REGION Network 54: PBV-82 CIP ISOLATION
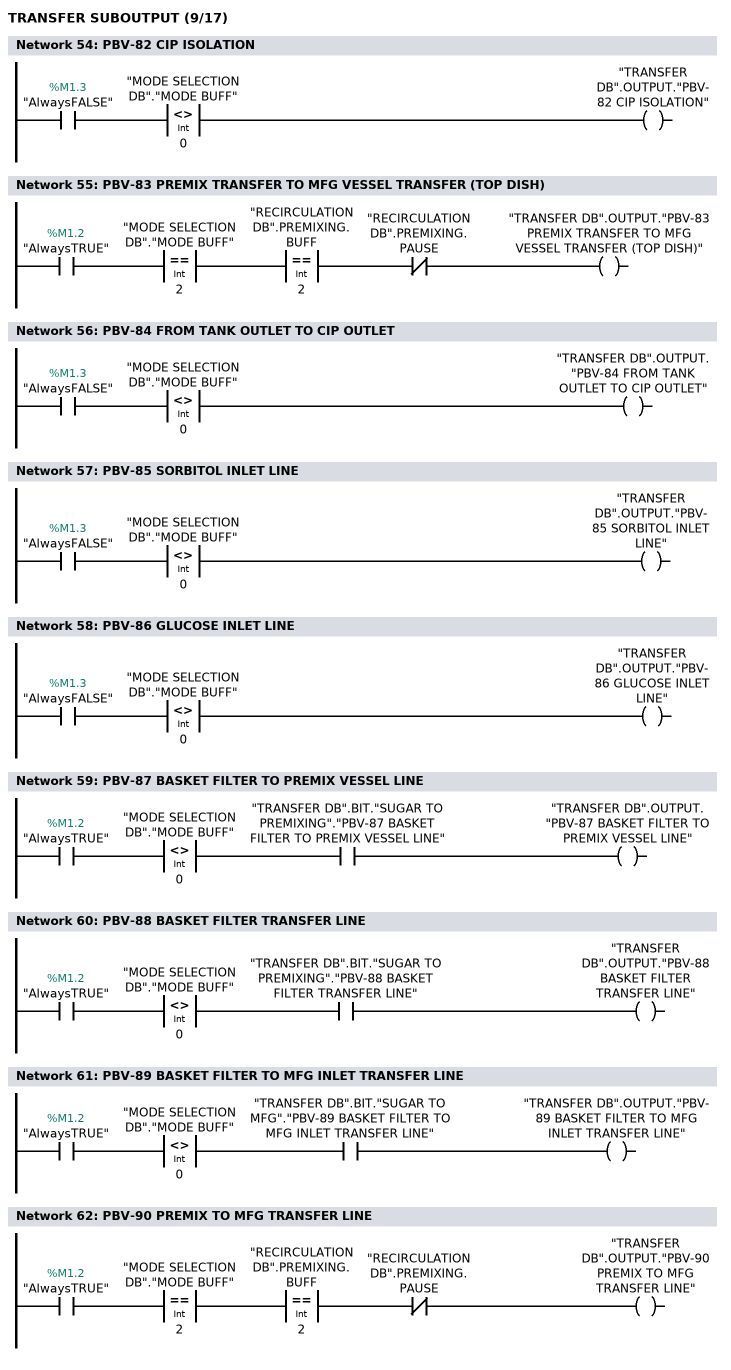
   RUNG wire#powerrail
      Contact( "AlwaysFALSE" )
      { S7_Templates := "SrcType := Int" } NE_Contact(in1 := "MODE SELECTION DB"."MODE BUFF", in2 := 0)
      Coil( "TRANSFER DB".OUTPUT."PBV-82 CIP ISOLATION" )
   END_RUNG
   // the same network as SCL:
   "TRANSFER DB".OUTPUT."PBV-82 CIP ISOLATION" := "AlwaysFALSE" AND ("MODE SELECTION DB"."MODE BUFF" <> 0);
END_REGION

REGION Network 55: PBV-83 PREMIX TRANSFER TO MFG VESSEL TRANSFER (TOP DISH)
   RUNG wire#powerrail
      Contact( "AlwaysTRUE" )
      { S7_Templates := "SrcType := Int" } EQ_Contact(in1 := "MODE SELECTION DB"."MODE BUFF", in2 := 2)
      { S7_Templates := "SrcType := Int" } EQ_Contact(in1 := "RECIRCULATION DB".PREMIXING.BUFF, in2 := 2)
      I_Contact( "RECIRCULATION DB".PREMIXING.PAUSE )
      Coil( "TRANSFER DB".OUTPUT."PBV-83 PREMIX TRANSFER TO MFG VESSEL TRANSFER (TOP DISH)" )
   END_RUNG
   // the same network as SCL:
   "TRANSFER DB".OUTPUT."PBV-83 PREMIX TRANSFER TO MFG VESSEL TRANSFER (TOP DISH)" := "AlwaysTRUE" AND ("MODE SELECTION DB"."MODE BUFF" = 2) AND ("RECIRCULATION DB".PREMIXING.BUFF = 2) AND NOT "RECIRCULATION DB".PREMIXING.PAUSE;
END_REGION

REGION Network 56: PBV-84 FROM TANK OUTLET TO CIP OUTLET
   RUNG wire#powerrail
      Contact( "AlwaysFALSE" )
      { S7_Templates := "SrcType := Int" } NE_Contact(in1 := "MODE SELECTION DB"."MODE BUFF", in2 := 0)
      Coil( "TRANSFER DB".OUTPUT."PBV-84 FROM TANK OUTLET TO CIP OUTLET" )
   END_RUNG
   // the same network as SCL:
   "TRANSFER DB".OUTPUT."PBV-84 FROM TANK OUTLET TO CIP OUTLET" := "AlwaysFALSE" AND ("MODE SELECTION DB"."MODE BUFF" <> 0);
END_REGION

REGION Network 57: PBV-85 SORBITOL INLET LINE
   RUNG wire#powerrail
      Contact( "AlwaysFALSE" )
      { S7_Templates := "SrcType := Int" } NE_Contact(in1 := "MODE SELECTION DB"."MODE BUFF", in2 := 0)
      Coil( "TRANSFER DB".OUTPUT."PBV-85 SORBITOL INLET LINE" )
   END_RUNG
   // the same network as SCL:
   "TRANSFER DB".OUTPUT."PBV-85 SORBITOL INLET LINE" := "AlwaysFALSE" AND ("MODE SELECTION DB"."MODE BUFF" <> 0);
END_REGION

REGION Network 58: PBV-86 GLUCOSE INLET LINE
   RUNG wire#powerrail
      Contact( "AlwaysFALSE" )
      { S7_Templates := "SrcType := Int" } NE_Contact(in1 := "MODE SELECTION DB"."MODE BUFF", in2 := 0)
      Coil( "TRANSFER DB".OUTPUT."PBV-86 GLUCOSE INLET LINE" )
   END_RUNG
   // the same network as SCL:
   "TRANSFER DB".OUTPUT."PBV-86 GLUCOSE INLET LINE" := "AlwaysFALSE" AND ("MODE SELECTION DB"."MODE BUFF" <> 0);
END_REGION

REGION Network 59: PBV-87 BASKET FILTER TO PREMIX VESSEL LINE
   RUNG wire#powerrail
      Contact( "AlwaysTRUE" )
      { S7_Templates := "SrcType := Int" } NE_Contact(in1 := "MODE SELECTION DB"."MODE BUFF", in2 := 0)
      Contact( "TRANSFER DB".BIT."SUGAR TO PREMIXING"."PBV-87 BASKET FILTER TO PREMIX VESSEL LINE" )
      Coil( "TRANSFER DB".OUTPUT."PBV-87 BASKET FILTER TO PREMIX VESSEL LINE" )
   END_RUNG
   // the same network as SCL:
   "TRANSFER DB".OUTPUT."PBV-87 BASKET FILTER TO PREMIX VESSEL LINE" := "AlwaysTRUE" AND ("MODE SELECTION DB"."MODE BUFF" <> 0) AND "TRANSFER DB".BIT."SUGAR TO PREMIXING"."PBV-87 BASKET FILTER TO PREMIX VESSEL LINE";
END_REGION

REGION Network 60: PBV-88 BASKET FILTER TRANSFER LINE
   RUNG wire#powerrail
      Contact( "AlwaysTRUE" )
      { S7_Templates := "SrcType := Int" } NE_Contact(in1 := "MODE SELECTION DB"."MODE BUFF", in2 := 0)
      Contact( "TRANSFER DB".BIT."SUGAR TO PREMIXING"."PBV-88 BASKET FILTER TRANSFER LINE" )
      Coil( "TRANSFER DB".OUTPUT."PBV-88 BASKET FILTER TRANSFER LINE" )
   END_RUNG
   // the same network as SCL:
   "TRANSFER DB".OUTPUT."PBV-88 BASKET FILTER TRANSFER LINE" := "AlwaysTRUE" AND ("MODE SELECTION DB"."MODE BUFF" <> 0) AND "TRANSFER DB".BIT."SUGAR TO PREMIXING"."PBV-88 BASKET FILTER TRANSFER LINE";
END_REGION

REGION Network 61: PBV-89 BASKET FILTER TO MFG INLET TRANSFER LINE
   RUNG wire#powerrail
      Contact( "AlwaysTRUE" )
      { S7_Templates := "SrcType := Int" } NE_Contact(in1 := "MODE SELECTION DB"."MODE BUFF", in2 := 0)
      Contact( "TRANSFER DB".BIT."SUGAR TO MFG"."PBV-89 BASKET FILTER TO MFG INLET TRANSFER LINE" )
      Coil( "TRANSFER DB".OUTPUT."PBV-89 BASKET FILTER TO MFG INLET TRANSFER LINE" )
   END_RUNG
   // the same network as SCL:
   "TRANSFER DB".OUTPUT."PBV-89 BASKET FILTER TO MFG INLET TRANSFER LINE" := "AlwaysTRUE" AND ("MODE SELECTION DB"."MODE BUFF" <> 0) AND "TRANSFER DB".BIT."SUGAR TO MFG"."PBV-89 BASKET FILTER TO MFG INLET TRANSFER LINE";
END_REGION

REGION Network 62: PBV-90 PREMIX TO MFG TRANSFER LINE
   RUNG wire#powerrail
      Contact( "AlwaysTRUE" )
      { S7_Templates := "SrcType := Int" } EQ_Contact(in1 := "MODE SELECTION DB"."MODE BUFF", in2 := 2)
      { S7_Templates := "SrcType := Int" } EQ_Contact(in1 := "RECIRCULATION DB".PREMIXING.BUFF, in2 := 2)
      I_Contact( "RECIRCULATION DB".PREMIXING.PAUSE )
      Coil( "TRANSFER DB".OUTPUT."PBV-90 PREMIX TO MFG TRANSFER LINE" )
   END_RUNG
   // the same network as SCL:
   "TRANSFER DB".OUTPUT."PBV-90 PREMIX TO MFG TRANSFER LINE" := "AlwaysTRUE" AND ("MODE SELECTION DB"."MODE BUFF" = 2) AND ("RECIRCULATION DB".PREMIXING.BUFF = 2) AND NOT "RECIRCULATION DB".PREMIXING.PAUSE;
END_REGION

REGION Network 63: PBV-91 PREMIX TO MFG TRANSFER LINE
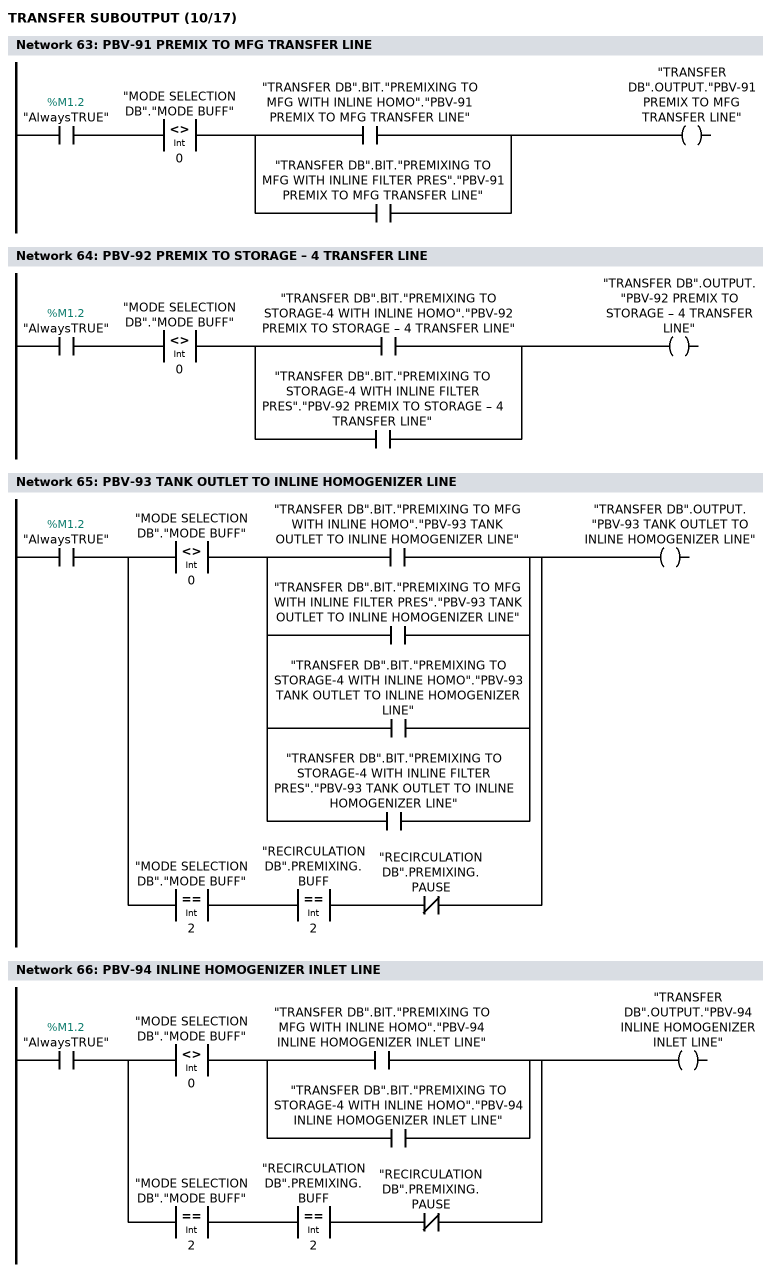
   RUNG wire#powerrail
      Contact( "AlwaysTRUE" )
      { S7_Templates := "SrcType := Int" } NE_Contact(in1 := "MODE SELECTION DB"."MODE BUFF", in2 := 0)
      wire#w1
      Contact( "TRANSFER DB".BIT."PREMIXING TO MFG WITH INLINE HOMO"."PBV-91 PREMIX TO MFG TRANSFER LINE" )
      wire#w2
      Coil( "TRANSFER DB".OUTPUT."PBV-91 PREMIX TO MFG TRANSFER LINE" )
   END_RUNG
   RUNG wire#w1
      Contact( "TRANSFER DB".BIT."PREMIXING TO MFG WITH INLINE FILTER PRES"."PBV-91 PREMIX TO MFG TRANSFER LINE" )
   END_RUNG wire#w2
   // the same network as SCL:
   "TRANSFER DB".OUTPUT."PBV-91 PREMIX TO MFG TRANSFER LINE" := "AlwaysTRUE" AND ("MODE SELECTION DB"."MODE BUFF" <> 0) AND ("TRANSFER DB".BIT."PREMIXING TO MFG WITH INLINE HOMO"."PBV-91 PREMIX TO MFG TRANSFER LINE" OR "TRANSFER DB".BIT."PREMIXING TO MFG WITH INLINE FILTER PRES"."PBV-91 PREMIX TO MFG TRANSFER LINE");
END_REGION

REGION Network 64: PBV-92 PREMIX TO STORAGE – 4 TRANSFER LINE
   RUNG wire#powerrail
      Contact( "AlwaysTRUE" )
      { S7_Templates := "SrcType := Int" } NE_Contact(in1 := "MODE SELECTION DB"."MODE BUFF", in2 := 0)
      wire#w1
      Contact( "TRANSFER DB".BIT."PREMIXING TO STORAGE-4 WITH INLINE HOMO"."PBV-92 PREMIX TO STORAGE – 4 TRANSFER LINE" )
      wire#w2
      Coil( "TRANSFER DB".OUTPUT."PBV-92 PREMIX TO STORAGE – 4 TRANSFER LINE" )
   END_RUNG
   RUNG wire#w1
      Contact( "TRANSFER DB".BIT."PREMIXING TO STORAGE-4 WITH INLINE FILTER PRES"."PBV-92 PREMIX TO STORAGE – 4 TRANSFER LINE" )
   END_RUNG wire#w2
   // the same network as SCL:
   "TRANSFER DB".OUTPUT."PBV-92 PREMIX TO STORAGE – 4 TRANSFER LINE" := "AlwaysTRUE" AND ("MODE SELECTION DB"."MODE BUFF" <> 0) AND ("TRANSFER DB".BIT."PREMIXING TO STORAGE-4 WITH INLINE HOMO"."PBV-92 PREMIX TO STORAGE – 4 TRANSFER LINE" OR "TRANSFER DB".BIT."PREMIXING TO STORAGE-4 WITH INLINE FILTER PRES"."PBV-92 PREMIX TO STORAGE – 4 TRANSFER LINE");
END_REGION

REGION Network 65: PBV-93 TANK OUTLET TO INLINE HOMOGENIZER LINE
   RUNG wire#powerrail
      Contact( "AlwaysTRUE" )
      wire#w1
      { S7_Templates := "SrcType := Int" } NE_Contact(in1 := "MODE SELECTION DB"."MODE BUFF", in2 := 0)
      wire#w2
      Contact( "TRANSFER DB".BIT."PREMIXING TO MFG WITH INLINE HOMO"."PBV-93 TANK OUTLET TO INLINE HOMOGENIZER LINE" )
      wire#w3
      Coil( "TRANSFER DB".OUTPUT."PBV-93 TANK OUTLET TO INLINE HOMOGENIZER LINE" )
   END_RUNG
   RUNG wire#w2
      Contact( "TRANSFER DB".BIT."PREMIXING TO MFG WITH INLINE FILTER PRES"."PBV-93 TANK OUTLET TO INLINE HOMOGENIZER LINE" )
   END_RUNG wire#w3
   RUNG wire#w2
      Contact( "TRANSFER DB".BIT."PREMIXING TO STORAGE-4 WITH INLINE HOMO"."PBV-93 TANK OUTLET TO INLINE HOMOGENIZER LINE" )
   END_RUNG wire#w3
   RUNG wire#w2
      Contact( "TRANSFER DB".BIT."PREMIXING TO STORAGE-4 WITH INLINE FILTER PRES"."PBV-93 TANK OUTLET TO INLINE HOMOGENIZER LINE" )
   END_RUNG wire#w3
   RUNG wire#w1
      { S7_Templates := "SrcType := Int" } EQ_Contact(in1 := "MODE SELECTION DB"."MODE BUFF", in2 := 2)
      { S7_Templates := "SrcType := Int" } EQ_Contact(in1 := "RECIRCULATION DB".PREMIXING.BUFF, in2 := 2)
      I_Contact( "RECIRCULATION DB".PREMIXING.PAUSE )
   END_RUNG wire#w3
   // the same network as SCL:
   "TRANSFER DB".OUTPUT."PBV-93 TANK OUTLET TO INLINE HOMOGENIZER LINE" := "AlwaysTRUE" AND ((("MODE SELECTION DB"."MODE BUFF" <> 0) AND ("TRANSFER DB".BIT."PREMIXING TO MFG WITH INLINE HOMO"."PBV-93 TANK OUTLET TO INLINE HOMOGENIZER LINE" OR "TRANSFER DB".BIT."PREMIXING TO MFG WITH INLINE FILTER PRES"."PBV-93 TANK OUTLET TO INLINE HOMOGENIZER LINE" OR "TRANSFER DB".BIT."PREMIXING TO STORAGE-4 WITH INLINE HOMO"."PBV-93 TANK OUTLET TO INLINE HOMOGENIZER LINE" OR "TRANSFER DB".BIT."PREMIXING TO STORAGE-4 WITH INLINE FILTER PRES"."PBV-93 TANK OUTLET TO INLINE HOMOGENIZER LINE")) OR (("MODE SELECTION DB"."MODE BUFF" = 2) AND ("RECIRCULATION DB".PREMIXING.BUFF = 2) AND NOT "RECIRCULATION DB".PREMIXING.PAUSE));
END_REGION

REGION Network 66: PBV-94 INLINE HOMOGENIZER INLET LINE
   RUNG wire#powerrail
      Contact( "AlwaysTRUE" )
      wire#w1
      { S7_Templates := "SrcType := Int" } NE_Contact(in1 := "MODE SELECTION DB"."MODE BUFF", in2 := 0)
      wire#w2
      Contact( "TRANSFER DB".BIT."PREMIXING TO MFG WITH INLINE HOMO"."PBV-94 INLINE HOMOGENIZER INLET LINE" )
      wire#w3
      Coil( "TRANSFER DB".OUTPUT."PBV-94 INLINE HOMOGENIZER INLET LINE" )
   END_RUNG
   RUNG wire#w2
      Contact( "TRANSFER DB".BIT."PREMIXING TO STORAGE-4 WITH INLINE HOMO"."PBV-94 INLINE HOMOGENIZER INLET LINE" )
   END_RUNG wire#w3
   RUNG wire#w1
      { S7_Templates := "SrcType := Int" } EQ_Contact(in1 := "MODE SELECTION DB"."MODE BUFF", in2 := 2)
      { S7_Templates := "SrcType := Int" } EQ_Contact(in1 := "RECIRCULATION DB".PREMIXING.BUFF, in2 := 2)
      I_Contact( "RECIRCULATION DB".PREMIXING.PAUSE )
   END_RUNG wire#w3
   // the same network as SCL:
   "TRANSFER DB".OUTPUT."PBV-94 INLINE HOMOGENIZER INLET LINE" := "AlwaysTRUE" AND ((("MODE SELECTION DB"."MODE BUFF" <> 0) AND ("TRANSFER DB".BIT."PREMIXING TO MFG WITH INLINE HOMO"."PBV-94 INLINE HOMOGENIZER INLET LINE" OR "TRANSFER DB".BIT."PREMIXING TO STORAGE-4 WITH INLINE HOMO"."PBV-94 INLINE HOMOGENIZER INLET LINE")) OR (("MODE SELECTION DB"."MODE BUFF" = 2) AND ("RECIRCULATION DB".PREMIXING.BUFF = 2) AND NOT "RECIRCULATION DB".PREMIXING.PAUSE));
END_REGION

REGION Network 67: PBV-95 TANK OUTLET TO FILTER PRESS LINE
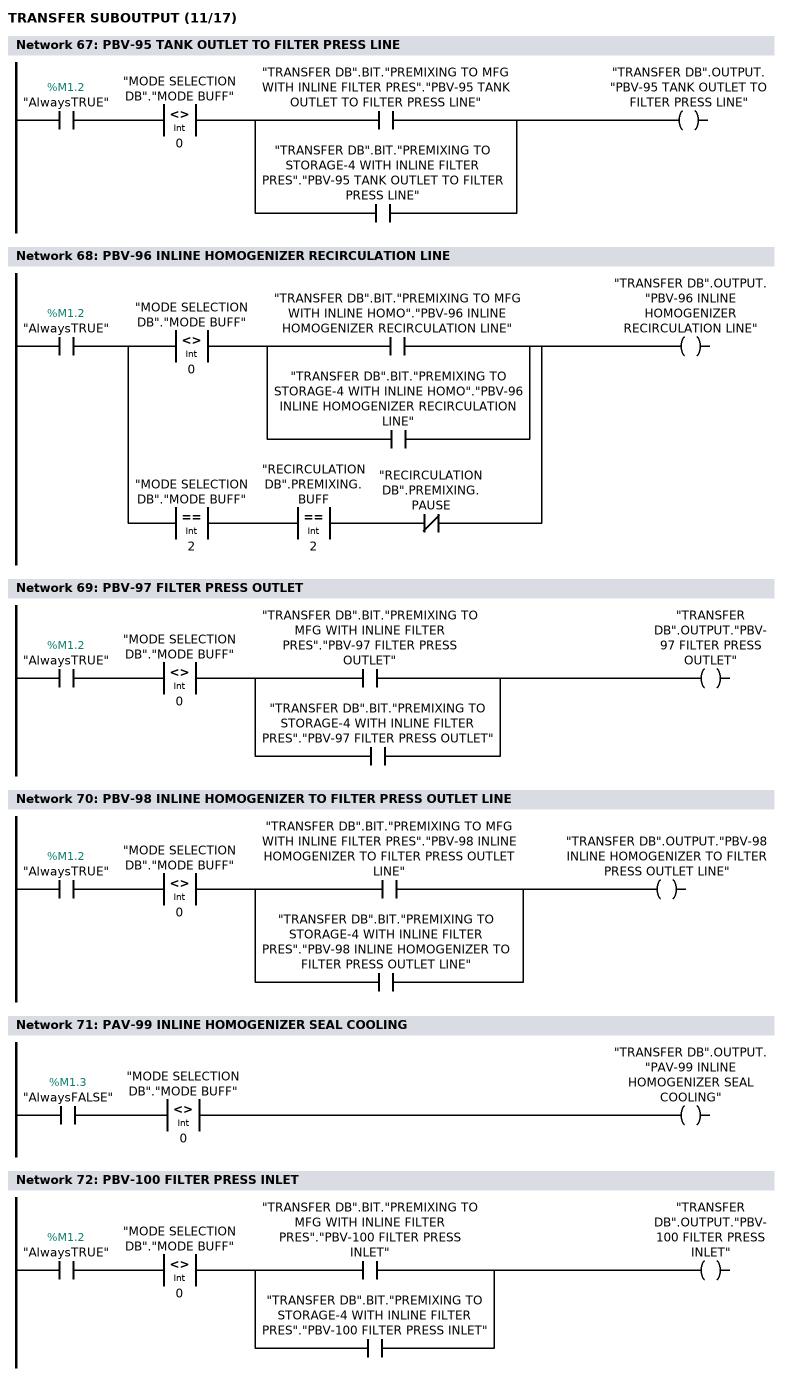
   RUNG wire#powerrail
      Contact( "AlwaysTRUE" )
      { S7_Templates := "SrcType := Int" } NE_Contact(in1 := "MODE SELECTION DB"."MODE BUFF", in2 := 0)
      wire#w1
      Contact( "TRANSFER DB".BIT."PREMIXING TO MFG WITH INLINE FILTER PRES"."PBV-95 TANK OUTLET TO FILTER PRESS LINE" )
      wire#w2
      Coil( "TRANSFER DB".OUTPUT."PBV-95 TANK OUTLET TO FILTER PRESS LINE" )
   END_RUNG
   RUNG wire#w1
      Contact( "TRANSFER DB".BIT."PREMIXING TO STORAGE-4 WITH INLINE FILTER PRES"."PBV-95 TANK OUTLET TO FILTER PRESS LINE" )
   END_RUNG wire#w2
   // the same network as SCL:
   "TRANSFER DB".OUTPUT."PBV-95 TANK OUTLET TO FILTER PRESS LINE" := "AlwaysTRUE" AND ("MODE SELECTION DB"."MODE BUFF" <> 0) AND ("TRANSFER DB".BIT."PREMIXING TO MFG WITH INLINE FILTER PRES"."PBV-95 TANK OUTLET TO FILTER PRESS LINE" OR "TRANSFER DB".BIT."PREMIXING TO STORAGE-4 WITH INLINE FILTER PRES"."PBV-95 TANK OUTLET TO FILTER PRESS LINE");
END_REGION

REGION Network 68: PBV-96 INLINE HOMOGENIZER RECIRCULATION LINE
   RUNG wire#powerrail
      Contact( "AlwaysTRUE" )
      wire#w1
      { S7_Templates := "SrcType := Int" } NE_Contact(in1 := "MODE SELECTION DB"."MODE BUFF", in2 := 0)
      wire#w2
      Contact( "TRANSFER DB".BIT."PREMIXING TO MFG WITH INLINE HOMO"."PBV-96 INLINE HOMOGENIZER RECIRCULATION LINE" )
      wire#w3
      Coil( "TRANSFER DB".OUTPUT."PBV-96 INLINE HOMOGENIZER RECIRCULATION LINE" )
   END_RUNG
   RUNG wire#w2
      Contact( "TRANSFER DB".BIT."PREMIXING TO STORAGE-4 WITH INLINE HOMO"."PBV-96 INLINE HOMOGENIZER RECIRCULATION LINE" )
   END_RUNG wire#w3
   RUNG wire#w1
      { S7_Templates := "SrcType := Int" } EQ_Contact(in1 := "MODE SELECTION DB"."MODE BUFF", in2 := 2)
      { S7_Templates := "SrcType := Int" } EQ_Contact(in1 := "RECIRCULATION DB".PREMIXING.BUFF, in2 := 2)
      I_Contact( "RECIRCULATION DB".PREMIXING.PAUSE )
   END_RUNG wire#w3
   // the same network as SCL:
   "TRANSFER DB".OUTPUT."PBV-96 INLINE HOMOGENIZER RECIRCULATION LINE" := "AlwaysTRUE" AND ((("MODE SELECTION DB"."MODE BUFF" <> 0) AND ("TRANSFER DB".BIT."PREMIXING TO MFG WITH INLINE HOMO"."PBV-96 INLINE HOMOGENIZER RECIRCULATION LINE" OR "TRANSFER DB".BIT."PREMIXING TO STORAGE-4 WITH INLINE HOMO"."PBV-96 INLINE HOMOGENIZER RECIRCULATION LINE")) OR (("MODE SELECTION DB"."MODE BUFF" = 2) AND ("RECIRCULATION DB".PREMIXING.BUFF = 2) AND NOT "RECIRCULATION DB".PREMIXING.PAUSE));
END_REGION

REGION Network 69: PBV-97 FILTER PRESS OUTLET
   RUNG wire#powerrail
      Contact( "AlwaysTRUE" )
      { S7_Templates := "SrcType := Int" } NE_Contact(in1 := "MODE SELECTION DB"."MODE BUFF", in2 := 0)
      wire#w1
      Contact( "TRANSFER DB".BIT."PREMIXING TO MFG WITH INLINE FILTER PRES"."PBV-97 FILTER PRESS OUTLET" )
      wire#w2
      Coil( "TRANSFER DB".OUTPUT."PBV-97 FILTER PRESS OUTLET" )
   END_RUNG
   RUNG wire#w1
      Contact( "TRANSFER DB".BIT."PREMIXING TO STORAGE-4 WITH INLINE FILTER PRES"."PBV-97 FILTER PRESS OUTLET" )
   END_RUNG wire#w2
   // the same network as SCL:
   "TRANSFER DB".OUTPUT."PBV-97 FILTER PRESS OUTLET" := "AlwaysTRUE" AND ("MODE SELECTION DB"."MODE BUFF" <> 0) AND ("TRANSFER DB".BIT."PREMIXING TO MFG WITH INLINE FILTER PRES"."PBV-97 FILTER PRESS OUTLET" OR "TRANSFER DB".BIT."PREMIXING TO STORAGE-4 WITH INLINE FILTER PRES"."PBV-97 FILTER PRESS OUTLET");
END_REGION

REGION Network 70: PBV-98 INLINE HOMOGENIZER TO FILTER PRESS OUTLET LINE
   RUNG wire#powerrail
      Contact( "AlwaysTRUE" )
      { S7_Templates := "SrcType := Int" } NE_Contact(in1 := "MODE SELECTION DB"."MODE BUFF", in2 := 0)
      wire#w1
      Contact( "TRANSFER DB".BIT."PREMIXING TO MFG WITH INLINE FILTER PRES"."PBV-98 INLINE HOMOGENIZER TO FILTER PRESS OUTLET LINE" )
      wire#w2
      Coil( "TRANSFER DB".OUTPUT."PBV-98 INLINE HOMOGENIZER TO FILTER PRESS OUTLET LINE" )
   END_RUNG
   RUNG wire#w1
      Contact( "TRANSFER DB".BIT."PREMIXING TO STORAGE-4 WITH INLINE FILTER PRES"."PBV-98 INLINE HOMOGENIZER TO FILTER PRESS OUTLET LINE" )
   END_RUNG wire#w2
   // the same network as SCL:
   "TRANSFER DB".OUTPUT."PBV-98 INLINE HOMOGENIZER TO FILTER PRESS OUTLET LINE" := "AlwaysTRUE" AND ("MODE SELECTION DB"."MODE BUFF" <> 0) AND ("TRANSFER DB".BIT."PREMIXING TO MFG WITH INLINE FILTER PRES"."PBV-98 INLINE HOMOGENIZER TO FILTER PRESS OUTLET LINE" OR "TRANSFER DB".BIT."PREMIXING TO STORAGE-4 WITH INLINE FILTER PRES"."PBV-98 INLINE HOMOGENIZER TO FILTER PRESS OUTLET LINE");
END_REGION

REGION Network 71: PAV-99 INLINE HOMOGENIZER SEAL COOLING
   RUNG wire#powerrail
      Contact( "AlwaysFALSE" )
      { S7_Templates := "SrcType := Int" } NE_Contact(in1 := "MODE SELECTION DB"."MODE BUFF", in2 := 0)
      Coil( "TRANSFER DB".OUTPUT."PAV-99 INLINE HOMOGENIZER SEAL COOLING" )
   END_RUNG
   // the same network as SCL:
   "TRANSFER DB".OUTPUT."PAV-99 INLINE HOMOGENIZER SEAL COOLING" := "AlwaysFALSE" AND ("MODE SELECTION DB"."MODE BUFF" <> 0);
END_REGION

REGION Network 72: PBV-100 FILTER PRESS INLET
   RUNG wire#powerrail
      Contact( "AlwaysTRUE" )
      { S7_Templates := "SrcType := Int" } NE_Contact(in1 := "MODE SELECTION DB"."MODE BUFF", in2 := 0)
      wire#w1
      Contact( "TRANSFER DB".BIT."PREMIXING TO MFG WITH INLINE FILTER PRES"."PBV-100 FILTER PRESS INLET" )
      wire#w2
      Coil( "TRANSFER DB".OUTPUT."PBV-100 FILTER PRESS INLET" )
   END_RUNG
   RUNG wire#w1
      Contact( "TRANSFER DB".BIT."PREMIXING TO STORAGE-4 WITH INLINE FILTER PRES"."PBV-100 FILTER PRESS INLET" )
   END_RUNG wire#w2
   // the same network as SCL:
   "TRANSFER DB".OUTPUT."PBV-100 FILTER PRESS INLET" := "AlwaysTRUE" AND ("MODE SELECTION DB"."MODE BUFF" <> 0) AND ("TRANSFER DB".BIT."PREMIXING TO MFG WITH INLINE FILTER PRES"."PBV-100 FILTER PRESS INLET" OR "TRANSFER DB".BIT."PREMIXING TO STORAGE-4 WITH INLINE FILTER PRES"."PBV-100 FILTER PRESS INLET");
END_REGION

REGION Network 73: PBV-101 SUGAR MELTING TO MFG TRANSFER (TOP DISH)
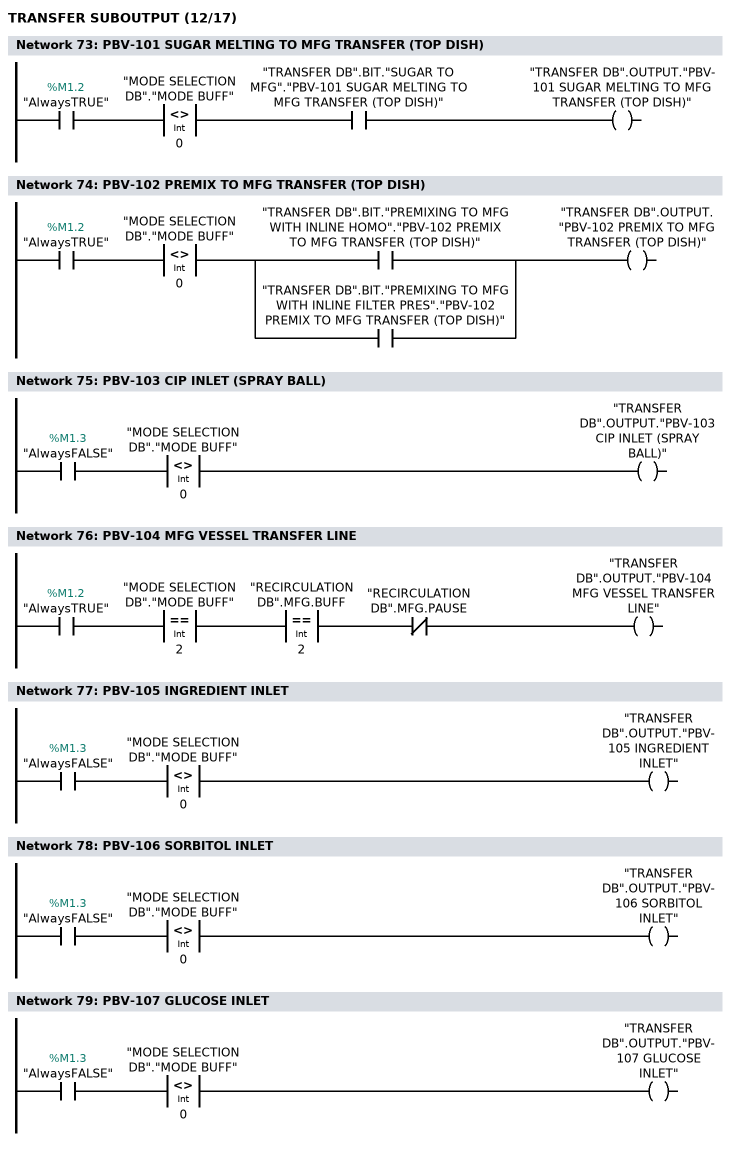
   RUNG wire#powerrail
      Contact( "AlwaysTRUE" )
      { S7_Templates := "SrcType := Int" } NE_Contact(in1 := "MODE SELECTION DB"."MODE BUFF", in2 := 0)
      Contact( "TRANSFER DB".BIT."SUGAR TO MFG"."PBV-101 SUGAR MELTING TO MFG TRANSFER (TOP DISH)" )
      Coil( "TRANSFER DB".OUTPUT."PBV-101 SUGAR MELTING TO MFG TRANSFER (TOP DISH)" )
   END_RUNG
   // the same network as SCL:
   "TRANSFER DB".OUTPUT."PBV-101 SUGAR MELTING TO MFG TRANSFER (TOP DISH)" := "AlwaysTRUE" AND ("MODE SELECTION DB"."MODE BUFF" <> 0) AND "TRANSFER DB".BIT."SUGAR TO MFG"."PBV-101 SUGAR MELTING TO MFG TRANSFER (TOP DISH)";
END_REGION

REGION Network 74: PBV-102 PREMIX TO MFG TRANSFER (TOP DISH)
   RUNG wire#powerrail
      Contact( "AlwaysTRUE" )
      { S7_Templates := "SrcType := Int" } NE_Contact(in1 := "MODE SELECTION DB"."MODE BUFF", in2 := 0)
      wire#w1
      Contact( "TRANSFER DB".BIT."PREMIXING TO MFG WITH INLINE HOMO"."PBV-102 PREMIX TO MFG TRANSFER (TOP DISH)" )
      wire#w2
      Coil( "TRANSFER DB".OUTPUT."PBV-102 PREMIX TO MFG TRANSFER (TOP DISH)" )
   END_RUNG
   RUNG wire#w1
      Contact( "TRANSFER DB".BIT."PREMIXING TO MFG WITH INLINE FILTER PRES"."PBV-102 PREMIX TO MFG TRANSFER (TOP DISH)" )
   END_RUNG wire#w2
   // the same network as SCL:
   "TRANSFER DB".OUTPUT."PBV-102 PREMIX TO MFG TRANSFER (TOP DISH)" := "AlwaysTRUE" AND ("MODE SELECTION DB"."MODE BUFF" <> 0) AND ("TRANSFER DB".BIT."PREMIXING TO MFG WITH INLINE HOMO"."PBV-102 PREMIX TO MFG TRANSFER (TOP DISH)" OR "TRANSFER DB".BIT."PREMIXING TO MFG WITH INLINE FILTER PRES"."PBV-102 PREMIX TO MFG TRANSFER (TOP DISH)");
END_REGION

REGION Network 75: PBV-103 CIP INLET (SPRAY BALL)
   RUNG wire#powerrail
      Contact( "AlwaysFALSE" )
      { S7_Templates := "SrcType := Int" } NE_Contact(in1 := "MODE SELECTION DB"."MODE BUFF", in2 := 0)
      Coil( "TRANSFER DB".OUTPUT."PBV-103 CIP INLET (SPRAY BALL)" )
   END_RUNG
   // the same network as SCL:
   "TRANSFER DB".OUTPUT."PBV-103 CIP INLET (SPRAY BALL)" := "AlwaysFALSE" AND ("MODE SELECTION DB"."MODE BUFF" <> 0);
END_REGION

REGION Network 76: PBV-104 MFG VESSEL TRANSFER LINE
   RUNG wire#powerrail
      Contact( "AlwaysTRUE" )
      { S7_Templates := "SrcType := Int" } EQ_Contact(in1 := "MODE SELECTION DB"."MODE BUFF", in2 := 2)
      { S7_Templates := "SrcType := Int" } EQ_Contact(in1 := "RECIRCULATION DB".MFG.BUFF, in2 := 2)
      I_Contact( "RECIRCULATION DB".MFG.PAUSE )
      Coil( "TRANSFER DB".OUTPUT."PBV-104 MFG VESSEL TRANSFER LINE" )
   END_RUNG
   // the same network as SCL:
   "TRANSFER DB".OUTPUT."PBV-104 MFG VESSEL TRANSFER LINE" := "AlwaysTRUE" AND ("MODE SELECTION DB"."MODE BUFF" = 2) AND ("RECIRCULATION DB".MFG.BUFF = 2) AND NOT "RECIRCULATION DB".MFG.PAUSE;
END_REGION

REGION Network 77: PBV-105 INGREDIENT INLET
   RUNG wire#powerrail
      Contact( "AlwaysFALSE" )
      { S7_Templates := "SrcType := Int" } NE_Contact(in1 := "MODE SELECTION DB"."MODE BUFF", in2 := 0)
      Coil( "TRANSFER DB".OUTPUT."PBV-105 INGREDIENT INLET" )
   END_RUNG
   // the same network as SCL:
   "TRANSFER DB".OUTPUT."PBV-105 INGREDIENT INLET" := "AlwaysFALSE" AND ("MODE SELECTION DB"."MODE BUFF" <> 0);
END_REGION

REGION Network 78: PBV-106 SORBITOL INLET
   RUNG wire#powerrail
      Contact( "AlwaysFALSE" )
      { S7_Templates := "SrcType := Int" } NE_Contact(in1 := "MODE SELECTION DB"."MODE BUFF", in2 := 0)
      Coil( "TRANSFER DB".OUTPUT."PBV-106 SORBITOL INLET" )
   END_RUNG
   // the same network as SCL:
   "TRANSFER DB".OUTPUT."PBV-106 SORBITOL INLET" := "AlwaysFALSE" AND ("MODE SELECTION DB"."MODE BUFF" <> 0);
END_REGION

REGION Network 79: PBV-107 GLUCOSE INLET
   RUNG wire#powerrail
      Contact( "AlwaysFALSE" )
      { S7_Templates := "SrcType := Int" } NE_Contact(in1 := "MODE SELECTION DB"."MODE BUFF", in2 := 0)
      Coil( "TRANSFER DB".OUTPUT."PBV-107 GLUCOSE INLET" )
   END_RUNG
   // the same network as SCL:
   "TRANSFER DB".OUTPUT."PBV-107 GLUCOSE INLET" := "AlwaysFALSE" AND ("MODE SELECTION DB"."MODE BUFF" <> 0);
END_REGION

REGION Network 80: PBV-108 INLINE HOMOGENIZER TO FILTER PRESS INLET LINE
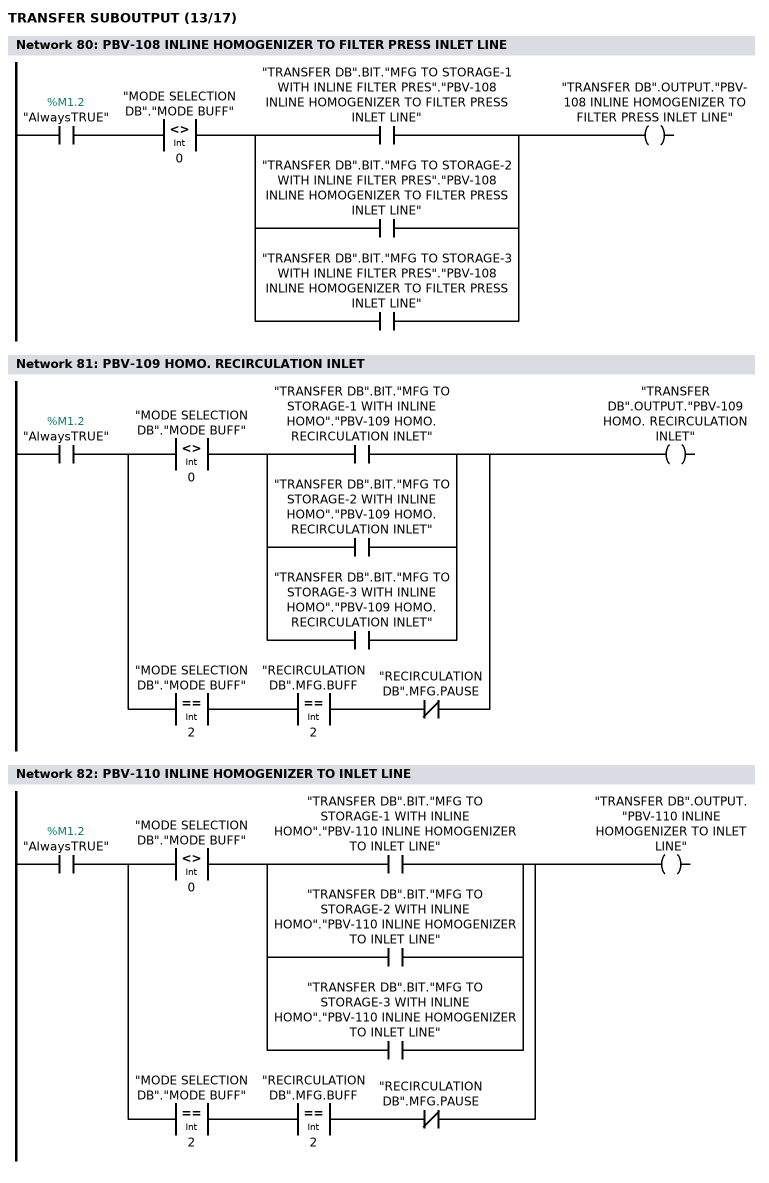
   RUNG wire#powerrail
      Contact( "AlwaysTRUE" )
      { S7_Templates := "SrcType := Int" } NE_Contact(in1 := "MODE SELECTION DB"."MODE BUFF", in2 := 0)
      wire#w1
      Contact( "TRANSFER DB".BIT."MFG TO STORAGE-1 WITH INLINE FILTER PRES"."PBV-108 INLINE HOMOGENIZER TO FILTER PRESS INLET LINE" )
      wire#w2
      Coil( "TRANSFER DB".OUTPUT."PBV-108 INLINE HOMOGENIZER TO FILTER PRESS INLET LINE" )
   END_RUNG
   RUNG wire#w1
      Contact( "TRANSFER DB".BIT."MFG TO STORAGE-2 WITH INLINE FILTER PRES"."PBV-108 INLINE HOMOGENIZER TO FILTER PRESS INLET LINE" )
   END_RUNG wire#w2
   RUNG wire#w1
      Contact( "TRANSFER DB".BIT."MFG TO STORAGE-3 WITH INLINE FILTER PRES"."PBV-108 INLINE HOMOGENIZER TO FILTER PRESS INLET LINE" )
   END_RUNG wire#w2
   // the same network as SCL:
   "TRANSFER DB".OUTPUT."PBV-108 INLINE HOMOGENIZER TO FILTER PRESS INLET LINE" := "AlwaysTRUE" AND ("MODE SELECTION DB"."MODE BUFF" <> 0) AND ("TRANSFER DB".BIT."MFG TO STORAGE-1 WITH INLINE FILTER PRES"."PBV-108 INLINE HOMOGENIZER TO FILTER PRESS INLET LINE" OR "TRANSFER DB".BIT."MFG TO STORAGE-2 WITH INLINE FILTER PRES"."PBV-108 INLINE HOMOGENIZER TO FILTER PRESS INLET LINE" OR "TRANSFER DB".BIT."MFG TO STORAGE-3 WITH INLINE FILTER PRES"."PBV-108 INLINE HOMOGENIZER TO FILTER PRESS INLET LINE");
END_REGION

REGION Network 81: PBV-109 HOMO. RECIRCULATION INLET
   RUNG wire#powerrail
      Contact( "AlwaysTRUE" )
      wire#w1
      { S7_Templates := "SrcType := Int" } NE_Contact(in1 := "MODE SELECTION DB"."MODE BUFF", in2 := 0)
      wire#w2
      Contact( "TRANSFER DB".BIT."MFG TO STORAGE-1 WITH INLINE HOMO"."PBV-109 HOMO. RECIRCULATION INLET" )
      wire#w3
      Coil( "TRANSFER DB".OUTPUT."PBV-109 HOMO. RECIRCULATION INLET" )
   END_RUNG
   RUNG wire#w2
      Contact( "TRANSFER DB".BIT."MFG TO STORAGE-2 WITH INLINE HOMO"."PBV-109 HOMO. RECIRCULATION INLET" )
   END_RUNG wire#w3
   RUNG wire#w2
      Contact( "TRANSFER DB".BIT."MFG TO STORAGE-3 WITH INLINE HOMO"."PBV-109 HOMO. RECIRCULATION INLET" )
   END_RUNG wire#w3
   RUNG wire#w1
      { S7_Templates := "SrcType := Int" } EQ_Contact(in1 := "MODE SELECTION DB"."MODE BUFF", in2 := 2)
      { S7_Templates := "SrcType := Int" } EQ_Contact(in1 := "RECIRCULATION DB".MFG.BUFF, in2 := 2)
      I_Contact( "RECIRCULATION DB".MFG.PAUSE )
   END_RUNG wire#w3
   // the same network as SCL:
   "TRANSFER DB".OUTPUT."PBV-109 HOMO. RECIRCULATION INLET" := "AlwaysTRUE" AND ((("MODE SELECTION DB"."MODE BUFF" <> 0) AND ("TRANSFER DB".BIT."MFG TO STORAGE-1 WITH INLINE HOMO"."PBV-109 HOMO. RECIRCULATION INLET" OR "TRANSFER DB".BIT."MFG TO STORAGE-2 WITH INLINE HOMO"."PBV-109 HOMO. RECIRCULATION INLET" OR "TRANSFER DB".BIT."MFG TO STORAGE-3 WITH INLINE HOMO"."PBV-109 HOMO. RECIRCULATION INLET")) OR (("MODE SELECTION DB"."MODE BUFF" = 2) AND ("RECIRCULATION DB".MFG.BUFF = 2) AND NOT "RECIRCULATION DB".MFG.PAUSE));
END_REGION

REGION Network 82: PBV-110 INLINE HOMOGENIZER TO INLET LINE
   RUNG wire#powerrail
      Contact( "AlwaysTRUE" )
      wire#w1
      { S7_Templates := "SrcType := Int" } NE_Contact(in1 := "MODE SELECTION DB"."MODE BUFF", in2 := 0)
      wire#w2
      Contact( "TRANSFER DB".BIT."MFG TO STORAGE-1 WITH INLINE HOMO"."PBV-110 INLINE HOMOGENIZER TO INLET LINE" )
      wire#w3
      Coil( "TRANSFER DB".OUTPUT."PBV-110 INLINE HOMOGENIZER TO INLET LINE" )
   END_RUNG
   RUNG wire#w2
      Contact( "TRANSFER DB".BIT."MFG TO STORAGE-2 WITH INLINE HOMO"."PBV-110 INLINE HOMOGENIZER TO INLET LINE" )
   END_RUNG wire#w3
   RUNG wire#w2
      Contact( "TRANSFER DB".BIT."MFG TO STORAGE-3 WITH INLINE HOMO"."PBV-110 INLINE HOMOGENIZER TO INLET LINE" )
   END_RUNG wire#w3
   RUNG wire#w1
      { S7_Templates := "SrcType := Int" } EQ_Contact(in1 := "MODE SELECTION DB"."MODE BUFF", in2 := 2)
      { S7_Templates := "SrcType := Int" } EQ_Contact(in1 := "RECIRCULATION DB".MFG.BUFF, in2 := 2)
      I_Contact( "RECIRCULATION DB".MFG.PAUSE )
   END_RUNG wire#w3
   // the same network as SCL:
   "TRANSFER DB".OUTPUT."PBV-110 INLINE HOMOGENIZER TO INLET LINE" := "AlwaysTRUE" AND ((("MODE SELECTION DB"."MODE BUFF" <> 0) AND ("TRANSFER DB".BIT."MFG TO STORAGE-1 WITH INLINE HOMO"."PBV-110 INLINE HOMOGENIZER TO INLET LINE" OR "TRANSFER DB".BIT."MFG TO STORAGE-2 WITH INLINE HOMO"."PBV-110 INLINE HOMOGENIZER TO INLET LINE" OR "TRANSFER DB".BIT."MFG TO STORAGE-3 WITH INLINE HOMO"."PBV-110 INLINE HOMOGENIZER TO INLET LINE")) OR (("MODE SELECTION DB"."MODE BUFF" = 2) AND ("RECIRCULATION DB".MFG.BUFF = 2) AND NOT "RECIRCULATION DB".MFG.PAUSE));
END_REGION

REGION Network 83: PBV-111 FILTER PRESS OUTLER VALVE
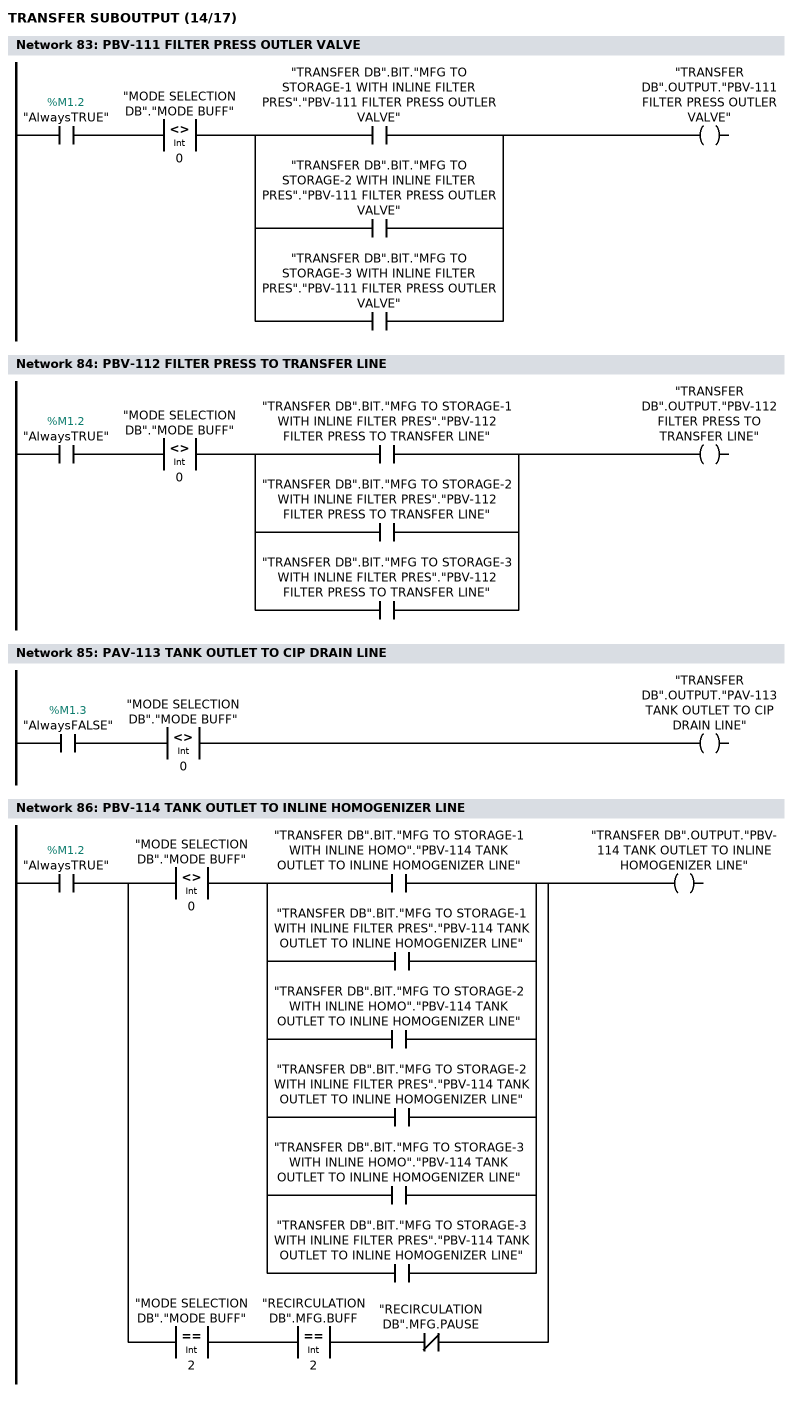
   RUNG wire#powerrail
      Contact( "AlwaysTRUE" )
      { S7_Templates := "SrcType := Int" } NE_Contact(in1 := "MODE SELECTION DB"."MODE BUFF", in2 := 0)
      wire#w1
      Contact( "TRANSFER DB".BIT."MFG TO STORAGE-1 WITH INLINE FILTER PRES"."PBV-111 FILTER PRESS OUTLER VALVE" )
      wire#w2
      Coil( "TRANSFER DB".OUTPUT."PBV-111 FILTER PRESS OUTLER VALVE" )
   END_RUNG
   RUNG wire#w1
      Contact( "TRANSFER DB".BIT."MFG TO STORAGE-2 WITH INLINE FILTER PRES"."PBV-111 FILTER PRESS OUTLER VALVE" )
   END_RUNG wire#w2
   RUNG wire#w1
      Contact( "TRANSFER DB".BIT."MFG TO STORAGE-3 WITH INLINE FILTER PRES"."PBV-111 FILTER PRESS OUTLER VALVE" )
   END_RUNG wire#w2
   // the same network as SCL:
   "TRANSFER DB".OUTPUT."PBV-111 FILTER PRESS OUTLER VALVE" := "AlwaysTRUE" AND ("MODE SELECTION DB"."MODE BUFF" <> 0) AND ("TRANSFER DB".BIT."MFG TO STORAGE-1 WITH INLINE FILTER PRES"."PBV-111 FILTER PRESS OUTLER VALVE" OR "TRANSFER DB".BIT."MFG TO STORAGE-2 WITH INLINE FILTER PRES"."PBV-111 FILTER PRESS OUTLER VALVE" OR "TRANSFER DB".BIT."MFG TO STORAGE-3 WITH INLINE FILTER PRES"."PBV-111 FILTER PRESS OUTLER VALVE");
END_REGION

REGION Network 84: PBV-112 FILTER PRESS TO TRANSFER LINE
   RUNG wire#powerrail
      Contact( "AlwaysTRUE" )
      { S7_Templates := "SrcType := Int" } NE_Contact(in1 := "MODE SELECTION DB"."MODE BUFF", in2 := 0)
      wire#w1
      Contact( "TRANSFER DB".BIT."MFG TO STORAGE-1 WITH INLINE FILTER PRES"."PBV-112 FILTER PRESS TO TRANSFER LINE" )
      wire#w2
      Coil( "TRANSFER DB".OUTPUT."PBV-112 FILTER PRESS TO TRANSFER LINE" )
   END_RUNG
   RUNG wire#w1
      Contact( "TRANSFER DB".BIT."MFG TO STORAGE-2 WITH INLINE FILTER PRES"."PBV-112 FILTER PRESS TO TRANSFER LINE" )
   END_RUNG wire#w2
   RUNG wire#w1
      Contact( "TRANSFER DB".BIT."MFG TO STORAGE-3 WITH INLINE FILTER PRES"."PBV-112 FILTER PRESS TO TRANSFER LINE" )
   END_RUNG wire#w2
   // the same network as SCL:
   "TRANSFER DB".OUTPUT."PBV-112 FILTER PRESS TO TRANSFER LINE" := "AlwaysTRUE" AND ("MODE SELECTION DB"."MODE BUFF" <> 0) AND ("TRANSFER DB".BIT."MFG TO STORAGE-1 WITH INLINE FILTER PRES"."PBV-112 FILTER PRESS TO TRANSFER LINE" OR "TRANSFER DB".BIT."MFG TO STORAGE-2 WITH INLINE FILTER PRES"."PBV-112 FILTER PRESS TO TRANSFER LINE" OR "TRANSFER DB".BIT."MFG TO STORAGE-3 WITH INLINE FILTER PRES"."PBV-112 FILTER PRESS TO TRANSFER LINE");
END_REGION

REGION Network 85: PAV-113 TANK OUTLET TO CIP DRAIN LINE
   RUNG wire#powerrail
      Contact( "AlwaysFALSE" )
      { S7_Templates := "SrcType := Int" } NE_Contact(in1 := "MODE SELECTION DB"."MODE BUFF", in2 := 0)
      Coil( "TRANSFER DB".OUTPUT."PAV-113 TANK OUTLET TO CIP DRAIN LINE" )
   END_RUNG
   // the same network as SCL:
   "TRANSFER DB".OUTPUT."PAV-113 TANK OUTLET TO CIP DRAIN LINE" := "AlwaysFALSE" AND ("MODE SELECTION DB"."MODE BUFF" <> 0);
END_REGION

REGION Network 86: PBV-114 TANK OUTLET TO INLINE HOMOGENIZER LINE
   RUNG wire#powerrail
      Contact( "AlwaysTRUE" )
      wire#w1
      { S7_Templates := "SrcType := Int" } NE_Contact(in1 := "MODE SELECTION DB"."MODE BUFF", in2 := 0)
      wire#w2
      Contact( "TRANSFER DB".BIT."MFG TO STORAGE-1 WITH INLINE HOMO"."PBV-114 TANK OUTLET TO INLINE HOMOGENIZER LINE" )
      wire#w3
      Coil( "TRANSFER DB".OUTPUT."PBV-114 TANK OUTLET TO INLINE HOMOGENIZER LINE" )
   END_RUNG
   RUNG wire#w2
      Contact( "TRANSFER DB".BIT."MFG TO STORAGE-1 WITH INLINE FILTER PRES"."PBV-114 TANK OUTLET TO INLINE HOMOGENIZER LINE" )
   END_RUNG wire#w3
   RUNG wire#w2
      Contact( "TRANSFER DB".BIT."MFG TO STORAGE-2 WITH INLINE HOMO"."PBV-114 TANK OUTLET TO INLINE HOMOGENIZER LINE" )
   END_RUNG wire#w3
   RUNG wire#w2
      Contact( "TRANSFER DB".BIT."MFG TO STORAGE-2 WITH INLINE FILTER PRES"."PBV-114 TANK OUTLET TO INLINE HOMOGENIZER LINE" )
   END_RUNG wire#w3
   RUNG wire#w2
      Contact( "TRANSFER DB".BIT."MFG TO STORAGE-3 WITH INLINE HOMO"."PBV-114 TANK OUTLET TO INLINE HOMOGENIZER LINE" )
   END_RUNG wire#w3
   RUNG wire#w2
      Contact( "TRANSFER DB".BIT."MFG TO STORAGE-3 WITH INLINE FILTER PRES"."PBV-114 TANK OUTLET TO INLINE HOMOGENIZER LINE" )
   END_RUNG wire#w3
   RUNG wire#w1
      { S7_Templates := "SrcType := Int" } EQ_Contact(in1 := "MODE SELECTION DB"."MODE BUFF", in2 := 2)
      { S7_Templates := "SrcType := Int" } EQ_Contact(in1 := "RECIRCULATION DB".MFG.BUFF, in2 := 2)
      I_Contact( "RECIRCULATION DB".MFG.PAUSE )
   END_RUNG wire#w3
   // the same network as SCL:
   "TRANSFER DB".OUTPUT."PBV-114 TANK OUTLET TO INLINE HOMOGENIZER LINE" := "AlwaysTRUE" AND ((("MODE SELECTION DB"."MODE BUFF" <> 0) AND ("TRANSFER DB".BIT."MFG TO STORAGE-1 WITH INLINE HOMO"."PBV-114 TANK OUTLET TO INLINE HOMOGENIZER LINE" OR "TRANSFER DB".BIT."MFG TO STORAGE-1 WITH INLINE FILTER PRES"."PBV-114 TANK OUTLET TO INLINE HOMOGENIZER LINE" OR "TRANSFER DB".BIT."MFG TO STORAGE-2 WITH INLINE HOMO"."PBV-114 TANK OUTLET TO INLINE HOMOGENIZER LINE" OR "TRANSFER DB".BIT."MFG TO STORAGE-2 WITH INLINE FILTER PRES"."PBV-114 TANK OUTLET TO INLINE HOMOGENIZER LINE" OR "TRANSFER DB".BIT."MFG TO STORAGE-3 WITH INLINE HOMO"."PBV-114 TANK OUTLET TO INLINE HOMOGENIZER LINE" OR "TRANSFER DB".BIT."MFG TO STORAGE-3 WITH INLINE FILTER PRES"."PBV-114 TANK OUTLET TO INLINE HOMOGENIZER LINE")) OR (("MODE SELECTION DB"."MODE BUFF" = 2) AND ("RECIRCULATION DB".MFG.BUFF = 2) AND NOT "RECIRCULATION DB".MFG.PAUSE));
END_REGION

REGION Network 87: PBV-115 MFG TO STORAGE – 1 TRANSFER LINE
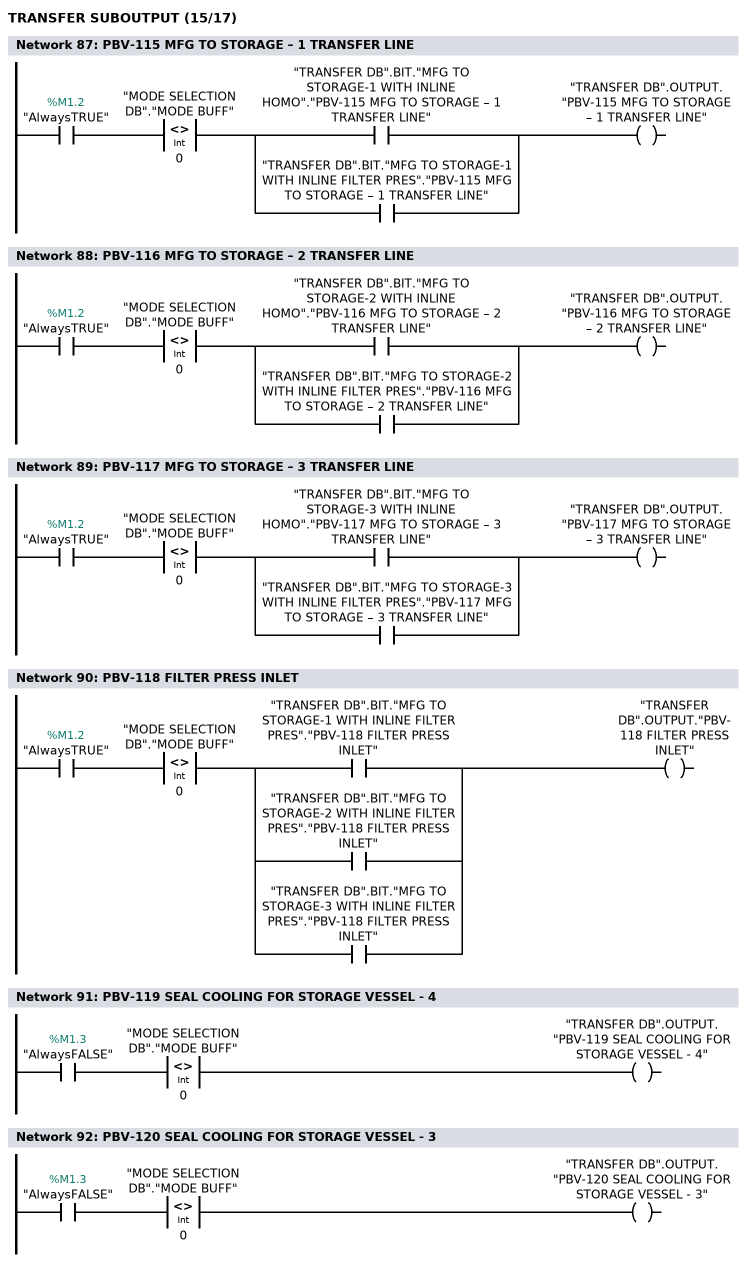
   RUNG wire#powerrail
      Contact( "AlwaysTRUE" )
      { S7_Templates := "SrcType := Int" } NE_Contact(in1 := "MODE SELECTION DB"."MODE BUFF", in2 := 0)
      wire#w1
      Contact( "TRANSFER DB".BIT."MFG TO STORAGE-1 WITH INLINE HOMO"."PBV-115 MFG TO STORAGE – 1 TRANSFER LINE" )
      wire#w2
      Coil( "TRANSFER DB".OUTPUT."PBV-115 MFG TO STORAGE – 1 TRANSFER LINE" )
   END_RUNG
   RUNG wire#w1
      Contact( "TRANSFER DB".BIT."MFG TO STORAGE-1 WITH INLINE FILTER PRES"."PBV-115 MFG TO STORAGE – 1 TRANSFER LINE" )
   END_RUNG wire#w2
   // the same network as SCL:
   "TRANSFER DB".OUTPUT."PBV-115 MFG TO STORAGE – 1 TRANSFER LINE" := "AlwaysTRUE" AND ("MODE SELECTION DB"."MODE BUFF" <> 0) AND ("TRANSFER DB".BIT."MFG TO STORAGE-1 WITH INLINE HOMO"."PBV-115 MFG TO STORAGE – 1 TRANSFER LINE" OR "TRANSFER DB".BIT."MFG TO STORAGE-1 WITH INLINE FILTER PRES"."PBV-115 MFG TO STORAGE – 1 TRANSFER LINE");
END_REGION

REGION Network 88: PBV-116 MFG TO STORAGE – 2 TRANSFER LINE
   RUNG wire#powerrail
      Contact( "AlwaysTRUE" )
      { S7_Templates := "SrcType := Int" } NE_Contact(in1 := "MODE SELECTION DB"."MODE BUFF", in2 := 0)
      wire#w1
      Contact( "TRANSFER DB".BIT."MFG TO STORAGE-2 WITH INLINE HOMO"."PBV-116 MFG TO STORAGE – 2 TRANSFER LINE" )
      wire#w2
      Coil( "TRANSFER DB".OUTPUT."PBV-116 MFG TO STORAGE – 2 TRANSFER LINE" )
   END_RUNG
   RUNG wire#w1
      Contact( "TRANSFER DB".BIT."MFG TO STORAGE-2 WITH INLINE FILTER PRES"."PBV-116 MFG TO STORAGE – 2 TRANSFER LINE" )
   END_RUNG wire#w2
   // the same network as SCL:
   "TRANSFER DB".OUTPUT."PBV-116 MFG TO STORAGE – 2 TRANSFER LINE" := "AlwaysTRUE" AND ("MODE SELECTION DB"."MODE BUFF" <> 0) AND ("TRANSFER DB".BIT."MFG TO STORAGE-2 WITH INLINE HOMO"."PBV-116 MFG TO STORAGE – 2 TRANSFER LINE" OR "TRANSFER DB".BIT."MFG TO STORAGE-2 WITH INLINE FILTER PRES"."PBV-116 MFG TO STORAGE – 2 TRANSFER LINE");
END_REGION

REGION Network 89: PBV-117 MFG TO STORAGE – 3 TRANSFER LINE
   RUNG wire#powerrail
      Contact( "AlwaysTRUE" )
      { S7_Templates := "SrcType := Int" } NE_Contact(in1 := "MODE SELECTION DB"."MODE BUFF", in2 := 0)
      wire#w1
      Contact( "TRANSFER DB".BIT."MFG TO STORAGE-3 WITH INLINE HOMO"."PBV-117 MFG TO STORAGE – 3 TRANSFER LINE" )
      wire#w2
      Coil( "TRANSFER DB".OUTPUT."PBV-117 MFG TO STORAGE – 3 TRANSFER LINE" )
   END_RUNG
   RUNG wire#w1
      Contact( "TRANSFER DB".BIT."MFG TO STORAGE-3 WITH INLINE FILTER PRES"."PBV-117 MFG TO STORAGE – 3 TRANSFER LINE" )
   END_RUNG wire#w2
   // the same network as SCL:
   "TRANSFER DB".OUTPUT."PBV-117 MFG TO STORAGE – 3 TRANSFER LINE" := "AlwaysTRUE" AND ("MODE SELECTION DB"."MODE BUFF" <> 0) AND ("TRANSFER DB".BIT."MFG TO STORAGE-3 WITH INLINE HOMO"."PBV-117 MFG TO STORAGE – 3 TRANSFER LINE" OR "TRANSFER DB".BIT."MFG TO STORAGE-3 WITH INLINE FILTER PRES"."PBV-117 MFG TO STORAGE – 3 TRANSFER LINE");
END_REGION

REGION Network 90: PBV-118 FILTER PRESS INLET
   RUNG wire#powerrail
      Contact( "AlwaysTRUE" )
      { S7_Templates := "SrcType := Int" } NE_Contact(in1 := "MODE SELECTION DB"."MODE BUFF", in2 := 0)
      wire#w1
      Contact( "TRANSFER DB".BIT."MFG TO STORAGE-1 WITH INLINE FILTER PRES"."PBV-118 FILTER PRESS INLET" )
      wire#w2
      Coil( "TRANSFER DB".OUTPUT."PBV-118 FILTER PRESS INLET" )
   END_RUNG
   RUNG wire#w1
      Contact( "TRANSFER DB".BIT."MFG TO STORAGE-2 WITH INLINE FILTER PRES"."PBV-118 FILTER PRESS INLET" )
   END_RUNG wire#w2
   RUNG wire#w1
      Contact( "TRANSFER DB".BIT."MFG TO STORAGE-3 WITH INLINE FILTER PRES"."PBV-118 FILTER PRESS INLET" )
   END_RUNG wire#w2
   // the same network as SCL:
   "TRANSFER DB".OUTPUT."PBV-118 FILTER PRESS INLET" := "AlwaysTRUE" AND ("MODE SELECTION DB"."MODE BUFF" <> 0) AND ("TRANSFER DB".BIT."MFG TO STORAGE-1 WITH INLINE FILTER PRES"."PBV-118 FILTER PRESS INLET" OR "TRANSFER DB".BIT."MFG TO STORAGE-2 WITH INLINE FILTER PRES"."PBV-118 FILTER PRESS INLET" OR "TRANSFER DB".BIT."MFG TO STORAGE-3 WITH INLINE FILTER PRES"."PBV-118 FILTER PRESS INLET");
END_REGION

REGION Network 91: PBV-119 SEAL COOLING FOR STORAGE VESSEL - 4
   RUNG wire#powerrail
      Contact( "AlwaysFALSE" )
      { S7_Templates := "SrcType := Int" } NE_Contact(in1 := "MODE SELECTION DB"."MODE BUFF", in2 := 0)
      Coil( "TRANSFER DB".OUTPUT."PBV-119 SEAL COOLING FOR STORAGE VESSEL - 4" )
   END_RUNG
   // the same network as SCL:
   "TRANSFER DB".OUTPUT."PBV-119 SEAL COOLING FOR STORAGE VESSEL - 4" := "AlwaysFALSE" AND ("MODE SELECTION DB"."MODE BUFF" <> 0);
END_REGION

REGION Network 92: PBV-120 SEAL COOLING FOR STORAGE VESSEL - 3
   RUNG wire#powerrail
      Contact( "AlwaysFALSE" )
      { S7_Templates := "SrcType := Int" } NE_Contact(in1 := "MODE SELECTION DB"."MODE BUFF", in2 := 0)
      Coil( "TRANSFER DB".OUTPUT."PBV-120 SEAL COOLING FOR STORAGE VESSEL - 3" )
   END_RUNG
   // the same network as SCL:
   "TRANSFER DB".OUTPUT."PBV-120 SEAL COOLING FOR STORAGE VESSEL - 3" := "AlwaysFALSE" AND ("MODE SELECTION DB"."MODE BUFF" <> 0);
END_REGION

REGION Network 93: PBV-121 SEAL COOLING FOR STORAGE VESSEL - 2
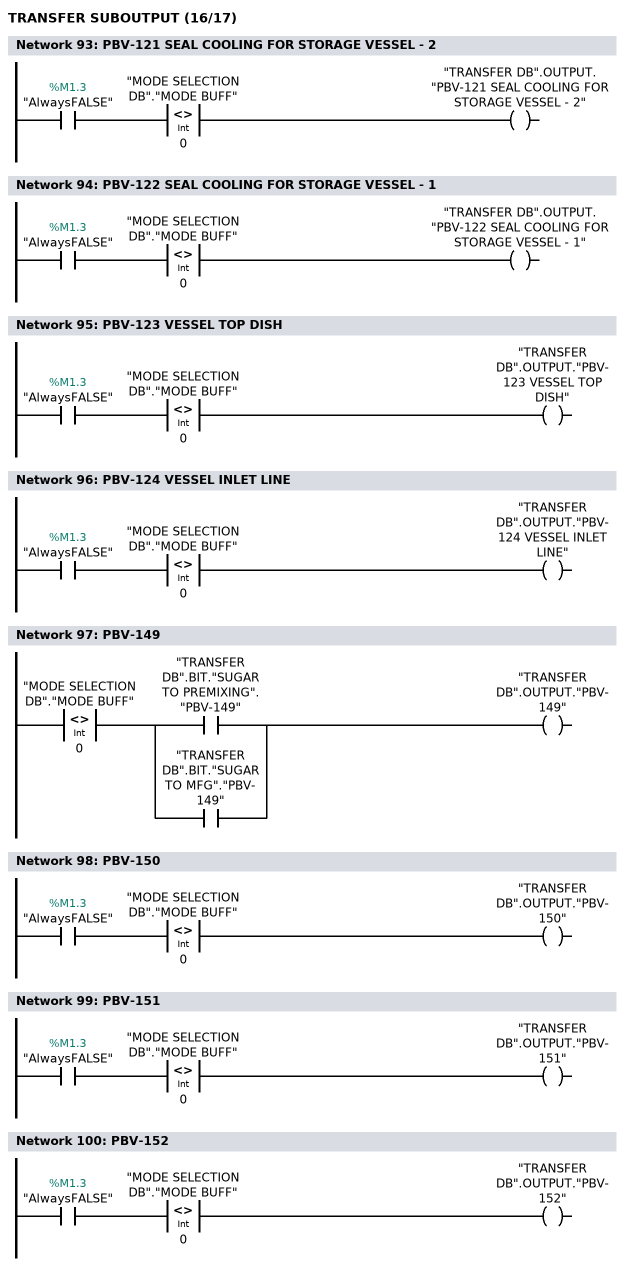
   RUNG wire#powerrail
      Contact( "AlwaysFALSE" )
      { S7_Templates := "SrcType := Int" } NE_Contact(in1 := "MODE SELECTION DB"."MODE BUFF", in2 := 0)
      Coil( "TRANSFER DB".OUTPUT."PBV-121 SEAL COOLING FOR STORAGE VESSEL - 2" )
   END_RUNG
   // the same network as SCL:
   "TRANSFER DB".OUTPUT."PBV-121 SEAL COOLING FOR STORAGE VESSEL - 2" := "AlwaysFALSE" AND ("MODE SELECTION DB"."MODE BUFF" <> 0);
END_REGION

REGION Network 94: PBV-122 SEAL COOLING FOR STORAGE VESSEL - 1
   RUNG wire#powerrail
      Contact( "AlwaysFALSE" )
      { S7_Templates := "SrcType := Int" } NE_Contact(in1 := "MODE SELECTION DB"."MODE BUFF", in2 := 0)
      Coil( "TRANSFER DB".OUTPUT."PBV-122 SEAL COOLING FOR STORAGE VESSEL - 1" )
   END_RUNG
   // the same network as SCL:
   "TRANSFER DB".OUTPUT."PBV-122 SEAL COOLING FOR STORAGE VESSEL - 1" := "AlwaysFALSE" AND ("MODE SELECTION DB"."MODE BUFF" <> 0);
END_REGION

REGION Network 95: PBV-123 VESSEL TOP DISH
   RUNG wire#powerrail
      Contact( "AlwaysFALSE" )
      { S7_Templates := "SrcType := Int" } NE_Contact(in1 := "MODE SELECTION DB"."MODE BUFF", in2 := 0)
      Coil( "TRANSFER DB".OUTPUT."PBV-123 VESSEL TOP DISH" )
   END_RUNG
   // the same network as SCL:
   "TRANSFER DB".OUTPUT."PBV-123 VESSEL TOP DISH" := "AlwaysFALSE" AND ("MODE SELECTION DB"."MODE BUFF" <> 0);
END_REGION

REGION Network 96: PBV-124 VESSEL INLET LINE
   RUNG wire#powerrail
      Contact( "AlwaysFALSE" )
      { S7_Templates := "SrcType := Int" } NE_Contact(in1 := "MODE SELECTION DB"."MODE BUFF", in2 := 0)
      Coil( "TRANSFER DB".OUTPUT."PBV-124 VESSEL INLET LINE" )
   END_RUNG
   // the same network as SCL:
   "TRANSFER DB".OUTPUT."PBV-124 VESSEL INLET LINE" := "AlwaysFALSE" AND ("MODE SELECTION DB"."MODE BUFF" <> 0);
END_REGION

REGION Network 97: PBV-149
   RUNG wire#powerrail
      { S7_Templates := "SrcType := Int" } NE_Contact(in1 := "MODE SELECTION DB"."MODE BUFF", in2 := 0)
      wire#w1
      Contact( "TRANSFER DB".BIT."SUGAR TO PREMIXING"."PBV-149" )
      wire#w2
      Coil( "TRANSFER DB".OUTPUT."PBV-149" )
   END_RUNG
   RUNG wire#w1
      Contact( "TRANSFER DB".BIT."SUGAR TO MFG"."PBV-149" )
   END_RUNG wire#w2
   // the same network as SCL:
   "TRANSFER DB".OUTPUT."PBV-149" := ("MODE SELECTION DB"."MODE BUFF" <> 0) AND ("TRANSFER DB".BIT."SUGAR TO PREMIXING"."PBV-149" OR "TRANSFER DB".BIT."SUGAR TO MFG"."PBV-149");
END_REGION

REGION Network 98: PBV-150
   RUNG wire#powerrail
      Contact( "AlwaysFALSE" )
      { S7_Templates := "SrcType := Int" } NE_Contact(in1 := "MODE SELECTION DB"."MODE BUFF", in2 := 0)
      Coil( "TRANSFER DB".OUTPUT."PBV-150" )
   END_RUNG
   // the same network as SCL:
   "TRANSFER DB".OUTPUT."PBV-150" := "AlwaysFALSE" AND ("MODE SELECTION DB"."MODE BUFF" <> 0);
END_REGION

REGION Network 99: PBV-151
   RUNG wire#powerrail
      Contact( "AlwaysFALSE" )
      { S7_Templates := "SrcType := Int" } NE_Contact(in1 := "MODE SELECTION DB"."MODE BUFF", in2 := 0)
      Coil( "TRANSFER DB".OUTPUT."PBV-151" )
   END_RUNG
   // the same network as SCL:
   "TRANSFER DB".OUTPUT."PBV-151" := "AlwaysFALSE" AND ("MODE SELECTION DB"."MODE BUFF" <> 0);
END_REGION

REGION Network 100: PBV-152
   RUNG wire#powerrail
      Contact( "AlwaysFALSE" )
      { S7_Templates := "SrcType := Int" } NE_Contact(in1 := "MODE SELECTION DB"."MODE BUFF", in2 := 0)
      Coil( "TRANSFER DB".OUTPUT."PBV-152" )
   END_RUNG
   // the same network as SCL:
   "TRANSFER DB".OUTPUT."PBV-152" := "AlwaysFALSE" AND ("MODE SELECTION DB"."MODE BUFF" <> 0);
END_REGION

REGION Network 101: PBV-153
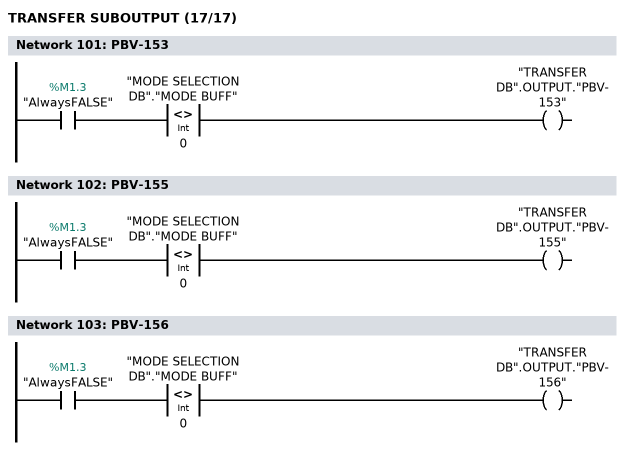
   RUNG wire#powerrail
      Contact( "AlwaysFALSE" )
      { S7_Templates := "SrcType := Int" } NE_Contact(in1 := "MODE SELECTION DB"."MODE BUFF", in2 := 0)
      Coil( "TRANSFER DB".OUTPUT."PBV-153" )
   END_RUNG
   // the same network as SCL:
   "TRANSFER DB".OUTPUT."PBV-153" := "AlwaysFALSE" AND ("MODE SELECTION DB"."MODE BUFF" <> 0);
END_REGION

REGION Network 102: PBV-155
   RUNG wire#powerrail
      Contact( "AlwaysFALSE" )
      { S7_Templates := "SrcType := Int" } NE_Contact(in1 := "MODE SELECTION DB"."MODE BUFF", in2 := 0)
      Coil( "TRANSFER DB".OUTPUT."PBV-155" )
   END_RUNG
   // the same network as SCL:
   "TRANSFER DB".OUTPUT."PBV-155" := "AlwaysFALSE" AND ("MODE SELECTION DB"."MODE BUFF" <> 0);
END_REGION

REGION Network 103: PBV-156
   RUNG wire#powerrail
      Contact( "AlwaysFALSE" )
      { S7_Templates := "SrcType := Int" } NE_Contact(in1 := "MODE SELECTION DB"."MODE BUFF", in2 := 0)
      Coil( "TRANSFER DB".OUTPUT."PBV-156" )
   END_RUNG
   // the same network as SCL:
   "TRANSFER DB".OUTPUT."PBV-156" := "AlwaysFALSE" AND ("MODE SELECTION DB"."MODE BUFF" <> 0);
END_REGION
END_FUNCTION

FUNCTION "AUTO ALARM" : Void   // FC17, LAD
{ S7_Optimized_Access := 'TRUE' }
// stored: SetENOAutomatically false
BEGIN

REGION Network 1: ///////////////////////////////MFG PUPUP/////////////////////////////////////
END_REGION

REGION Network 2: PURIFIED WATER PROCESS SELECT
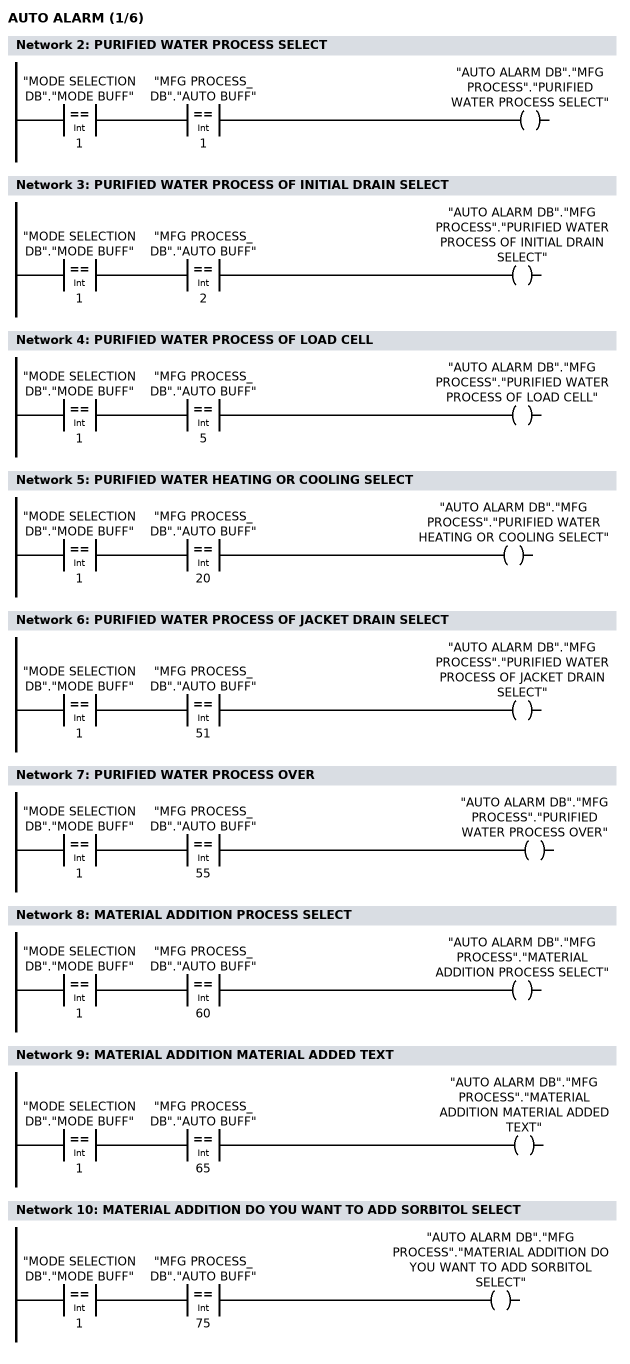
   RUNG wire#powerrail
      { S7_Templates := "SrcType := Int" } EQ_Contact(in1 := "MODE SELECTION DB"."MODE BUFF", in2 := 1)
      { S7_Templates := "SrcType := Int" } EQ_Contact(in1 := "MFG PROCESS_DB"."AUTO BUFF", in2 := 1)
      Coil( "AUTO ALARM DB"."MFG PROCESS"."PURIFIED WATER PROCESS SELECT" )
   END_RUNG
   // the same network as SCL:
   "AUTO ALARM DB"."MFG PROCESS"."PURIFIED WATER PROCESS SELECT" := ("MODE SELECTION DB"."MODE BUFF" = 1) AND ("MFG PROCESS_DB"."AUTO BUFF" = 1);
END_REGION

REGION Network 3: PURIFIED WATER PROCESS OF INITIAL DRAIN SELECT
   RUNG wire#powerrail
      { S7_Templates := "SrcType := Int" } EQ_Contact(in1 := "MODE SELECTION DB"."MODE BUFF", in2 := 1)
      { S7_Templates := "SrcType := Int" } EQ_Contact(in1 := "MFG PROCESS_DB"."AUTO BUFF", in2 := 2)
      Coil( "AUTO ALARM DB"."MFG PROCESS"."PURIFIED WATER PROCESS OF INITIAL DRAIN SELECT" )
   END_RUNG
   // the same network as SCL:
   "AUTO ALARM DB"."MFG PROCESS"."PURIFIED WATER PROCESS OF INITIAL DRAIN SELECT" := ("MODE SELECTION DB"."MODE BUFF" = 1) AND ("MFG PROCESS_DB"."AUTO BUFF" = 2);
END_REGION

REGION Network 4: PURIFIED WATER PROCESS OF LOAD CELL
   RUNG wire#powerrail
      { S7_Templates := "SrcType := Int" } EQ_Contact(in1 := "MODE SELECTION DB"."MODE BUFF", in2 := 1)
      { S7_Templates := "SrcType := Int" } EQ_Contact(in1 := "MFG PROCESS_DB"."AUTO BUFF", in2 := 5)
      Coil( "AUTO ALARM DB"."MFG PROCESS"."PURIFIED WATER PROCESS OF LOAD CELL" )
   END_RUNG
   // the same network as SCL:
   "AUTO ALARM DB"."MFG PROCESS"."PURIFIED WATER PROCESS OF LOAD CELL" := ("MODE SELECTION DB"."MODE BUFF" = 1) AND ("MFG PROCESS_DB"."AUTO BUFF" = 5);
END_REGION

REGION Network 5: PURIFIED WATER HEATING OR COOLING SELECT
   RUNG wire#powerrail
      { S7_Templates := "SrcType := Int" } EQ_Contact(in1 := "MODE SELECTION DB"."MODE BUFF", in2 := 1)
      { S7_Templates := "SrcType := Int" } EQ_Contact(in1 := "MFG PROCESS_DB"."AUTO BUFF", in2 := 20)
      Coil( "AUTO ALARM DB"."MFG PROCESS"."PURIFIED WATER HEATING OR COOLING SELECT" )
   END_RUNG
   // the same network as SCL:
   "AUTO ALARM DB"."MFG PROCESS"."PURIFIED WATER HEATING OR COOLING SELECT" := ("MODE SELECTION DB"."MODE BUFF" = 1) AND ("MFG PROCESS_DB"."AUTO BUFF" = 20);
END_REGION

REGION Network 6: PURIFIED WATER PROCESS OF JACKET DRAIN SELECT
   RUNG wire#powerrail
      { S7_Templates := "SrcType := Int" } EQ_Contact(in1 := "MODE SELECTION DB"."MODE BUFF", in2 := 1)
      { S7_Templates := "SrcType := Int" } EQ_Contact(in1 := "MFG PROCESS_DB"."AUTO BUFF", in2 := 51)
      Coil( "AUTO ALARM DB"."MFG PROCESS"."PURIFIED WATER PROCESS OF JACKET DRAIN SELECT" )
   END_RUNG
   // the same network as SCL:
   "AUTO ALARM DB"."MFG PROCESS"."PURIFIED WATER PROCESS OF JACKET DRAIN SELECT" := ("MODE SELECTION DB"."MODE BUFF" = 1) AND ("MFG PROCESS_DB"."AUTO BUFF" = 51);
END_REGION

REGION Network 7: PURIFIED WATER PROCESS OVER
   RUNG wire#powerrail
      { S7_Templates := "SrcType := Int" } EQ_Contact(in1 := "MODE SELECTION DB"."MODE BUFF", in2 := 1)
      { S7_Templates := "SrcType := Int" } EQ_Contact(in1 := "MFG PROCESS_DB"."AUTO BUFF", in2 := 55)
      Coil( "AUTO ALARM DB"."MFG PROCESS"."PURIFIED WATER PROCESS OVER" )
   END_RUNG
   // the same network as SCL:
   "AUTO ALARM DB"."MFG PROCESS"."PURIFIED WATER PROCESS OVER" := ("MODE SELECTION DB"."MODE BUFF" = 1) AND ("MFG PROCESS_DB"."AUTO BUFF" = 55);
END_REGION

REGION Network 8: MATERIAL ADDITION PROCESS SELECT
   RUNG wire#powerrail
      { S7_Templates := "SrcType := Int" } EQ_Contact(in1 := "MODE SELECTION DB"."MODE BUFF", in2 := 1)
      { S7_Templates := "SrcType := Int" } EQ_Contact(in1 := "MFG PROCESS_DB"."AUTO BUFF", in2 := 60)
      Coil( "AUTO ALARM DB"."MFG PROCESS"."MATERIAL ADDITION PROCESS SELECT" )
   END_RUNG
   // the same network as SCL:
   "AUTO ALARM DB"."MFG PROCESS"."MATERIAL ADDITION PROCESS SELECT" := ("MODE SELECTION DB"."MODE BUFF" = 1) AND ("MFG PROCESS_DB"."AUTO BUFF" = 60);
END_REGION

REGION Network 9: MATERIAL ADDITION MATERIAL ADDED TEXT
   RUNG wire#powerrail
      { S7_Templates := "SrcType := Int" } EQ_Contact(in1 := "MODE SELECTION DB"."MODE BUFF", in2 := 1)
      { S7_Templates := "SrcType := Int" } EQ_Contact(in1 := "MFG PROCESS_DB"."AUTO BUFF", in2 := 65)
      Coil( "AUTO ALARM DB"."MFG PROCESS"."MATERIAL ADDITION MATERIAL ADDED TEXT" )
   END_RUNG
   // the same network as SCL:
   "AUTO ALARM DB"."MFG PROCESS"."MATERIAL ADDITION MATERIAL ADDED TEXT" := ("MODE SELECTION DB"."MODE BUFF" = 1) AND ("MFG PROCESS_DB"."AUTO BUFF" = 65);
END_REGION

REGION Network 10: MATERIAL ADDITION DO YOU WANT TO ADD SORBITOL SELECT
   RUNG wire#powerrail
      { S7_Templates := "SrcType := Int" } EQ_Contact(in1 := "MODE SELECTION DB"."MODE BUFF", in2 := 1)
      { S7_Templates := "SrcType := Int" } EQ_Contact(in1 := "MFG PROCESS_DB"."AUTO BUFF", in2 := 75)
      Coil( "AUTO ALARM DB"."MFG PROCESS"."MATERIAL ADDITION DO YOU WANT TO ADD SORBITOL SELECT" )
   END_RUNG
   // the same network as SCL:
   "AUTO ALARM DB"."MFG PROCESS"."MATERIAL ADDITION DO YOU WANT TO ADD SORBITOL SELECT" := ("MODE SELECTION DB"."MODE BUFF" = 1) AND ("MFG PROCESS_DB"."AUTO BUFF" = 75);
END_REGION

REGION Network 11: MATERIAL ADDITION OF SORBITOL OVER
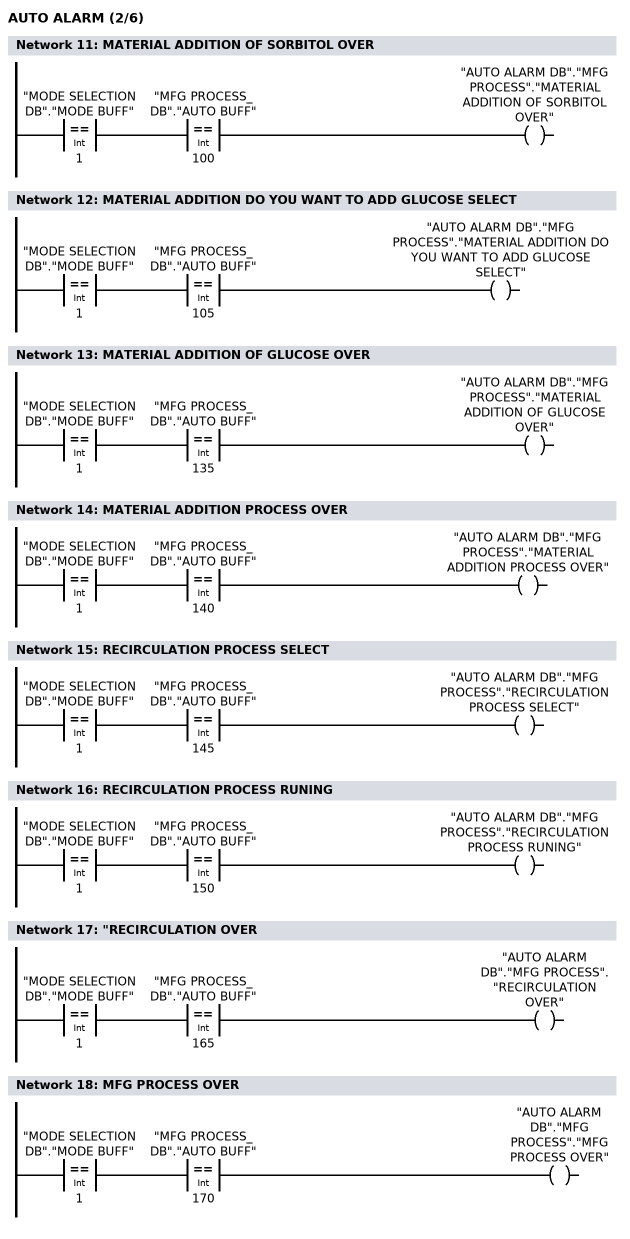
   RUNG wire#powerrail
      { S7_Templates := "SrcType := Int" } EQ_Contact(in1 := "MODE SELECTION DB"."MODE BUFF", in2 := 1)
      { S7_Templates := "SrcType := Int" } EQ_Contact(in1 := "MFG PROCESS_DB"."AUTO BUFF", in2 := 100)
      Coil( "AUTO ALARM DB"."MFG PROCESS"."MATERIAL ADDITION OF SORBITOL OVER" )
   END_RUNG
   // the same network as SCL:
   "AUTO ALARM DB"."MFG PROCESS"."MATERIAL ADDITION OF SORBITOL OVER" := ("MODE SELECTION DB"."MODE BUFF" = 1) AND ("MFG PROCESS_DB"."AUTO BUFF" = 100);
END_REGION

REGION Network 12: MATERIAL ADDITION DO YOU WANT TO ADD GLUCOSE SELECT
   RUNG wire#powerrail
      { S7_Templates := "SrcType := Int" } EQ_Contact(in1 := "MODE SELECTION DB"."MODE BUFF", in2 := 1)
      { S7_Templates := "SrcType := Int" } EQ_Contact(in1 := "MFG PROCESS_DB"."AUTO BUFF", in2 := 105)
      Coil( "AUTO ALARM DB"."MFG PROCESS"."MATERIAL ADDITION DO YOU WANT TO ADD GLUCOSE SELECT" )
   END_RUNG
   // the same network as SCL:
   "AUTO ALARM DB"."MFG PROCESS"."MATERIAL ADDITION DO YOU WANT TO ADD GLUCOSE SELECT" := ("MODE SELECTION DB"."MODE BUFF" = 1) AND ("MFG PROCESS_DB"."AUTO BUFF" = 105);
END_REGION

REGION Network 13: MATERIAL ADDITION OF GLUCOSE OVER
   RUNG wire#powerrail
      { S7_Templates := "SrcType := Int" } EQ_Contact(in1 := "MODE SELECTION DB"."MODE BUFF", in2 := 1)
      { S7_Templates := "SrcType := Int" } EQ_Contact(in1 := "MFG PROCESS_DB"."AUTO BUFF", in2 := 135)
      Coil( "AUTO ALARM DB"."MFG PROCESS"."MATERIAL ADDITION OF GLUCOSE OVER" )
   END_RUNG
   // the same network as SCL:
   "AUTO ALARM DB"."MFG PROCESS"."MATERIAL ADDITION OF GLUCOSE OVER" := ("MODE SELECTION DB"."MODE BUFF" = 1) AND ("MFG PROCESS_DB"."AUTO BUFF" = 135);
END_REGION

REGION Network 14: MATERIAL ADDITION PROCESS OVER
   RUNG wire#powerrail
      { S7_Templates := "SrcType := Int" } EQ_Contact(in1 := "MODE SELECTION DB"."MODE BUFF", in2 := 1)
      { S7_Templates := "SrcType := Int" } EQ_Contact(in1 := "MFG PROCESS_DB"."AUTO BUFF", in2 := 140)
      Coil( "AUTO ALARM DB"."MFG PROCESS"."MATERIAL ADDITION PROCESS OVER" )
   END_RUNG
   // the same network as SCL:
   "AUTO ALARM DB"."MFG PROCESS"."MATERIAL ADDITION PROCESS OVER" := ("MODE SELECTION DB"."MODE BUFF" = 1) AND ("MFG PROCESS_DB"."AUTO BUFF" = 140);
END_REGION

REGION Network 15: RECIRCULATION PROCESS SELECT
   RUNG wire#powerrail
      { S7_Templates := "SrcType := Int" } EQ_Contact(in1 := "MODE SELECTION DB"."MODE BUFF", in2 := 1)
      { S7_Templates := "SrcType := Int" } EQ_Contact(in1 := "MFG PROCESS_DB"."AUTO BUFF", in2 := 145)
      Coil( "AUTO ALARM DB"."MFG PROCESS"."RECIRCULATION PROCESS SELECT" )
   END_RUNG
   // the same network as SCL:
   "AUTO ALARM DB"."MFG PROCESS"."RECIRCULATION PROCESS SELECT" := ("MODE SELECTION DB"."MODE BUFF" = 1) AND ("MFG PROCESS_DB"."AUTO BUFF" = 145);
END_REGION

REGION Network 16: RECIRCULATION PROCESS RUNING
   RUNG wire#powerrail
      { S7_Templates := "SrcType := Int" } EQ_Contact(in1 := "MODE SELECTION DB"."MODE BUFF", in2 := 1)
      { S7_Templates := "SrcType := Int" } EQ_Contact(in1 := "MFG PROCESS_DB"."AUTO BUFF", in2 := 150)
      Coil( "AUTO ALARM DB"."MFG PROCESS"."RECIRCULATION PROCESS RUNING" )
   END_RUNG
   // the same network as SCL:
   "AUTO ALARM DB"."MFG PROCESS"."RECIRCULATION PROCESS RUNING" := ("MODE SELECTION DB"."MODE BUFF" = 1) AND ("MFG PROCESS_DB"."AUTO BUFF" = 150);
END_REGION

REGION Network 17: "RECIRCULATION OVER
   RUNG wire#powerrail
      { S7_Templates := "SrcType := Int" } EQ_Contact(in1 := "MODE SELECTION DB"."MODE BUFF", in2 := 1)
      { S7_Templates := "SrcType := Int" } EQ_Contact(in1 := "MFG PROCESS_DB"."AUTO BUFF", in2 := 165)
      Coil( "AUTO ALARM DB"."MFG PROCESS"."RECIRCULATION OVER" )
   END_RUNG
   // the same network as SCL:
   "AUTO ALARM DB"."MFG PROCESS"."RECIRCULATION OVER" := ("MODE SELECTION DB"."MODE BUFF" = 1) AND ("MFG PROCESS_DB"."AUTO BUFF" = 165);
END_REGION

REGION Network 18: MFG PROCESS OVER
   RUNG wire#powerrail
      { S7_Templates := "SrcType := Int" } EQ_Contact(in1 := "MODE SELECTION DB"."MODE BUFF", in2 := 1)
      { S7_Templates := "SrcType := Int" } EQ_Contact(in1 := "MFG PROCESS_DB"."AUTO BUFF", in2 := 170)
      Coil( "AUTO ALARM DB"."MFG PROCESS"."MFG PROCESS OVER" )
   END_RUNG
   // the same network as SCL:
   "AUTO ALARM DB"."MFG PROCESS"."MFG PROCESS OVER" := ("MODE SELECTION DB"."MODE BUFF" = 1) AND ("MFG PROCESS_DB"."AUTO BUFF" = 170);
END_REGION

REGION Network 20: TRANSFER START_MFG TO STORAGE-1 WITH INLINE HOMO
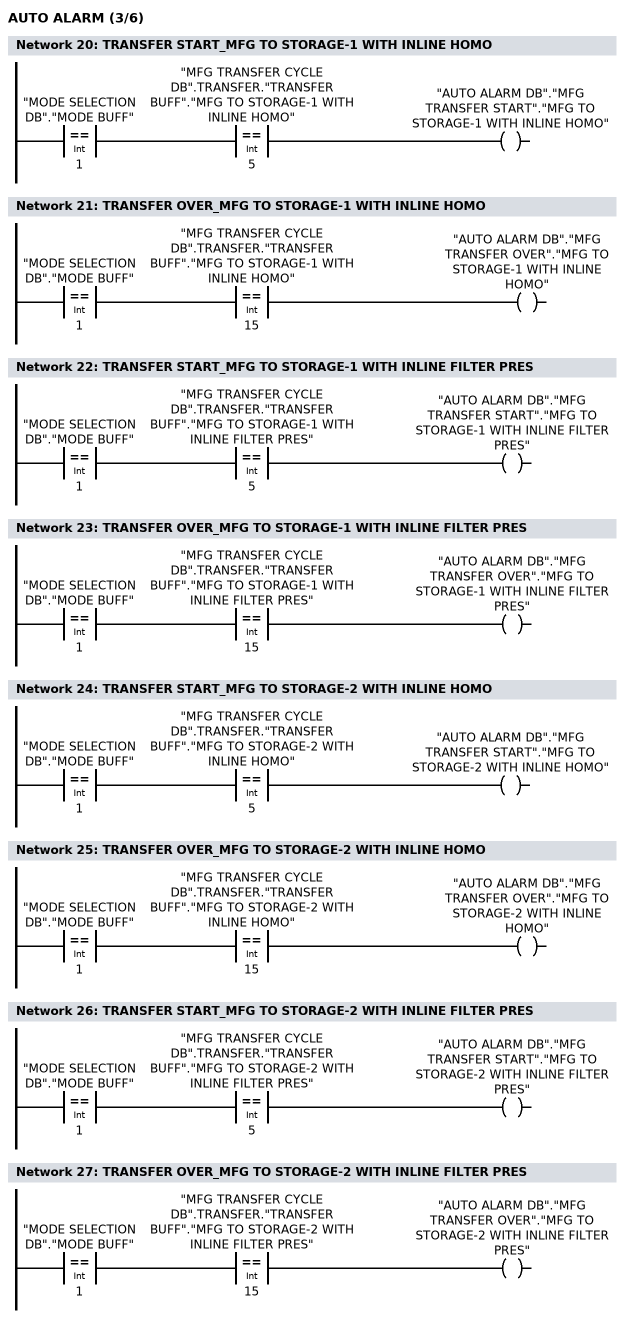
   RUNG wire#powerrail
      { S7_Templates := "SrcType := Int" } EQ_Contact(in1 := "MODE SELECTION DB"."MODE BUFF", in2 := 1)
      { S7_Templates := "SrcType := Int" } EQ_Contact(in1 := "MFG TRANSFER CYCLE DB".TRANSFER."TRANSFER BUFF"."MFG TO STORAGE-1 WITH INLINE HOMO", in2 := 5)
      Coil( "AUTO ALARM DB"."MFG TRANSFER START"."MFG TO STORAGE-1 WITH INLINE HOMO" )
   END_RUNG
   // the same network as SCL:
   "AUTO ALARM DB"."MFG TRANSFER START"."MFG TO STORAGE-1 WITH INLINE HOMO" := ("MODE SELECTION DB"."MODE BUFF" = 1) AND ("MFG TRANSFER CYCLE DB".TRANSFER."TRANSFER BUFF"."MFG TO STORAGE-1 WITH INLINE HOMO" = 5);
END_REGION

REGION Network 21: TRANSFER OVER_MFG TO STORAGE-1 WITH INLINE HOMO
   RUNG wire#powerrail
      { S7_Templates := "SrcType := Int" } EQ_Contact(in1 := "MODE SELECTION DB"."MODE BUFF", in2 := 1)
      { S7_Templates := "SrcType := Int" } EQ_Contact(in1 := "MFG TRANSFER CYCLE DB".TRANSFER."TRANSFER BUFF"."MFG TO STORAGE-1 WITH INLINE HOMO", in2 := 15)
      Coil( "AUTO ALARM DB"."MFG TRANSFER OVER"."MFG TO STORAGE-1 WITH INLINE HOMO" )
   END_RUNG
   // the same network as SCL:
   "AUTO ALARM DB"."MFG TRANSFER OVER"."MFG TO STORAGE-1 WITH INLINE HOMO" := ("MODE SELECTION DB"."MODE BUFF" = 1) AND ("MFG TRANSFER CYCLE DB".TRANSFER."TRANSFER BUFF"."MFG TO STORAGE-1 WITH INLINE HOMO" = 15);
END_REGION

REGION Network 22: TRANSFER START_MFG TO STORAGE-1 WITH INLINE FILTER PRES
   RUNG wire#powerrail
      { S7_Templates := "SrcType := Int" } EQ_Contact(in1 := "MODE SELECTION DB"."MODE BUFF", in2 := 1)
      { S7_Templates := "SrcType := Int" } EQ_Contact(in1 := "MFG TRANSFER CYCLE DB".TRANSFER."TRANSFER BUFF"."MFG TO STORAGE-1 WITH INLINE FILTER PRES", in2 := 5)
      Coil( "AUTO ALARM DB"."MFG TRANSFER START"."MFG TO STORAGE-1 WITH INLINE FILTER PRES" )
   END_RUNG
   // the same network as SCL:
   "AUTO ALARM DB"."MFG TRANSFER START"."MFG TO STORAGE-1 WITH INLINE FILTER PRES" := ("MODE SELECTION DB"."MODE BUFF" = 1) AND ("MFG TRANSFER CYCLE DB".TRANSFER."TRANSFER BUFF"."MFG TO STORAGE-1 WITH INLINE FILTER PRES" = 5);
END_REGION

REGION Network 23: TRANSFER OVER_MFG TO STORAGE-1 WITH INLINE FILTER PRES
   RUNG wire#powerrail
      { S7_Templates := "SrcType := Int" } EQ_Contact(in1 := "MODE SELECTION DB"."MODE BUFF", in2 := 1)
      { S7_Templates := "SrcType := Int" } EQ_Contact(in1 := "MFG TRANSFER CYCLE DB".TRANSFER."TRANSFER BUFF"."MFG TO STORAGE-1 WITH INLINE FILTER PRES", in2 := 15)
      Coil( "AUTO ALARM DB"."MFG TRANSFER OVER"."MFG TO STORAGE-1 WITH INLINE FILTER PRES" )
   END_RUNG
   // the same network as SCL:
   "AUTO ALARM DB"."MFG TRANSFER OVER"."MFG TO STORAGE-1 WITH INLINE FILTER PRES" := ("MODE SELECTION DB"."MODE BUFF" = 1) AND ("MFG TRANSFER CYCLE DB".TRANSFER."TRANSFER BUFF"."MFG TO STORAGE-1 WITH INLINE FILTER PRES" = 15);
END_REGION

REGION Network 24: TRANSFER START_MFG TO STORAGE-2 WITH INLINE HOMO
   RUNG wire#powerrail
      { S7_Templates := "SrcType := Int" } EQ_Contact(in1 := "MODE SELECTION DB"."MODE BUFF", in2 := 1)
      { S7_Templates := "SrcType := Int" } EQ_Contact(in1 := "MFG TRANSFER CYCLE DB".TRANSFER."TRANSFER BUFF"."MFG TO STORAGE-2 WITH INLINE HOMO", in2 := 5)
      Coil( "AUTO ALARM DB"."MFG TRANSFER START"."MFG TO STORAGE-2 WITH INLINE HOMO" )
   END_RUNG
   // the same network as SCL:
   "AUTO ALARM DB"."MFG TRANSFER START"."MFG TO STORAGE-2 WITH INLINE HOMO" := ("MODE SELECTION DB"."MODE BUFF" = 1) AND ("MFG TRANSFER CYCLE DB".TRANSFER."TRANSFER BUFF"."MFG TO STORAGE-2 WITH INLINE HOMO" = 5);
END_REGION

REGION Network 25: TRANSFER OVER_MFG TO STORAGE-2 WITH INLINE HOMO
   RUNG wire#powerrail
      { S7_Templates := "SrcType := Int" } EQ_Contact(in1 := "MODE SELECTION DB"."MODE BUFF", in2 := 1)
      { S7_Templates := "SrcType := Int" } EQ_Contact(in1 := "MFG TRANSFER CYCLE DB".TRANSFER."TRANSFER BUFF"."MFG TO STORAGE-2 WITH INLINE HOMO", in2 := 15)
      Coil( "AUTO ALARM DB"."MFG TRANSFER OVER"."MFG TO STORAGE-2 WITH INLINE HOMO" )
   END_RUNG
   // the same network as SCL:
   "AUTO ALARM DB"."MFG TRANSFER OVER"."MFG TO STORAGE-2 WITH INLINE HOMO" := ("MODE SELECTION DB"."MODE BUFF" = 1) AND ("MFG TRANSFER CYCLE DB".TRANSFER."TRANSFER BUFF"."MFG TO STORAGE-2 WITH INLINE HOMO" = 15);
END_REGION

REGION Network 26: TRANSFER START_MFG TO STORAGE-2 WITH INLINE FILTER PRES
   RUNG wire#powerrail
      { S7_Templates := "SrcType := Int" } EQ_Contact(in1 := "MODE SELECTION DB"."MODE BUFF", in2 := 1)
      { S7_Templates := "SrcType := Int" } EQ_Contact(in1 := "MFG TRANSFER CYCLE DB".TRANSFER."TRANSFER BUFF"."MFG TO STORAGE-2 WITH INLINE FILTER PRES", in2 := 5)
      Coil( "AUTO ALARM DB"."MFG TRANSFER START"."MFG TO STORAGE-2 WITH INLINE FILTER PRES" )
   END_RUNG
   // the same network as SCL:
   "AUTO ALARM DB"."MFG TRANSFER START"."MFG TO STORAGE-2 WITH INLINE FILTER PRES" := ("MODE SELECTION DB"."MODE BUFF" = 1) AND ("MFG TRANSFER CYCLE DB".TRANSFER."TRANSFER BUFF"."MFG TO STORAGE-2 WITH INLINE FILTER PRES" = 5);
END_REGION

REGION Network 27: TRANSFER OVER_MFG TO STORAGE-2 WITH INLINE FILTER PRES
   RUNG wire#powerrail
      { S7_Templates := "SrcType := Int" } EQ_Contact(in1 := "MODE SELECTION DB"."MODE BUFF", in2 := 1)
      { S7_Templates := "SrcType := Int" } EQ_Contact(in1 := "MFG TRANSFER CYCLE DB".TRANSFER."TRANSFER BUFF"."MFG TO STORAGE-2 WITH INLINE FILTER PRES", in2 := 15)
      Coil( "AUTO ALARM DB"."MFG TRANSFER OVER"."MFG TO STORAGE-2 WITH INLINE FILTER PRES" )
   END_RUNG
   // the same network as SCL:
   "AUTO ALARM DB"."MFG TRANSFER OVER"."MFG TO STORAGE-2 WITH INLINE FILTER PRES" := ("MODE SELECTION DB"."MODE BUFF" = 1) AND ("MFG TRANSFER CYCLE DB".TRANSFER."TRANSFER BUFF"."MFG TO STORAGE-2 WITH INLINE FILTER PRES" = 15);
END_REGION

REGION Network 28: TRANSFER START_MFG TO STORAGE-3 WITH INLINE HOMO
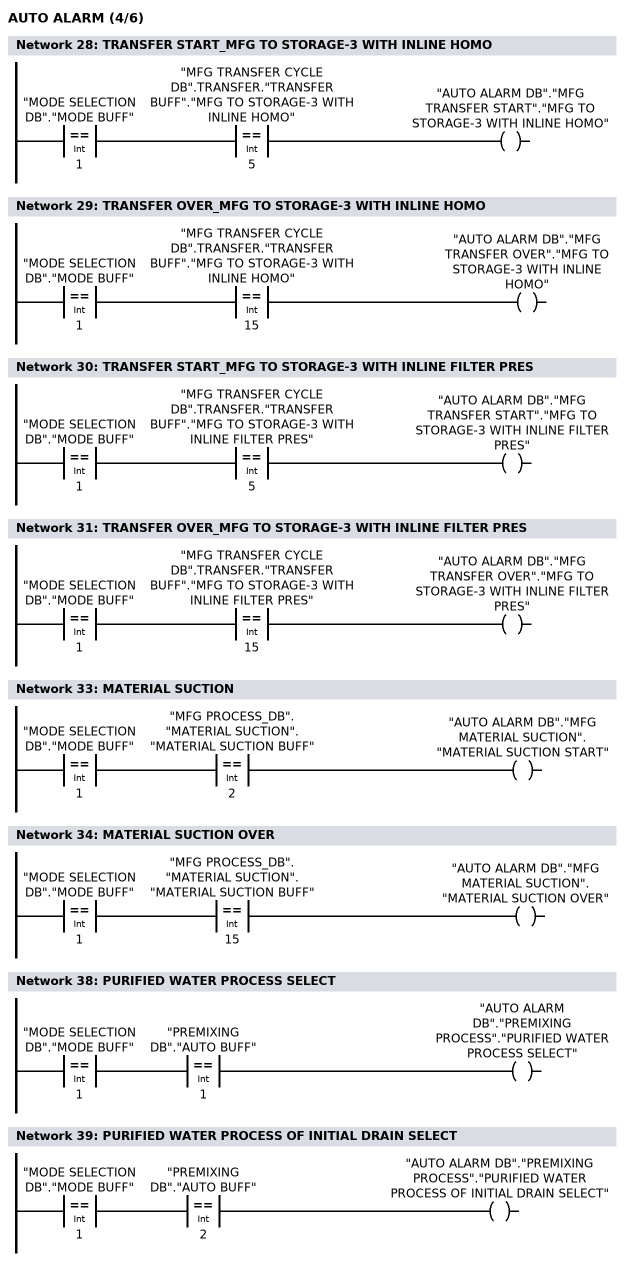
   RUNG wire#powerrail
      { S7_Templates := "SrcType := Int" } EQ_Contact(in1 := "MODE SELECTION DB"."MODE BUFF", in2 := 1)
      { S7_Templates := "SrcType := Int" } EQ_Contact(in1 := "MFG TRANSFER CYCLE DB".TRANSFER."TRANSFER BUFF"."MFG TO STORAGE-3 WITH INLINE HOMO", in2 := 5)
      Coil( "AUTO ALARM DB"."MFG TRANSFER START"."MFG TO STORAGE-3 WITH INLINE HOMO" )
   END_RUNG
   // the same network as SCL:
   "AUTO ALARM DB"."MFG TRANSFER START"."MFG TO STORAGE-3 WITH INLINE HOMO" := ("MODE SELECTION DB"."MODE BUFF" = 1) AND ("MFG TRANSFER CYCLE DB".TRANSFER."TRANSFER BUFF"."MFG TO STORAGE-3 WITH INLINE HOMO" = 5);
END_REGION

REGION Network 29: TRANSFER OVER_MFG TO STORAGE-3 WITH INLINE HOMO
   RUNG wire#powerrail
      { S7_Templates := "SrcType := Int" } EQ_Contact(in1 := "MODE SELECTION DB"."MODE BUFF", in2 := 1)
      { S7_Templates := "SrcType := Int" } EQ_Contact(in1 := "MFG TRANSFER CYCLE DB".TRANSFER."TRANSFER BUFF"."MFG TO STORAGE-3 WITH INLINE HOMO", in2 := 15)
      Coil( "AUTO ALARM DB"."MFG TRANSFER OVER"."MFG TO STORAGE-3 WITH INLINE HOMO" )
   END_RUNG
   // the same network as SCL:
   "AUTO ALARM DB"."MFG TRANSFER OVER"."MFG TO STORAGE-3 WITH INLINE HOMO" := ("MODE SELECTION DB"."MODE BUFF" = 1) AND ("MFG TRANSFER CYCLE DB".TRANSFER."TRANSFER BUFF"."MFG TO STORAGE-3 WITH INLINE HOMO" = 15);
END_REGION

REGION Network 30: TRANSFER START_MFG TO STORAGE-3 WITH INLINE FILTER PRES
   RUNG wire#powerrail
      { S7_Templates := "SrcType := Int" } EQ_Contact(in1 := "MODE SELECTION DB"."MODE BUFF", in2 := 1)
      { S7_Templates := "SrcType := Int" } EQ_Contact(in1 := "MFG TRANSFER CYCLE DB".TRANSFER."TRANSFER BUFF"."MFG TO STORAGE-3 WITH INLINE FILTER PRES", in2 := 5)
      Coil( "AUTO ALARM DB"."MFG TRANSFER START"."MFG TO STORAGE-3 WITH INLINE FILTER PRES" )
   END_RUNG
   // the same network as SCL:
   "AUTO ALARM DB"."MFG TRANSFER START"."MFG TO STORAGE-3 WITH INLINE FILTER PRES" := ("MODE SELECTION DB"."MODE BUFF" = 1) AND ("MFG TRANSFER CYCLE DB".TRANSFER."TRANSFER BUFF"."MFG TO STORAGE-3 WITH INLINE FILTER PRES" = 5);
END_REGION

REGION Network 31: TRANSFER OVER_MFG TO STORAGE-3 WITH INLINE FILTER PRES
   RUNG wire#powerrail
      { S7_Templates := "SrcType := Int" } EQ_Contact(in1 := "MODE SELECTION DB"."MODE BUFF", in2 := 1)
      { S7_Templates := "SrcType := Int" } EQ_Contact(in1 := "MFG TRANSFER CYCLE DB".TRANSFER."TRANSFER BUFF"."MFG TO STORAGE-3 WITH INLINE FILTER PRES", in2 := 15)
      Coil( "AUTO ALARM DB"."MFG TRANSFER OVER"."MFG TO STORAGE-3 WITH INLINE FILTER PRES" )
   END_RUNG
   // the same network as SCL:
   "AUTO ALARM DB"."MFG TRANSFER OVER"."MFG TO STORAGE-3 WITH INLINE FILTER PRES" := ("MODE SELECTION DB"."MODE BUFF" = 1) AND ("MFG TRANSFER CYCLE DB".TRANSFER."TRANSFER BUFF"."MFG TO STORAGE-3 WITH INLINE FILTER PRES" = 15);
END_REGION

REGION Network 33: MATERIAL SUCTION
   RUNG wire#powerrail
      { S7_Templates := "SrcType := Int" } EQ_Contact(in1 := "MODE SELECTION DB"."MODE BUFF", in2 := 1)
      { S7_Templates := "SrcType := Int" } EQ_Contact(in1 := "MFG PROCESS_DB"."MATERIAL SUCTION"."MATERIAL SUCTION BUFF", in2 := 2)
      Coil( "AUTO ALARM DB"."MFG MATERIAL SUCTION"."MATERIAL SUCTION START" )
   END_RUNG
   // the same network as SCL:
   "AUTO ALARM DB"."MFG MATERIAL SUCTION"."MATERIAL SUCTION START" := ("MODE SELECTION DB"."MODE BUFF" = 1) AND ("MFG PROCESS_DB"."MATERIAL SUCTION"."MATERIAL SUCTION BUFF" = 2);
END_REGION

REGION Network 34: MATERIAL SUCTION OVER
   RUNG wire#powerrail
      { S7_Templates := "SrcType := Int" } EQ_Contact(in1 := "MODE SELECTION DB"."MODE BUFF", in2 := 1)
      { S7_Templates := "SrcType := Int" } EQ_Contact(in1 := "MFG PROCESS_DB"."MATERIAL SUCTION"."MATERIAL SUCTION BUFF", in2 := 15)
      Coil( "AUTO ALARM DB"."MFG MATERIAL SUCTION"."MATERIAL SUCTION OVER" )
   END_RUNG
   // the same network as SCL:
   "AUTO ALARM DB"."MFG MATERIAL SUCTION"."MATERIAL SUCTION OVER" := ("MODE SELECTION DB"."MODE BUFF" = 1) AND ("MFG PROCESS_DB"."MATERIAL SUCTION"."MATERIAL SUCTION BUFF" = 15);
END_REGION

REGION Network 37: /////////////////////////////// PREMIXING PUPUP /////////////////////////////////////
END_REGION

REGION Network 38: PURIFIED WATER PROCESS SELECT
   RUNG wire#powerrail
      { S7_Templates := "SrcType := Int" } EQ_Contact(in1 := "MODE SELECTION DB"."MODE BUFF", in2 := 1)
      { S7_Templates := "SrcType := Int" } EQ_Contact(in1 := "PREMIXING DB"."AUTO BUFF", in2 := 1)
      Coil( "AUTO ALARM DB"."PREMIXING PROCESS"."PURIFIED WATER PROCESS SELECT" )
   END_RUNG
   // the same network as SCL:
   "AUTO ALARM DB"."PREMIXING PROCESS"."PURIFIED WATER PROCESS SELECT" := ("MODE SELECTION DB"."MODE BUFF" = 1) AND ("PREMIXING DB"."AUTO BUFF" = 1);
END_REGION

REGION Network 39: PURIFIED WATER PROCESS OF INITIAL DRAIN SELECT
   RUNG wire#powerrail
      { S7_Templates := "SrcType := Int" } EQ_Contact(in1 := "MODE SELECTION DB"."MODE BUFF", in2 := 1)
      { S7_Templates := "SrcType := Int" } EQ_Contact(in1 := "PREMIXING DB"."AUTO BUFF", in2 := 2)
      Coil( "AUTO ALARM DB"."PREMIXING PROCESS"."PURIFIED WATER PROCESS OF INITIAL DRAIN SELECT" )
   END_RUNG
   // the same network as SCL:
   "AUTO ALARM DB"."PREMIXING PROCESS"."PURIFIED WATER PROCESS OF INITIAL DRAIN SELECT" := ("MODE SELECTION DB"."MODE BUFF" = 1) AND ("PREMIXING DB"."AUTO BUFF" = 2);
END_REGION

REGION Network 40: PURIFIED WATER PROCESS OF LOAD CELL
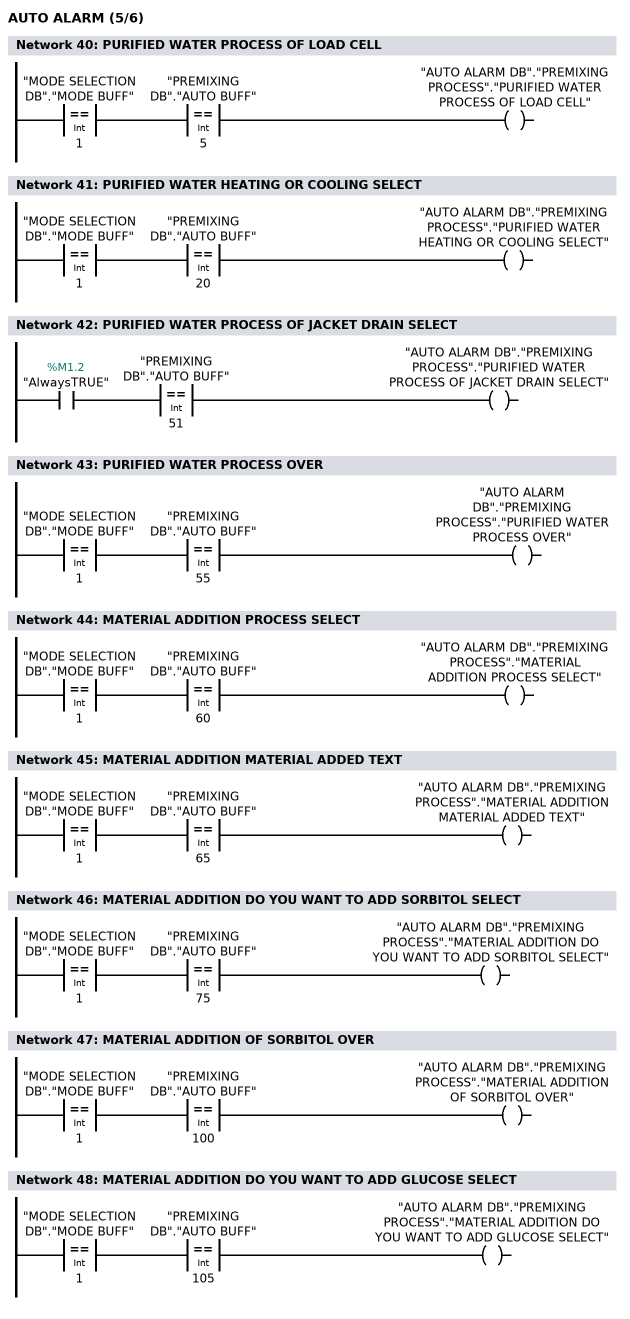
   RUNG wire#powerrail
      { S7_Templates := "SrcType := Int" } EQ_Contact(in1 := "MODE SELECTION DB"."MODE BUFF", in2 := 1)
      { S7_Templates := "SrcType := Int" } EQ_Contact(in1 := "PREMIXING DB"."AUTO BUFF", in2 := 5)
      Coil( "AUTO ALARM DB"."PREMIXING PROCESS"."PURIFIED WATER PROCESS OF LOAD CELL" )
   END_RUNG
   // the same network as SCL:
   "AUTO ALARM DB"."PREMIXING PROCESS"."PURIFIED WATER PROCESS OF LOAD CELL" := ("MODE SELECTION DB"."MODE BUFF" = 1) AND ("PREMIXING DB"."AUTO BUFF" = 5);
END_REGION

REGION Network 41: PURIFIED WATER HEATING OR COOLING SELECT
   RUNG wire#powerrail
      { S7_Templates := "SrcType := Int" } EQ_Contact(in1 := "MODE SELECTION DB"."MODE BUFF", in2 := 1)
      { S7_Templates := "SrcType := Int" } EQ_Contact(in1 := "PREMIXING DB"."AUTO BUFF", in2 := 20)
      Coil( "AUTO ALARM DB"."PREMIXING PROCESS"."PURIFIED WATER HEATING OR COOLING SELECT" )
   END_RUNG
   // the same network as SCL:
   "AUTO ALARM DB"."PREMIXING PROCESS"."PURIFIED WATER HEATING OR COOLING SELECT" := ("MODE SELECTION DB"."MODE BUFF" = 1) AND ("PREMIXING DB"."AUTO BUFF" = 20);
END_REGION

REGION Network 42: PURIFIED WATER PROCESS OF JACKET DRAIN SELECT
   RUNG wire#powerrail
      Contact( "AlwaysTRUE" )
      { S7_Templates := "SrcType := Int" } EQ_Contact(in1 := "PREMIXING DB"."AUTO BUFF", in2 := 51)
      Coil( "AUTO ALARM DB"."PREMIXING PROCESS"."PURIFIED WATER PROCESS OF JACKET DRAIN SELECT" )
   END_RUNG
   // the same network as SCL:
   "AUTO ALARM DB"."PREMIXING PROCESS"."PURIFIED WATER PROCESS OF JACKET DRAIN SELECT" := "AlwaysTRUE" AND ("PREMIXING DB"."AUTO BUFF" = 51);
END_REGION

REGION Network 43: PURIFIED WATER PROCESS OVER
   RUNG wire#powerrail
      { S7_Templates := "SrcType := Int" } EQ_Contact(in1 := "MODE SELECTION DB"."MODE BUFF", in2 := 1)
      { S7_Templates := "SrcType := Int" } EQ_Contact(in1 := "PREMIXING DB"."AUTO BUFF", in2 := 55)
      Coil( "AUTO ALARM DB"."PREMIXING PROCESS"."PURIFIED WATER PROCESS OVER" )
   END_RUNG
   // the same network as SCL:
   "AUTO ALARM DB"."PREMIXING PROCESS"."PURIFIED WATER PROCESS OVER" := ("MODE SELECTION DB"."MODE BUFF" = 1) AND ("PREMIXING DB"."AUTO BUFF" = 55);
END_REGION

REGION Network 44: MATERIAL ADDITION PROCESS SELECT
   RUNG wire#powerrail
      { S7_Templates := "SrcType := Int" } EQ_Contact(in1 := "MODE SELECTION DB"."MODE BUFF", in2 := 1)
      { S7_Templates := "SrcType := Int" } EQ_Contact(in1 := "PREMIXING DB"."AUTO BUFF", in2 := 60)
      Coil( "AUTO ALARM DB"."PREMIXING PROCESS"."MATERIAL ADDITION PROCESS SELECT" )
   END_RUNG
   // the same network as SCL:
   "AUTO ALARM DB"."PREMIXING PROCESS"."MATERIAL ADDITION PROCESS SELECT" := ("MODE SELECTION DB"."MODE BUFF" = 1) AND ("PREMIXING DB"."AUTO BUFF" = 60);
END_REGION

REGION Network 45: MATERIAL ADDITION MATERIAL ADDED TEXT
   RUNG wire#powerrail
      { S7_Templates := "SrcType := Int" } EQ_Contact(in1 := "MODE SELECTION DB"."MODE BUFF", in2 := 1)
      { S7_Templates := "SrcType := Int" } EQ_Contact(in1 := "PREMIXING DB"."AUTO BUFF", in2 := 65)
      Coil( "AUTO ALARM DB"."PREMIXING PROCESS"."MATERIAL ADDITION MATERIAL ADDED TEXT" )
   END_RUNG
   // the same network as SCL:
   "AUTO ALARM DB"."PREMIXING PROCESS"."MATERIAL ADDITION MATERIAL ADDED TEXT" := ("MODE SELECTION DB"."MODE BUFF" = 1) AND ("PREMIXING DB"."AUTO BUFF" = 65);
END_REGION

REGION Network 46: MATERIAL ADDITION DO YOU WANT TO ADD SORBITOL SELECT
   RUNG wire#powerrail
      { S7_Templates := "SrcType := Int" } EQ_Contact(in1 := "MODE SELECTION DB"."MODE BUFF", in2 := 1)
      { S7_Templates := "SrcType := Int" } EQ_Contact(in1 := "PREMIXING DB"."AUTO BUFF", in2 := 75)
      Coil( "AUTO ALARM DB"."PREMIXING PROCESS"."MATERIAL ADDITION DO YOU WANT TO ADD SORBITOL SELECT" )
   END_RUNG
   // the same network as SCL:
   "AUTO ALARM DB"."PREMIXING PROCESS"."MATERIAL ADDITION DO YOU WANT TO ADD SORBITOL SELECT" := ("MODE SELECTION DB"."MODE BUFF" = 1) AND ("PREMIXING DB"."AUTO BUFF" = 75);
END_REGION

REGION Network 47: MATERIAL ADDITION OF SORBITOL OVER
   RUNG wire#powerrail
      { S7_Templates := "SrcType := Int" } EQ_Contact(in1 := "MODE SELECTION DB"."MODE BUFF", in2 := 1)
      { S7_Templates := "SrcType := Int" } EQ_Contact(in1 := "PREMIXING DB"."AUTO BUFF", in2 := 100)
      Coil( "AUTO ALARM DB"."PREMIXING PROCESS"."MATERIAL ADDITION OF SORBITOL OVER" )
   END_RUNG
   // the same network as SCL:
   "AUTO ALARM DB"."PREMIXING PROCESS"."MATERIAL ADDITION OF SORBITOL OVER" := ("MODE SELECTION DB"."MODE BUFF" = 1) AND ("PREMIXING DB"."AUTO BUFF" = 100);
END_REGION

REGION Network 48: MATERIAL ADDITION DO YOU WANT TO ADD GLUCOSE SELECT
   RUNG wire#powerrail
      { S7_Templates := "SrcType := Int" } EQ_Contact(in1 := "MODE SELECTION DB"."MODE BUFF", in2 := 1)
      { S7_Templates := "SrcType := Int" } EQ_Contact(in1 := "PREMIXING DB"."AUTO BUFF", in2 := 105)
      Coil( "AUTO ALARM DB"."PREMIXING PROCESS"."MATERIAL ADDITION DO YOU WANT TO ADD GLUCOSE SELECT" )
   END_RUNG
   // the same network as SCL:
   "AUTO ALARM DB"."PREMIXING PROCESS"."MATERIAL ADDITION DO YOU WANT TO ADD GLUCOSE SELECT" := ("MODE SELECTION DB"."MODE BUFF" = 1) AND ("PREMIXING DB"."AUTO BUFF" = 105);
END_REGION

REGION Network 49: MATERIAL ADDITION OF GLUCOSE OVER
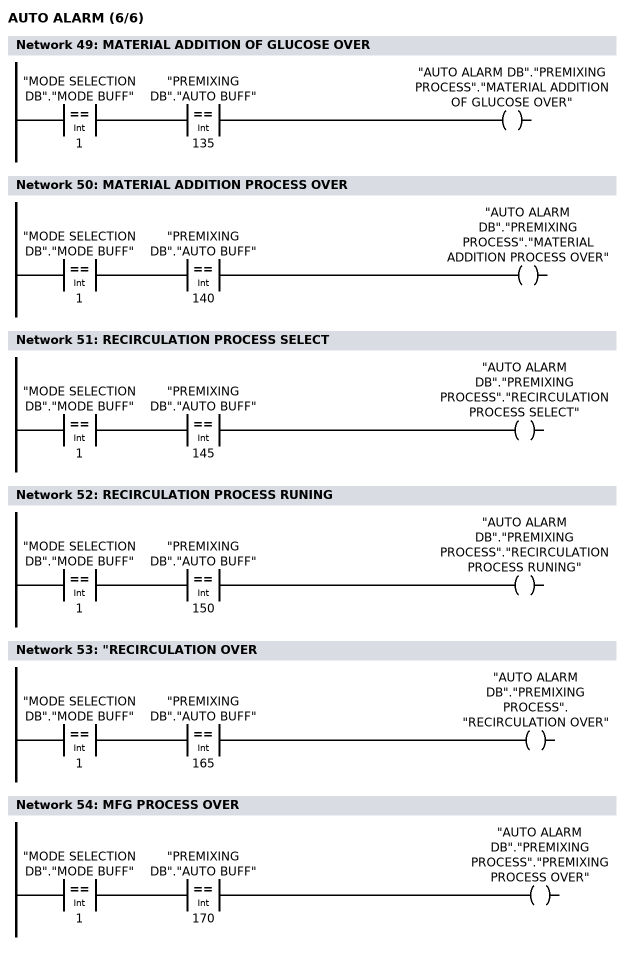
   RUNG wire#powerrail
      { S7_Templates := "SrcType := Int" } EQ_Contact(in1 := "MODE SELECTION DB"."MODE BUFF", in2 := 1)
      { S7_Templates := "SrcType := Int" } EQ_Contact(in1 := "PREMIXING DB"."AUTO BUFF", in2 := 135)
      Coil( "AUTO ALARM DB"."PREMIXING PROCESS"."MATERIAL ADDITION OF GLUCOSE OVER" )
   END_RUNG
   // the same network as SCL:
   "AUTO ALARM DB"."PREMIXING PROCESS"."MATERIAL ADDITION OF GLUCOSE OVER" := ("MODE SELECTION DB"."MODE BUFF" = 1) AND ("PREMIXING DB"."AUTO BUFF" = 135);
END_REGION

REGION Network 50: MATERIAL ADDITION PROCESS OVER
   RUNG wire#powerrail
      { S7_Templates := "SrcType := Int" } EQ_Contact(in1 := "MODE SELECTION DB"."MODE BUFF", in2 := 1)
      { S7_Templates := "SrcType := Int" } EQ_Contact(in1 := "PREMIXING DB"."AUTO BUFF", in2 := 140)
      Coil( "AUTO ALARM DB"."PREMIXING PROCESS"."MATERIAL ADDITION PROCESS OVER" )
   END_RUNG
   // the same network as SCL:
   "AUTO ALARM DB"."PREMIXING PROCESS"."MATERIAL ADDITION PROCESS OVER" := ("MODE SELECTION DB"."MODE BUFF" = 1) AND ("PREMIXING DB"."AUTO BUFF" = 140);
END_REGION

REGION Network 51: RECIRCULATION PROCESS SELECT
   RUNG wire#powerrail
      { S7_Templates := "SrcType := Int" } EQ_Contact(in1 := "MODE SELECTION DB"."MODE BUFF", in2 := 1)
      { S7_Templates := "SrcType := Int" } EQ_Contact(in1 := "PREMIXING DB"."AUTO BUFF", in2 := 145)
      Coil( "AUTO ALARM DB"."PREMIXING PROCESS"."RECIRCULATION PROCESS SELECT" )
   END_RUNG
   // the same network as SCL:
   "AUTO ALARM DB"."PREMIXING PROCESS"."RECIRCULATION PROCESS SELECT" := ("MODE SELECTION DB"."MODE BUFF" = 1) AND ("PREMIXING DB"."AUTO BUFF" = 145);
END_REGION

REGION Network 52: RECIRCULATION PROCESS RUNING
   RUNG wire#powerrail
      { S7_Templates := "SrcType := Int" } EQ_Contact(in1 := "MODE SELECTION DB"."MODE BUFF", in2 := 1)
      { S7_Templates := "SrcType := Int" } EQ_Contact(in1 := "PREMIXING DB"."AUTO BUFF", in2 := 150)
      Coil( "AUTO ALARM DB"."PREMIXING PROCESS"."RECIRCULATION PROCESS RUNING" )
   END_RUNG
   // the same network as SCL:
   "AUTO ALARM DB"."PREMIXING PROCESS"."RECIRCULATION PROCESS RUNING" := ("MODE SELECTION DB"."MODE BUFF" = 1) AND ("PREMIXING DB"."AUTO BUFF" = 150);
END_REGION

REGION Network 53: "RECIRCULATION OVER
   RUNG wire#powerrail
      { S7_Templates := "SrcType := Int" } EQ_Contact(in1 := "MODE SELECTION DB"."MODE BUFF", in2 := 1)
      { S7_Templates := "SrcType := Int" } EQ_Contact(in1 := "PREMIXING DB"."AUTO BUFF", in2 := 165)
      Coil( "AUTO ALARM DB"."PREMIXING PROCESS"."RECIRCULATION OVER" )
   END_RUNG
   // the same network as SCL:
   "AUTO ALARM DB"."PREMIXING PROCESS"."RECIRCULATION OVER" := ("MODE SELECTION DB"."MODE BUFF" = 1) AND ("PREMIXING DB"."AUTO BUFF" = 165);
END_REGION

REGION Network 54: MFG PROCESS OVER
   RUNG wire#powerrail
      { S7_Templates := "SrcType := Int" } EQ_Contact(in1 := "MODE SELECTION DB"."MODE BUFF", in2 := 1)
      { S7_Templates := "SrcType := Int" } EQ_Contact(in1 := "PREMIXING DB"."AUTO BUFF", in2 := 170)
      Coil( "AUTO ALARM DB"."PREMIXING PROCESS"."PREMIXING PROCESS OVER" )
   END_RUNG
   // the same network as SCL:
   "AUTO ALARM DB"."PREMIXING PROCESS"."PREMIXING PROCESS OVER" := ("MODE SELECTION DB"."MODE BUFF" = 1) AND ("PREMIXING DB"."AUTO BUFF" = 170);
END_REGION
END_FUNCTION

FUNCTION "MANUAL INTERLOCK" : Void   // FC8, LAD
{ S7_Optimized_Access := 'TRUE' }
// stored: SetENOAutomatically false
BEGIN

REGION Network 1: ERROR BIT
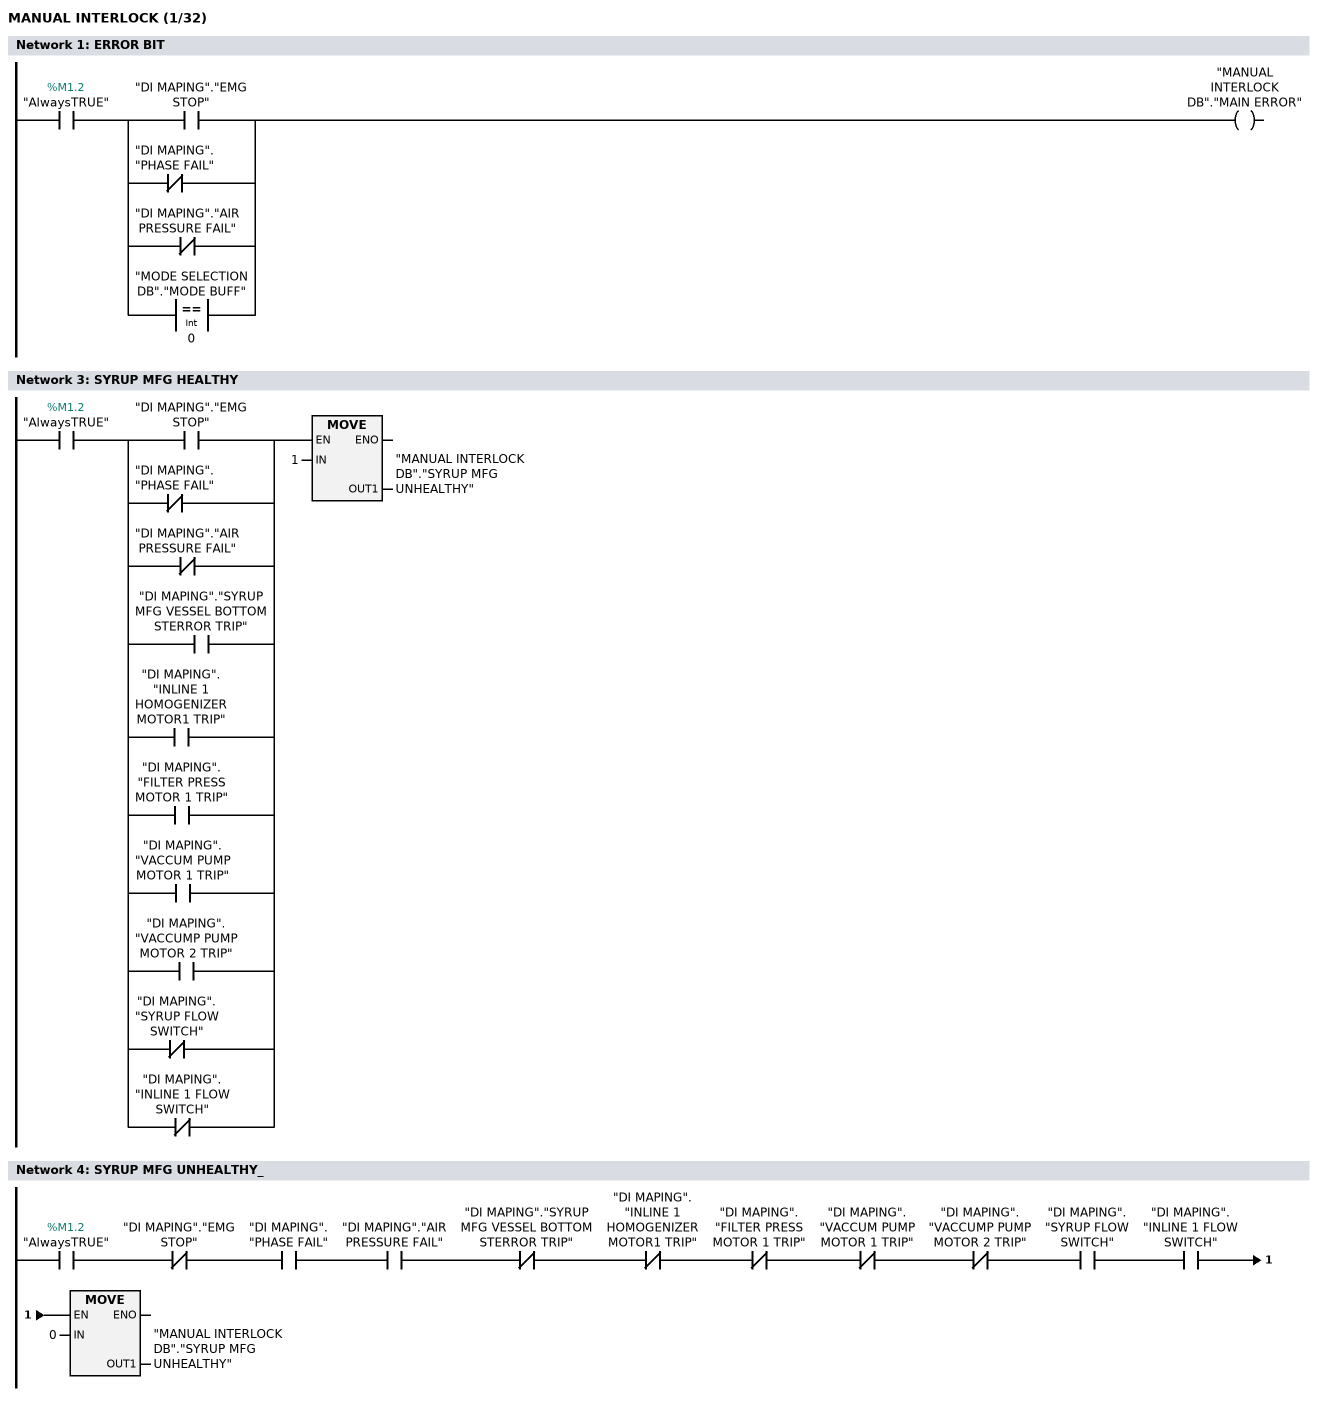
   RUNG wire#powerrail
      Contact( "AlwaysTRUE" )
      wire#w1
      Contact( "DI MAPING"."EMG STOP" )
      wire#w2
      Coil( "MANUAL INTERLOCK DB"."MAIN ERROR" )
   END_RUNG
   RUNG wire#w1
      I_Contact( "DI MAPING"."PHASE FAIL" )
   END_RUNG wire#w2
   RUNG wire#w1
      I_Contact( "DI MAPING"."AIR PRESSURE FAIL" )
   END_RUNG wire#w2
   RUNG wire#w1
      { S7_Templates := "SrcType := Int" } EQ_Contact(in1 := "MODE SELECTION DB"."MODE BUFF", in2 := 0)
   END_RUNG wire#w2
   // the same network as SCL:
   "MANUAL INTERLOCK DB"."MAIN ERROR" := "AlwaysTRUE" AND ("DI MAPING"."EMG STOP" OR NOT "DI MAPING"."PHASE FAIL" OR NOT "DI MAPING"."AIR PRESSURE FAIL" OR ("MODE SELECTION DB"."MODE BUFF" = 0));
END_REGION

REGION Network 3: SYRUP MFG HEALTHY
   RUNG wire#powerrail
      Contact( "AlwaysTRUE" )
      wire#w1
      Contact( "DI MAPING"."EMG STOP" )
      wire#w2
      Move(in := 1, out1 => "MANUAL INTERLOCK DB"."SYRUP MFG UNHEALTHY")
   END_RUNG
   RUNG wire#w1
      I_Contact( "DI MAPING"."PHASE FAIL" )
   END_RUNG wire#w2
   RUNG wire#w1
      I_Contact( "DI MAPING"."AIR PRESSURE FAIL" )
   END_RUNG wire#w2
   RUNG wire#w1
      Contact( "DI MAPING"."SYRUP MFG VESSEL BOTTOM STERROR TRIP" )
   END_RUNG wire#w2
   RUNG wire#w1
      Contact( "DI MAPING"."INLINE 1 HOMOGENIZER MOTOR1 TRIP" )
   END_RUNG wire#w2
   RUNG wire#w1
      Contact( "DI MAPING"."FILTER PRESS MOTOR 1 TRIP" )
   END_RUNG wire#w2
   RUNG wire#w1
      Contact( "DI MAPING"."VACCUM PUMP MOTOR 1 TRIP" )
   END_RUNG wire#w2
   RUNG wire#w1
      Contact( "DI MAPING"."VACCUMP PUMP MOTOR 2 TRIP" )
   END_RUNG wire#w2
   RUNG wire#w1
      I_Contact( "DI MAPING"."SYRUP FLOW SWITCH" )
   END_RUNG wire#w2
   RUNG wire#w1
      I_Contact( "DI MAPING"."INLINE 1 FLOW SWITCH" )
   END_RUNG wire#w2
   // the same network as SCL:
   IF "AlwaysTRUE" AND ("DI MAPING"."EMG STOP" OR NOT "DI MAPING"."PHASE FAIL" OR NOT "DI MAPING"."AIR PRESSURE FAIL" OR "DI MAPING"."SYRUP MFG VESSEL BOTTOM STERROR TRIP" OR "DI MAPING"."INLINE 1 HOMOGENIZER MOTOR1 TRIP" OR "DI MAPING"."FILTER PRESS MOTOR 1 TRIP" OR "DI MAPING"."VACCUM PUMP MOTOR 1 TRIP" OR "DI MAPING"."VACCUMP PUMP MOTOR 2 TRIP" OR NOT "DI MAPING"."SYRUP FLOW SWITCH" OR NOT "DI MAPING"."INLINE 1 FLOW SWITCH") THEN
       "MANUAL INTERLOCK DB"."SYRUP MFG UNHEALTHY" := 1;
   END_IF;
END_REGION

REGION Network 4: SYRUP MFG UNHEALTHY_
   RUNG wire#powerrail
      Contact( "AlwaysTRUE" )
      I_Contact( "DI MAPING"."EMG STOP" )
      Contact( "DI MAPING"."PHASE FAIL" )
      Contact( "DI MAPING"."AIR PRESSURE FAIL" )
      I_Contact( "DI MAPING"."SYRUP MFG VESSEL BOTTOM STERROR TRIP" )
      I_Contact( "DI MAPING"."INLINE 1 HOMOGENIZER MOTOR1 TRIP" )
      I_Contact( "DI MAPING"."FILTER PRESS MOTOR 1 TRIP" )
      I_Contact( "DI MAPING"."VACCUM PUMP MOTOR 1 TRIP" )
      I_Contact( "DI MAPING"."VACCUMP PUMP MOTOR 2 TRIP" )
      Contact( "DI MAPING"."SYRUP FLOW SWITCH" )
      Contact( "DI MAPING"."INLINE 1 FLOW SWITCH" )
      Move(in := 0, out1 => "MANUAL INTERLOCK DB"."SYRUP MFG UNHEALTHY")
   END_RUNG
   // the same network as SCL:
   IF "AlwaysTRUE" AND NOT "DI MAPING"."EMG STOP" AND "DI MAPING"."PHASE FAIL" AND "DI MAPING"."AIR PRESSURE FAIL" AND NOT "DI MAPING"."SYRUP MFG VESSEL BOTTOM STERROR TRIP" AND NOT "DI MAPING"."INLINE 1 HOMOGENIZER MOTOR1 TRIP" AND NOT "DI MAPING"."FILTER PRESS MOTOR 1 TRIP" AND NOT "DI MAPING"."VACCUM PUMP MOTOR 1 TRIP" AND NOT "DI MAPING"."VACCUMP PUMP MOTOR 2 TRIP" AND "DI MAPING"."SYRUP FLOW SWITCH" AND "DI MAPING"."INLINE 1 FLOW SWITCH" THEN
       "MANUAL INTERLOCK DB"."SYRUP MFG UNHEALTHY" := 0;
   END_IF;
END_REGION

REGION Network 5: PREMIXING HEALTHY
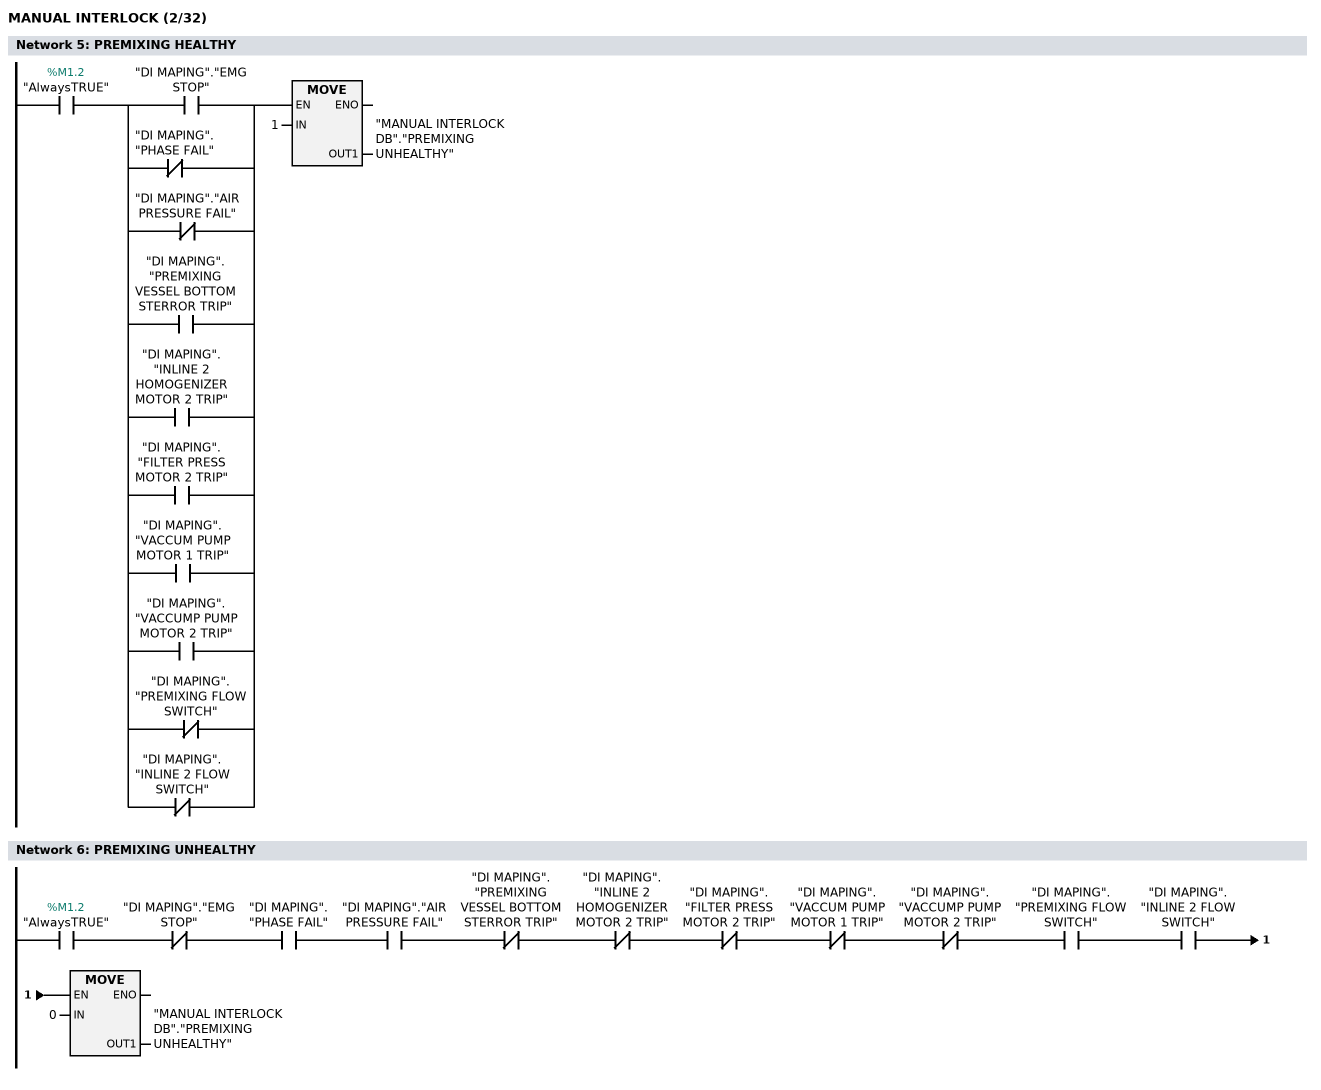
   RUNG wire#powerrail
      Contact( "AlwaysTRUE" )
      wire#w1
      Contact( "DI MAPING"."EMG STOP" )
      wire#w2
      Move(in := 1, out1 => "MANUAL INTERLOCK DB"."PREMIXING UNHEALTHY")
   END_RUNG
   RUNG wire#w1
      I_Contact( "DI MAPING"."PHASE FAIL" )
   END_RUNG wire#w2
   RUNG wire#w1
      I_Contact( "DI MAPING"."AIR PRESSURE FAIL" )
   END_RUNG wire#w2
   RUNG wire#w1
      Contact( "DI MAPING"."PREMIXING VESSEL BOTTOM STERROR TRIP" )
   END_RUNG wire#w2
   RUNG wire#w1
      Contact( "DI MAPING"."INLINE 2 HOMOGENIZER MOTOR 2 TRIP" )
   END_RUNG wire#w2
   RUNG wire#w1
      Contact( "DI MAPING"."FILTER PRESS MOTOR 2 TRIP" )
   END_RUNG wire#w2
   RUNG wire#w1
      Contact( "DI MAPING"."VACCUM PUMP MOTOR 1 TRIP" )
   END_RUNG wire#w2
   RUNG wire#w1
      Contact( "DI MAPING"."VACCUMP PUMP MOTOR 2 TRIP" )
   END_RUNG wire#w2
   RUNG wire#w1
      I_Contact( "DI MAPING"."PREMIXING FLOW SWITCH" )
   END_RUNG wire#w2
   RUNG wire#w1
      I_Contact( "DI MAPING"."INLINE 2 FLOW SWITCH" )
   END_RUNG wire#w2
   // the same network as SCL:
   IF "AlwaysTRUE" AND ("DI MAPING"."EMG STOP" OR NOT "DI MAPING"."PHASE FAIL" OR NOT "DI MAPING"."AIR PRESSURE FAIL" OR "DI MAPING"."PREMIXING VESSEL BOTTOM STERROR TRIP" OR "DI MAPING"."INLINE 2 HOMOGENIZER MOTOR 2 TRIP" OR "DI MAPING"."FILTER PRESS MOTOR 2 TRIP" OR "DI MAPING"."VACCUM PUMP MOTOR 1 TRIP" OR "DI MAPING"."VACCUMP PUMP MOTOR 2 TRIP" OR NOT "DI MAPING"."PREMIXING FLOW SWITCH" OR NOT "DI MAPING"."INLINE 2 FLOW SWITCH") THEN
       "MANUAL INTERLOCK DB"."PREMIXING UNHEALTHY" := 1;
   END_IF;
END_REGION

REGION Network 6: PREMIXING UNHEALTHY
   RUNG wire#powerrail
      Contact( "AlwaysTRUE" )
      I_Contact( "DI MAPING"."EMG STOP" )
      Contact( "DI MAPING"."PHASE FAIL" )
      Contact( "DI MAPING"."AIR PRESSURE FAIL" )
      I_Contact( "DI MAPING"."PREMIXING VESSEL BOTTOM STERROR TRIP" )
      I_Contact( "DI MAPING"."INLINE 2 HOMOGENIZER MOTOR 2 TRIP" )
      I_Contact( "DI MAPING"."FILTER PRESS MOTOR 2 TRIP" )
      I_Contact( "DI MAPING"."VACCUM PUMP MOTOR 1 TRIP" )
      I_Contact( "DI MAPING"."VACCUMP PUMP MOTOR 2 TRIP" )
      Contact( "DI MAPING"."PREMIXING FLOW SWITCH" )
      Contact( "DI MAPING"."INLINE 2 FLOW SWITCH" )
      Move(in := 0, out1 => "MANUAL INTERLOCK DB"."PREMIXING UNHEALTHY")
   END_RUNG
   // the same network as SCL:
   IF "AlwaysTRUE" AND NOT "DI MAPING"."EMG STOP" AND "DI MAPING"."PHASE FAIL" AND "DI MAPING"."AIR PRESSURE FAIL" AND NOT "DI MAPING"."PREMIXING VESSEL BOTTOM STERROR TRIP" AND NOT "DI MAPING"."INLINE 2 HOMOGENIZER MOTOR 2 TRIP" AND NOT "DI MAPING"."FILTER PRESS MOTOR 2 TRIP" AND NOT "DI MAPING"."VACCUM PUMP MOTOR 1 TRIP" AND NOT "DI MAPING"."VACCUMP PUMP MOTOR 2 TRIP" AND "DI MAPING"."PREMIXING FLOW SWITCH" AND "DI MAPING"."INLINE 2 FLOW SWITCH" THEN
       "MANUAL INTERLOCK DB"."PREMIXING UNHEALTHY" := 0;
   END_IF;
END_REGION

REGION Network 7: SUGAR HEALTHY
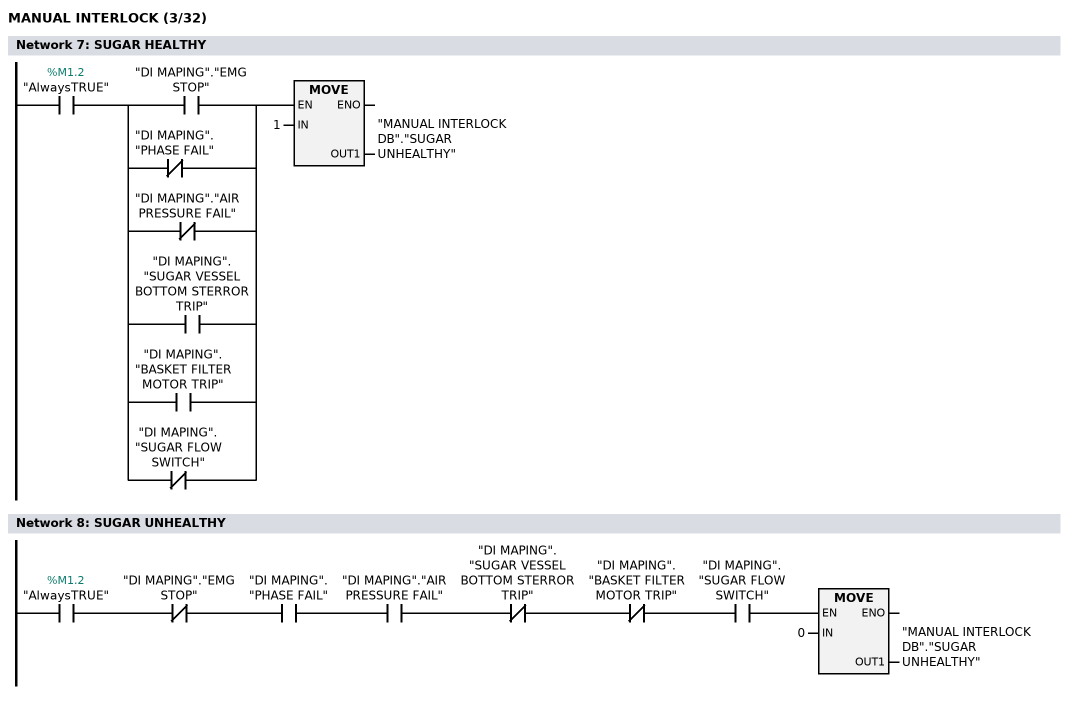
   RUNG wire#powerrail
      Contact( "AlwaysTRUE" )
      wire#w1
      Contact( "DI MAPING"."EMG STOP" )
      wire#w2
      Move(in := 1, out1 => "MANUAL INTERLOCK DB"."SUGAR UNHEALTHY")
   END_RUNG
   RUNG wire#w1
      I_Contact( "DI MAPING"."PHASE FAIL" )
   END_RUNG wire#w2
   RUNG wire#w1
      I_Contact( "DI MAPING"."AIR PRESSURE FAIL" )
   END_RUNG wire#w2
   RUNG wire#w1
      Contact( "DI MAPING"."SUGAR VESSEL BOTTOM STERROR TRIP" )
   END_RUNG wire#w2
   RUNG wire#w1
      Contact( "DI MAPING"."BASKET FILTER MOTOR TRIP" )
   END_RUNG wire#w2
   RUNG wire#w1
      I_Contact( "DI MAPING"."SUGAR FLOW SWITCH" )
   END_RUNG wire#w2
   // the same network as SCL:
   IF "AlwaysTRUE" AND ("DI MAPING"."EMG STOP" OR NOT "DI MAPING"."PHASE FAIL" OR NOT "DI MAPING"."AIR PRESSURE FAIL" OR "DI MAPING"."SUGAR VESSEL BOTTOM STERROR TRIP" OR "DI MAPING"."BASKET FILTER MOTOR TRIP" OR NOT "DI MAPING"."SUGAR FLOW SWITCH") THEN
       "MANUAL INTERLOCK DB"."SUGAR UNHEALTHY" := 1;
   END_IF;
END_REGION

REGION Network 8: SUGAR UNHEALTHY
   RUNG wire#powerrail
      Contact( "AlwaysTRUE" )
      I_Contact( "DI MAPING"."EMG STOP" )
      Contact( "DI MAPING"."PHASE FAIL" )
      Contact( "DI MAPING"."AIR PRESSURE FAIL" )
      I_Contact( "DI MAPING"."SUGAR VESSEL BOTTOM STERROR TRIP" )
      I_Contact( "DI MAPING"."BASKET FILTER MOTOR TRIP" )
      Contact( "DI MAPING"."SUGAR FLOW SWITCH" )
      Move(in := 0, out1 => "MANUAL INTERLOCK DB"."SUGAR UNHEALTHY")
   END_RUNG
   // the same network as SCL:
   IF "AlwaysTRUE" AND NOT "DI MAPING"."EMG STOP" AND "DI MAPING"."PHASE FAIL" AND "DI MAPING"."AIR PRESSURE FAIL" AND NOT "DI MAPING"."SUGAR VESSEL BOTTOM STERROR TRIP" AND NOT "DI MAPING"."BASKET FILTER MOTOR TRIP" AND "DI MAPING"."SUGAR FLOW SWITCH" THEN
       "MANUAL INTERLOCK DB"."SUGAR UNHEALTHY" := 0;
   END_IF;
END_REGION

REGION Network 10: ------------------------------------------ CONTINUE RESET-------------------------------------
END_REGION

REGION Network 11: SYRUP MFG PROCESS ERROR FOR CONTINUE
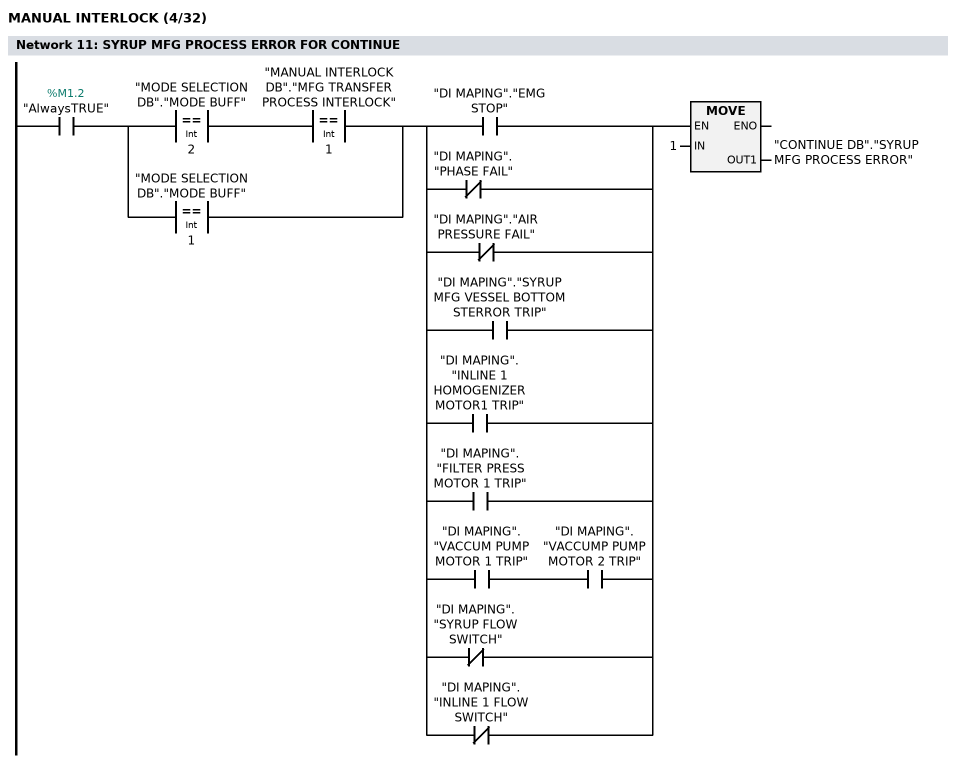
   RUNG wire#powerrail
      Contact( "AlwaysTRUE" )
      wire#w1
      { S7_Templates := "SrcType := Int" } EQ_Contact(in1 := "MODE SELECTION DB"."MODE BUFF", in2 := 2)
      { S7_Templates := "SrcType := Int" } EQ_Contact(in1 := "MANUAL INTERLOCK DB"."MFG TRANSFER PROCESS INTERLOCK", in2 := 1)
      wire#w2
      Contact( "DI MAPING"."EMG STOP" )
      wire#w3
      Move(in := 1, out1 => "CONTINUE DB"."SYRUP MFG PROCESS ERROR")
   END_RUNG
   RUNG wire#w1
      { S7_Templates := "SrcType := Int" } EQ_Contact(in1 := "MODE SELECTION DB"."MODE BUFF", in2 := 1)
   END_RUNG wire#w2
   RUNG wire#w2
      I_Contact( "DI MAPING"."PHASE FAIL" )
   END_RUNG wire#w3
   RUNG wire#w2
      I_Contact( "DI MAPING"."AIR PRESSURE FAIL" )
   END_RUNG wire#w3
   RUNG wire#w2
      Contact( "DI MAPING"."SYRUP MFG VESSEL BOTTOM STERROR TRIP" )
   END_RUNG wire#w3
   RUNG wire#w2
      Contact( "DI MAPING"."INLINE 1 HOMOGENIZER MOTOR1 TRIP" )
   END_RUNG wire#w3
   RUNG wire#w2
      Contact( "DI MAPING"."FILTER PRESS MOTOR 1 TRIP" )
   END_RUNG wire#w3
   RUNG wire#w2
      Contact( "DI MAPING"."VACCUM PUMP MOTOR 1 TRIP" )
      Contact( "DI MAPING"."VACCUMP PUMP MOTOR 2 TRIP" )
   END_RUNG wire#w3
   RUNG wire#w2
      I_Contact( "DI MAPING"."SYRUP FLOW SWITCH" )
   END_RUNG wire#w3
   RUNG wire#w2
      I_Contact( "DI MAPING"."INLINE 1 FLOW SWITCH" )
   END_RUNG wire#w3
   // the same network as SCL:
   IF "AlwaysTRUE" AND ((("MODE SELECTION DB"."MODE BUFF" = 2) AND ("MANUAL INTERLOCK DB"."MFG TRANSFER PROCESS INTERLOCK" = 1)) OR ("MODE SELECTION DB"."MODE BUFF" = 1)) AND ("DI MAPING"."EMG STOP" OR NOT "DI MAPING"."PHASE FAIL" OR NOT "DI MAPING"."AIR PRESSURE FAIL" OR "DI MAPING"."SYRUP MFG VESSEL BOTTOM STERROR TRIP" OR "DI MAPING"."INLINE 1 HOMOGENIZER MOTOR1 TRIP" OR "DI MAPING"."FILTER PRESS MOTOR 1 TRIP" OR ("DI MAPING"."VACCUM PUMP MOTOR 1 TRIP" AND "DI MAPING"."VACCUMP PUMP MOTOR 2 TRIP") OR NOT "DI MAPING"."SYRUP FLOW SWITCH" OR NOT "DI MAPING"."INLINE 1 FLOW SWITCH") THEN
       "CONTINUE DB"."SYRUP MFG PROCESS ERROR" := 1;
   END_IF;
END_REGION

REGION Network 12: PREMIXING PROCESS ERROR FOR CONTINUE
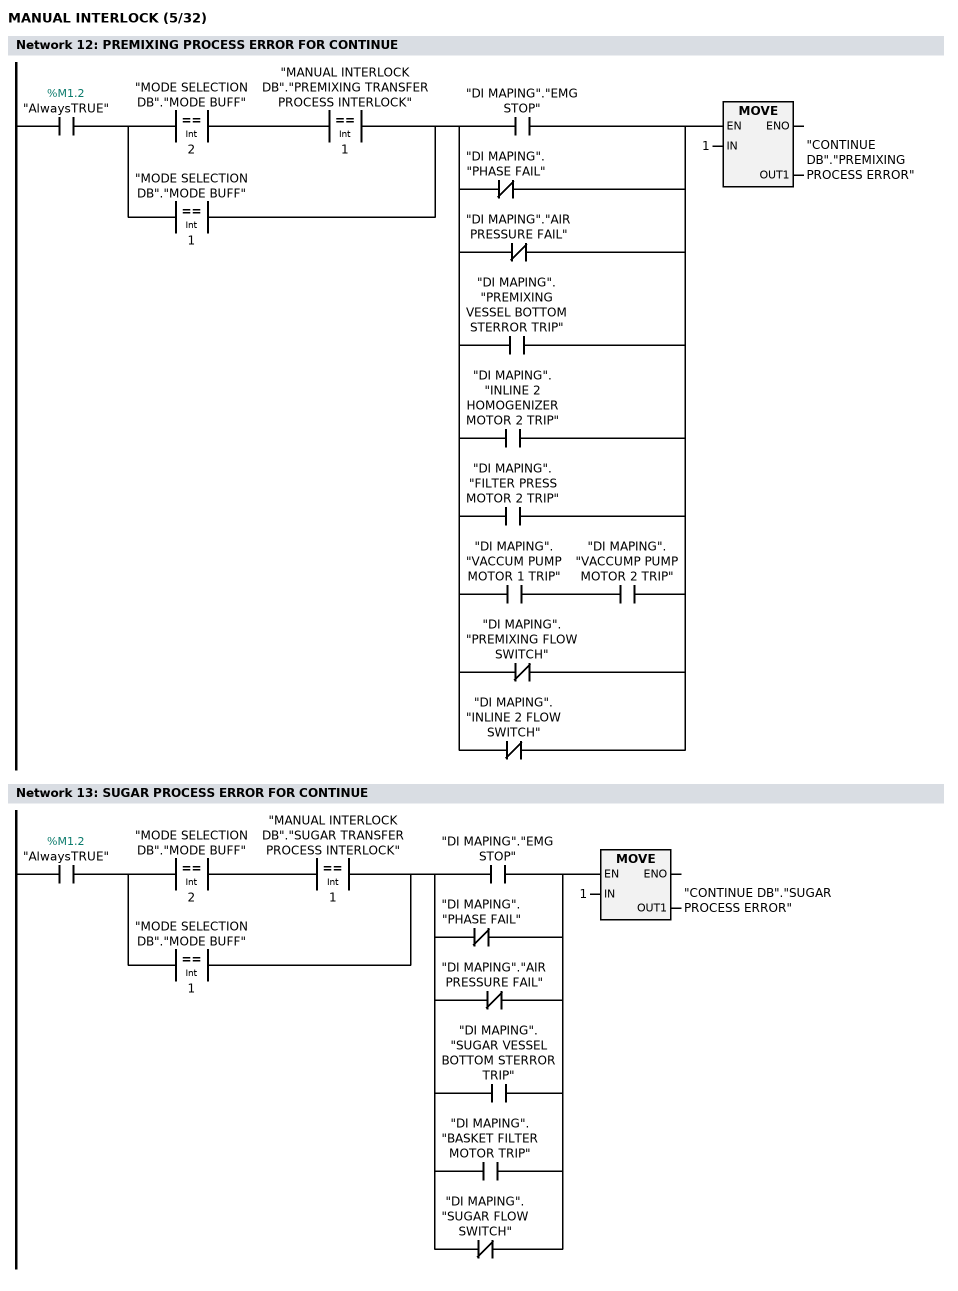
   RUNG wire#powerrail
      Contact( "AlwaysTRUE" )
      wire#w1
      { S7_Templates := "SrcType := Int" } EQ_Contact(in1 := "MODE SELECTION DB"."MODE BUFF", in2 := 2)
      { S7_Templates := "SrcType := Int" } EQ_Contact(in1 := "MANUAL INTERLOCK DB"."PREMIXING TRANSFER PROCESS INTERLOCK", in2 := 1)
      wire#w2
      Contact( "DI MAPING"."EMG STOP" )
      wire#w3
      Move(in := 1, out1 => "CONTINUE DB"."PREMIXING PROCESS ERROR")
   END_RUNG
   RUNG wire#w1
      { S7_Templates := "SrcType := Int" } EQ_Contact(in1 := "MODE SELECTION DB"."MODE BUFF", in2 := 1)
   END_RUNG wire#w2
   RUNG wire#w2
      I_Contact( "DI MAPING"."PHASE FAIL" )
   END_RUNG wire#w3
   RUNG wire#w2
      I_Contact( "DI MAPING"."AIR PRESSURE FAIL" )
   END_RUNG wire#w3
   RUNG wire#w2
      Contact( "DI MAPING"."PREMIXING VESSEL BOTTOM STERROR TRIP" )
   END_RUNG wire#w3
   RUNG wire#w2
      Contact( "DI MAPING"."INLINE 2 HOMOGENIZER MOTOR 2 TRIP" )
   END_RUNG wire#w3
   RUNG wire#w2
      Contact( "DI MAPING"."FILTER PRESS MOTOR 2 TRIP" )
   END_RUNG wire#w3
   RUNG wire#w2
      Contact( "DI MAPING"."VACCUM PUMP MOTOR 1 TRIP" )
      Contact( "DI MAPING"."VACCUMP PUMP MOTOR 2 TRIP" )
   END_RUNG wire#w3
   RUNG wire#w2
      I_Contact( "DI MAPING"."PREMIXING FLOW SWITCH" )
   END_RUNG wire#w3
   RUNG wire#w2
      I_Contact( "DI MAPING"."INLINE 2 FLOW SWITCH" )
   END_RUNG wire#w3
   // the same network as SCL:
   IF "AlwaysTRUE" AND ((("MODE SELECTION DB"."MODE BUFF" = 2) AND ("MANUAL INTERLOCK DB"."PREMIXING TRANSFER PROCESS INTERLOCK" = 1)) OR ("MODE SELECTION DB"."MODE BUFF" = 1)) AND ("DI MAPING"."EMG STOP" OR NOT "DI MAPING"."PHASE FAIL" OR NOT "DI MAPING"."AIR PRESSURE FAIL" OR "DI MAPING"."PREMIXING VESSEL BOTTOM STERROR TRIP" OR "DI MAPING"."INLINE 2 HOMOGENIZER MOTOR 2 TRIP" OR "DI MAPING"."FILTER PRESS MOTOR 2 TRIP" OR ("DI MAPING"."VACCUM PUMP MOTOR 1 TRIP" AND "DI MAPING"."VACCUMP PUMP MOTOR 2 TRIP") OR NOT "DI MAPING"."PREMIXING FLOW SWITCH" OR NOT "DI MAPING"."INLINE 2 FLOW SWITCH") THEN
       "CONTINUE DB"."PREMIXING PROCESS ERROR" := 1;
   END_IF;
END_REGION

REGION Network 13: SUGAR PROCESS ERROR FOR CONTINUE
   RUNG wire#powerrail
      Contact( "AlwaysTRUE" )
      wire#w1
      { S7_Templates := "SrcType := Int" } EQ_Contact(in1 := "MODE SELECTION DB"."MODE BUFF", in2 := 2)
      { S7_Templates := "SrcType := Int" } EQ_Contact(in1 := "MANUAL INTERLOCK DB"."SUGAR TRANSFER PROCESS INTERLOCK", in2 := 1)
      wire#w2
      Contact( "DI MAPING"."EMG STOP" )
      wire#w3
      Move(in := 1, out1 => "CONTINUE DB"."SUGAR PROCESS ERROR")
   END_RUNG
   RUNG wire#w1
      { S7_Templates := "SrcType := Int" } EQ_Contact(in1 := "MODE SELECTION DB"."MODE BUFF", in2 := 1)
   END_RUNG wire#w2
   RUNG wire#w2
      I_Contact( "DI MAPING"."PHASE FAIL" )
   END_RUNG wire#w3
   RUNG wire#w2
      I_Contact( "DI MAPING"."AIR PRESSURE FAIL" )
   END_RUNG wire#w3
   RUNG wire#w2
      Contact( "DI MAPING"."SUGAR VESSEL BOTTOM STERROR TRIP" )
   END_RUNG wire#w3
   RUNG wire#w2
      Contact( "DI MAPING"."BASKET FILTER MOTOR TRIP" )
   END_RUNG wire#w3
   RUNG wire#w2
      I_Contact( "DI MAPING"."SUGAR FLOW SWITCH" )
   END_RUNG wire#w3
   // the same network as SCL:
   IF "AlwaysTRUE" AND ((("MODE SELECTION DB"."MODE BUFF" = 2) AND ("MANUAL INTERLOCK DB"."SUGAR TRANSFER PROCESS INTERLOCK" = 1)) OR ("MODE SELECTION DB"."MODE BUFF" = 1)) AND ("DI MAPING"."EMG STOP" OR NOT "DI MAPING"."PHASE FAIL" OR NOT "DI MAPING"."AIR PRESSURE FAIL" OR "DI MAPING"."SUGAR VESSEL BOTTOM STERROR TRIP" OR "DI MAPING"."BASKET FILTER MOTOR TRIP" OR NOT "DI MAPING"."SUGAR FLOW SWITCH") THEN
       "CONTINUE DB"."SUGAR PROCESS ERROR" := 1;
   END_IF;
END_REGION

REGION Network 15: CONTINUE PROCESS-SYRUP MFG
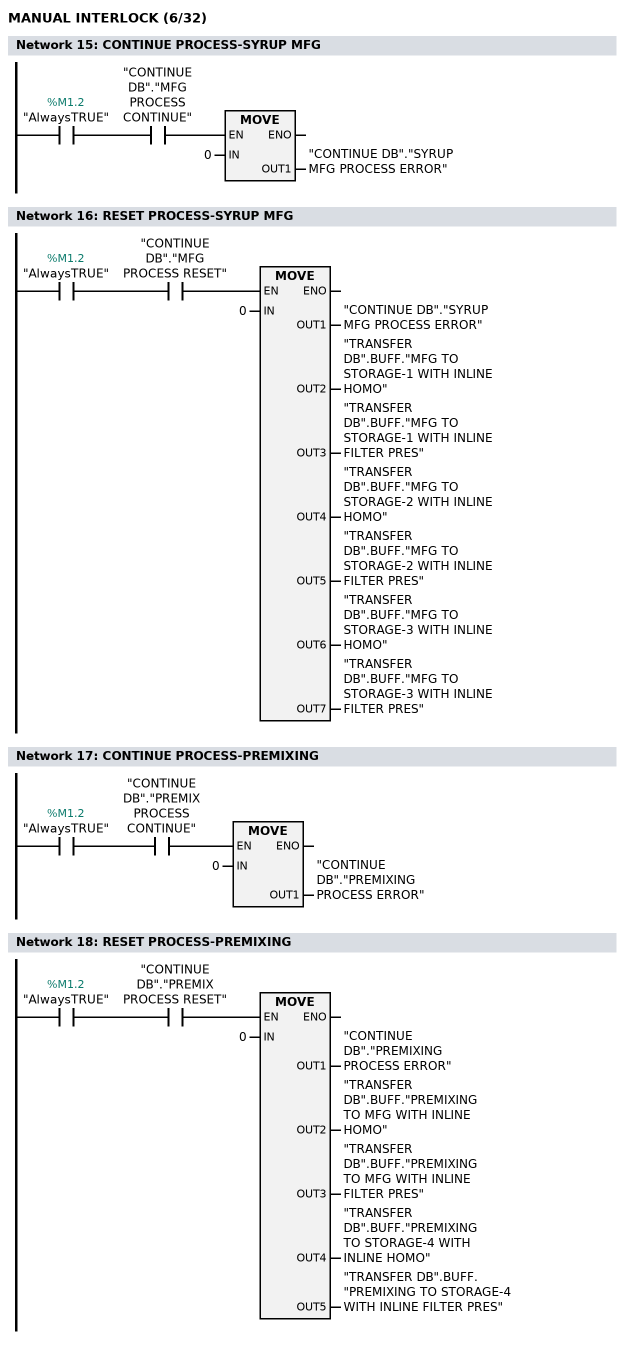
   RUNG wire#powerrail
      Contact( "AlwaysTRUE" )
      Contact( "CONTINUE DB"."MFG PROCESS CONTINUE" )
      Move(in := 0, out1 => "CONTINUE DB"."SYRUP MFG PROCESS ERROR")
   END_RUNG
   // the same network as SCL:
   IF "AlwaysTRUE" AND "CONTINUE DB"."MFG PROCESS CONTINUE" THEN
       "CONTINUE DB"."SYRUP MFG PROCESS ERROR" := 0;
   END_IF;
END_REGION

REGION Network 16: RESET PROCESS-SYRUP MFG
   RUNG wire#powerrail
      Contact( "AlwaysTRUE" )
      Contact( "CONTINUE DB"."MFG PROCESS RESET" )
      Move(in := 0, out1 => "CONTINUE DB"."SYRUP MFG PROCESS ERROR", out2 => "TRANSFER DB".BUFF."MFG TO STORAGE-1 WITH INLINE HOMO", out3 => "TRANSFER DB".BUFF."MFG TO STORAGE-1 WITH INLINE FILTER PRES", out4 => "TRANSFER DB".BUFF."MFG TO STORAGE-2 WITH INLINE HOMO", out5 => "TRANSFER DB".BUFF."MFG TO STORAGE-2 WITH INLINE FILTER PRES", out6 => "TRANSFER DB".BUFF."MFG TO STORAGE-3 WITH INLINE HOMO", out7 => "TRANSFER DB".BUFF."MFG TO STORAGE-3 WITH INLINE FILTER PRES")
   END_RUNG
   // the same network as SCL:
   IF "AlwaysTRUE" AND "CONTINUE DB"."MFG PROCESS RESET" THEN
       "CONTINUE DB"."SYRUP MFG PROCESS ERROR" := 0;
       "TRANSFER DB".BUFF."MFG TO STORAGE-1 WITH INLINE HOMO" := 0;
       "TRANSFER DB".BUFF."MFG TO STORAGE-1 WITH INLINE FILTER PRES" := 0;
       "TRANSFER DB".BUFF."MFG TO STORAGE-2 WITH INLINE HOMO" := 0;
       "TRANSFER DB".BUFF."MFG TO STORAGE-2 WITH INLINE FILTER PRES" := 0;
       "TRANSFER DB".BUFF."MFG TO STORAGE-3 WITH INLINE HOMO" := 0;
       "TRANSFER DB".BUFF."MFG TO STORAGE-3 WITH INLINE FILTER PRES" := 0;
   END_IF;
END_REGION

REGION Network 17: CONTINUE PROCESS-PREMIXING
   RUNG wire#powerrail
      Contact( "AlwaysTRUE" )
      Contact( "CONTINUE DB"."PREMIX PROCESS CONTINUE" )
      Move(in := 0, out1 => "CONTINUE DB"."PREMIXING PROCESS ERROR")
   END_RUNG
   // the same network as SCL:
   IF "AlwaysTRUE" AND "CONTINUE DB"."PREMIX PROCESS CONTINUE" THEN
       "CONTINUE DB"."PREMIXING PROCESS ERROR" := 0;
   END_IF;
END_REGION

REGION Network 18: RESET PROCESS-PREMIXING
   RUNG wire#powerrail
      Contact( "AlwaysTRUE" )
      Contact( "CONTINUE DB"."PREMIX PROCESS RESET" )
      Move(in := 0, out1 => "CONTINUE DB"."PREMIXING PROCESS ERROR", out2 => "TRANSFER DB".BUFF."PREMIXING TO MFG WITH INLINE HOMO", out3 => "TRANSFER DB".BUFF."PREMIXING TO MFG WITH INLINE FILTER PRES", out4 => "TRANSFER DB".BUFF."PREMIXING TO STORAGE-4 WITH INLINE HOMO", out5 => "TRANSFER DB".BUFF."PREMIXING TO STORAGE-4 WITH INLINE FILTER PRES")
   END_RUNG
   // the same network as SCL:
   IF "AlwaysTRUE" AND "CONTINUE DB"."PREMIX PROCESS RESET" THEN
       "CONTINUE DB"."PREMIXING PROCESS ERROR" := 0;
       "TRANSFER DB".BUFF."PREMIXING TO MFG WITH INLINE HOMO" := 0;
       "TRANSFER DB".BUFF."PREMIXING TO MFG WITH INLINE FILTER PRES" := 0;
       "TRANSFER DB".BUFF."PREMIXING TO STORAGE-4 WITH INLINE HOMO" := 0;
       "TRANSFER DB".BUFF."PREMIXING TO STORAGE-4 WITH INLINE FILTER PRES" := 0;
   END_IF;
END_REGION

REGION Network 19: CONTINUE PROCESS-SUGAR
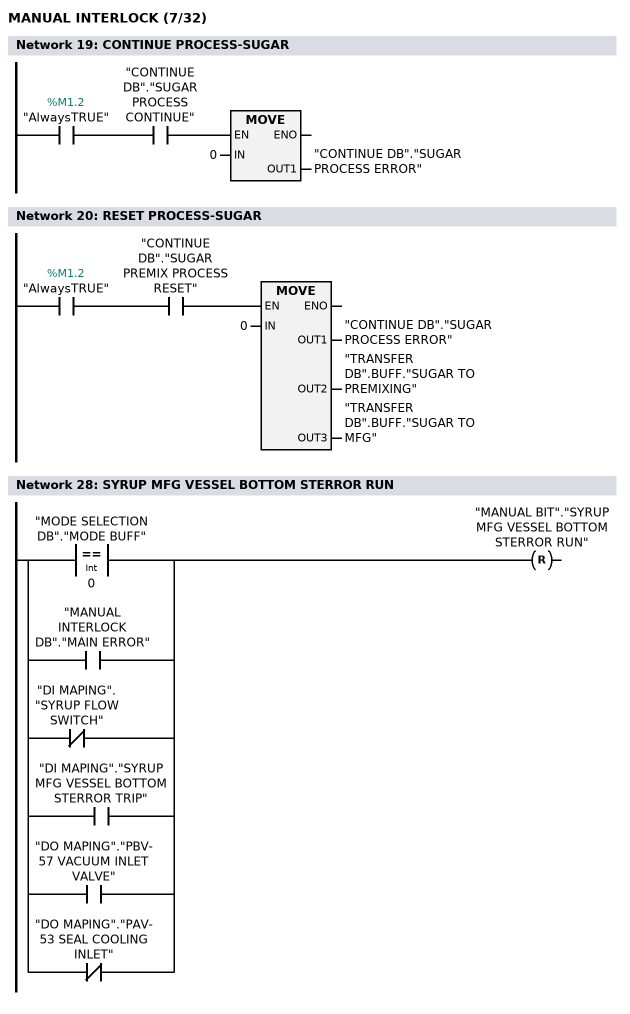
   RUNG wire#powerrail
      Contact( "AlwaysTRUE" )
      Contact( "CONTINUE DB"."SUGAR PROCESS CONTINUE" )
      Move(in := 0, out1 => "CONTINUE DB"."SUGAR PROCESS ERROR")
   END_RUNG
   // the same network as SCL:
   IF "AlwaysTRUE" AND "CONTINUE DB"."SUGAR PROCESS CONTINUE" THEN
       "CONTINUE DB"."SUGAR PROCESS ERROR" := 0;
   END_IF;
END_REGION

REGION Network 20: RESET PROCESS-SUGAR
   RUNG wire#powerrail
      Contact( "AlwaysTRUE" )
      Contact( "CONTINUE DB"."SUGAR PREMIX PROCESS RESET" )
      Move(in := 0, out1 => "CONTINUE DB"."SUGAR PROCESS ERROR", out2 => "TRANSFER DB".BUFF."SUGAR TO PREMIXING", out3 => "TRANSFER DB".BUFF."SUGAR TO MFG")
   END_RUNG
   // the same network as SCL:
   IF "AlwaysTRUE" AND "CONTINUE DB"."SUGAR PREMIX PROCESS RESET" THEN
       "CONTINUE DB"."SUGAR PROCESS ERROR" := 0;
       "TRANSFER DB".BUFF."SUGAR TO PREMIXING" := 0;
       "TRANSFER DB".BUFF."SUGAR TO MFG" := 0;
   END_IF;
END_REGION

REGION Network 22: ------------------------------TRANSFER PROCESS INTERLOCK---------------------------------------
END_REGION

REGION Network 23 (SCL): MFG TRANSFER PROCESS INTERLOCK
   IF 
       "TRANSFER DB".BUFF."MFG TO STORAGE-1 WITH INLINE HOMO" <> 0 OR
       "TRANSFER DB".BUFF."MFG TO STORAGE-1 WITH INLINE FILTER PRES" <> 0 OR
       "TRANSFER DB".BUFF."MFG TO STORAGE-2 WITH INLINE HOMO" <> 0 OR
       "TRANSFER DB".BUFF."MFG TO STORAGE-2 WITH INLINE FILTER PRES" <> 0 OR
       "TRANSFER DB".BUFF."MFG TO STORAGE-3 WITH INLINE HOMO" <> 0 OR
       "TRANSFER DB".BUFF."MFG TO STORAGE-3 WITH INLINE FILTER PRES" <> 0
   THEN
       "MANUAL INTERLOCK DB"."MFG TRANSFER PROCESS INTERLOCK" := 1;
   ELSIF "TRANSFER DB"."MFG VACCUM PUMP MOTOR-W 1 BIT"<>0
       OR "TRANSFER DB"."MFG VACCUMP PUMP MOTOR-S2 BIT"<>0
   THEN
       "MANUAL INTERLOCK DB"."MFG TRANSFER PROCESS INTERLOCK" := 2;
   ELSIF "RECIRCULATION DB".MFG.BUFF<>0
   THEN
       "MANUAL INTERLOCK DB"."MFG TRANSFER PROCESS INTERLOCK" := 3;
   ELSE
       "MANUAL INTERLOCK DB"."MFG TRANSFER PROCESS INTERLOCK" := 0;
   END_IF;
END_REGION

REGION Network 24 (SCL): PREMIXING TRANSFER PROCESS INTERLOCK
   IF
       "TRANSFER DB".BUFF."PREMIXING TO MFG WITH INLINE HOMO" <> 0 OR
       "TRANSFER DB".BUFF."PREMIXING TO MFG WITH INLINE FILTER PRES" <> 0 OR
       "TRANSFER DB".BUFF."PREMIXING TO STORAGE-4 WITH INLINE HOMO" <> 0 OR
       "TRANSFER DB".BUFF."PREMIXING TO STORAGE-4 WITH INLINE FILTER PRES" <> 0
   THEN
       "MANUAL INTERLOCK DB"."PREMIXING TRANSFER PROCESS INTERLOCK" := 1;
   ELSIF "TRANSFER DB"."PREMIXING VACCUM PUMP MOTOR-W 1 BIT"<>0 OR
       "TRANSFER DB"."PREMIXING VACCUMP PUMP MOTOR-S2 BIT"
   THEN
       "MANUAL INTERLOCK DB"."PREMIXING TRANSFER PROCESS INTERLOCK" := 2;
   ELSIF "RECIRCULATION DB".PREMIXING.BUFF<>0
   THEN
       "MANUAL INTERLOCK DB"."PREMIXING TRANSFER PROCESS INTERLOCK" := 3;
   ELSE
       "MANUAL INTERLOCK DB"."PREMIXING TRANSFER PROCESS INTERLOCK" := 0;
   END_IF;
END_REGION

REGION Network 25 (SCL): SUGAR TRANSFER PROCESS INTERLOCK
   IF "TRANSFER DB".BUFF."SUGAR TO PREMIXING" <>0 OR
       "TRANSFER DB".BUFF."SUGAR TO MFG"<>0
   THEN
       "MANUAL INTERLOCK DB"."SUGAR TRANSFER PROCESS INTERLOCK" := 1;
   ELSIF "DO MAPING"."PBV-30 VACUUM INLET VALVE" <>0
   THEN
       "MANUAL INTERLOCK DB"."SUGAR TRANSFER PROCESS INTERLOCK" := 2;
   ELSE
       "MANUAL INTERLOCK DB"."SUGAR TRANSFER PROCESS INTERLOCK" := 0;

   END_IF;
END_REGION

REGION Network 27: ------------------------------------------ MANUAL BIT RESET-------------------------------------
END_REGION

REGION Network 28: SYRUP MFG VESSEL BOTTOM STERROR RUN
   RUNG wire#powerrail
      { S7_Templates := "SrcType := Int" } EQ_Contact(in1 := "MODE SELECTION DB"."MODE BUFF", in2 := 0)
      wire#w1
      R_Coil( "MANUAL BIT"."SYRUP MFG VESSEL BOTTOM STERROR RUN" )
   END_RUNG
   RUNG wire#powerrail
      Contact( "MANUAL INTERLOCK DB"."MAIN ERROR" )
   END_RUNG wire#w1
   RUNG wire#powerrail
      I_Contact( "DI MAPING"."SYRUP FLOW SWITCH" )
   END_RUNG wire#w1
   RUNG wire#powerrail
      Contact( "DI MAPING"."SYRUP MFG VESSEL BOTTOM STERROR TRIP" )
   END_RUNG wire#w1
   RUNG wire#powerrail
      Contact( "DO MAPING"."PBV-57 VACUUM INLET VALVE" )
   END_RUNG wire#w1
   RUNG wire#powerrail
      I_Contact( "DO MAPING"."PAV-53 SEAL COOLING INLET" )
   END_RUNG wire#w1
   // the same network as SCL:
   IF ("MODE SELECTION DB"."MODE BUFF" = 0) OR "MANUAL INTERLOCK DB"."MAIN ERROR" OR NOT "DI MAPING"."SYRUP FLOW SWITCH" OR "DI MAPING"."SYRUP MFG VESSEL BOTTOM STERROR TRIP" OR "DO MAPING"."PBV-57 VACUUM INLET VALVE" OR NOT "DO MAPING"."PAV-53 SEAL COOLING INLET" THEN
       "MANUAL BIT"."SYRUP MFG VESSEL BOTTOM STERROR RUN" := FALSE;
   END_IF;
END_REGION

REGION Network 29: PREMIXING VESSEL BOTTOM STERROR RUN
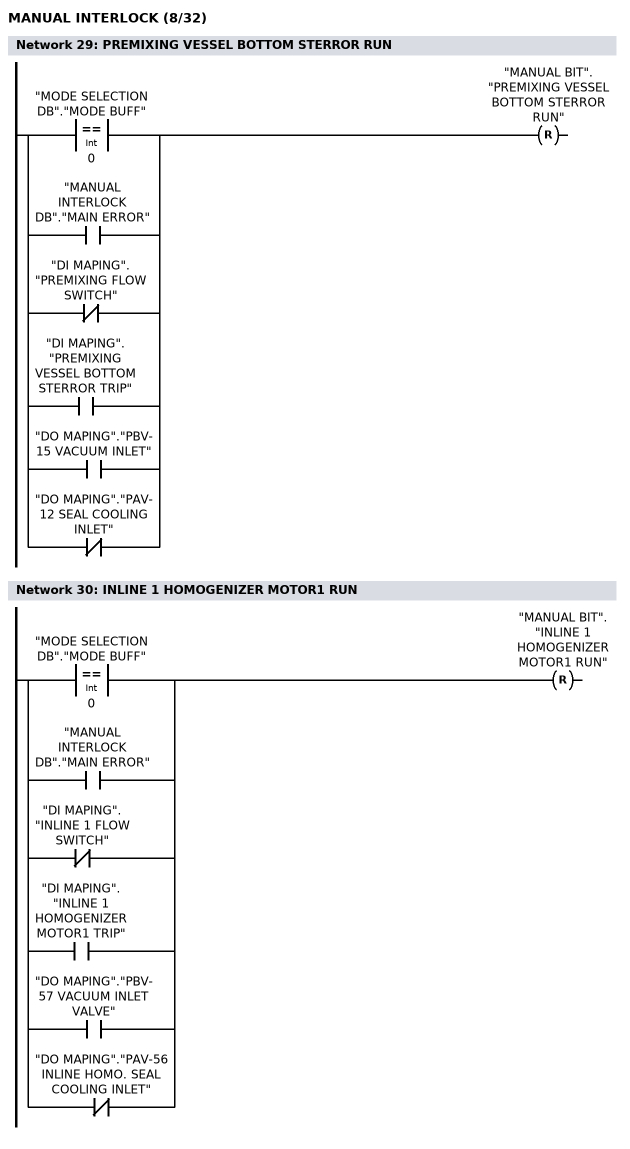
   RUNG wire#powerrail
      { S7_Templates := "SrcType := Int" } EQ_Contact(in1 := "MODE SELECTION DB"."MODE BUFF", in2 := 0)
      wire#w1
      R_Coil( "MANUAL BIT"."PREMIXING VESSEL BOTTOM STERROR RUN" )
   END_RUNG
   RUNG wire#powerrail
      Contact( "MANUAL INTERLOCK DB"."MAIN ERROR" )
   END_RUNG wire#w1
   RUNG wire#powerrail
      I_Contact( "DI MAPING"."PREMIXING FLOW SWITCH" )
   END_RUNG wire#w1
   RUNG wire#powerrail
      Contact( "DI MAPING"."PREMIXING VESSEL BOTTOM STERROR TRIP" )
   END_RUNG wire#w1
   RUNG wire#powerrail
      Contact( "DO MAPING"."PBV-15 VACUUM INLET" )
   END_RUNG wire#w1
   RUNG wire#powerrail
      I_Contact( "DO MAPING"."PAV-12 SEAL COOLING INLET" )
   END_RUNG wire#w1
   // the same network as SCL:
   IF ("MODE SELECTION DB"."MODE BUFF" = 0) OR "MANUAL INTERLOCK DB"."MAIN ERROR" OR NOT "DI MAPING"."PREMIXING FLOW SWITCH" OR "DI MAPING"."PREMIXING VESSEL BOTTOM STERROR TRIP" OR "DO MAPING"."PBV-15 VACUUM INLET" OR NOT "DO MAPING"."PAV-12 SEAL COOLING INLET" THEN
       "MANUAL BIT"."PREMIXING VESSEL BOTTOM STERROR RUN" := FALSE;
   END_IF;
END_REGION

REGION Network 30: INLINE 1 HOMOGENIZER MOTOR1 RUN
   RUNG wire#powerrail
      { S7_Templates := "SrcType := Int" } EQ_Contact(in1 := "MODE SELECTION DB"."MODE BUFF", in2 := 0)
      wire#w1
      R_Coil( "MANUAL BIT"."INLINE 1 HOMOGENIZER MOTOR1 RUN" )
   END_RUNG
   RUNG wire#powerrail
      Contact( "MANUAL INTERLOCK DB"."MAIN ERROR" )
   END_RUNG wire#w1
   RUNG wire#powerrail
      I_Contact( "DI MAPING"."INLINE 1 FLOW SWITCH" )
   END_RUNG wire#w1
   RUNG wire#powerrail
      Contact( "DI MAPING"."INLINE 1 HOMOGENIZER MOTOR1 TRIP" )
   END_RUNG wire#w1
   RUNG wire#powerrail
      Contact( "DO MAPING"."PBV-57 VACUUM INLET VALVE" )
   END_RUNG wire#w1
   RUNG wire#powerrail
      I_Contact( "DO MAPING"."PAV-56 INLINE HOMO. SEAL COOLING INLET" )
   END_RUNG wire#w1
   // the same network as SCL:
   IF ("MODE SELECTION DB"."MODE BUFF" = 0) OR "MANUAL INTERLOCK DB"."MAIN ERROR" OR NOT "DI MAPING"."INLINE 1 FLOW SWITCH" OR "DI MAPING"."INLINE 1 HOMOGENIZER MOTOR1 TRIP" OR "DO MAPING"."PBV-57 VACUUM INLET VALVE" OR NOT "DO MAPING"."PAV-56 INLINE HOMO. SEAL COOLING INLET" THEN
       "MANUAL BIT"."INLINE 1 HOMOGENIZER MOTOR1 RUN" := FALSE;
   END_IF;
END_REGION

REGION Network 31: INLINE 2 HOMOGENIZER MOTOR 2 RUN
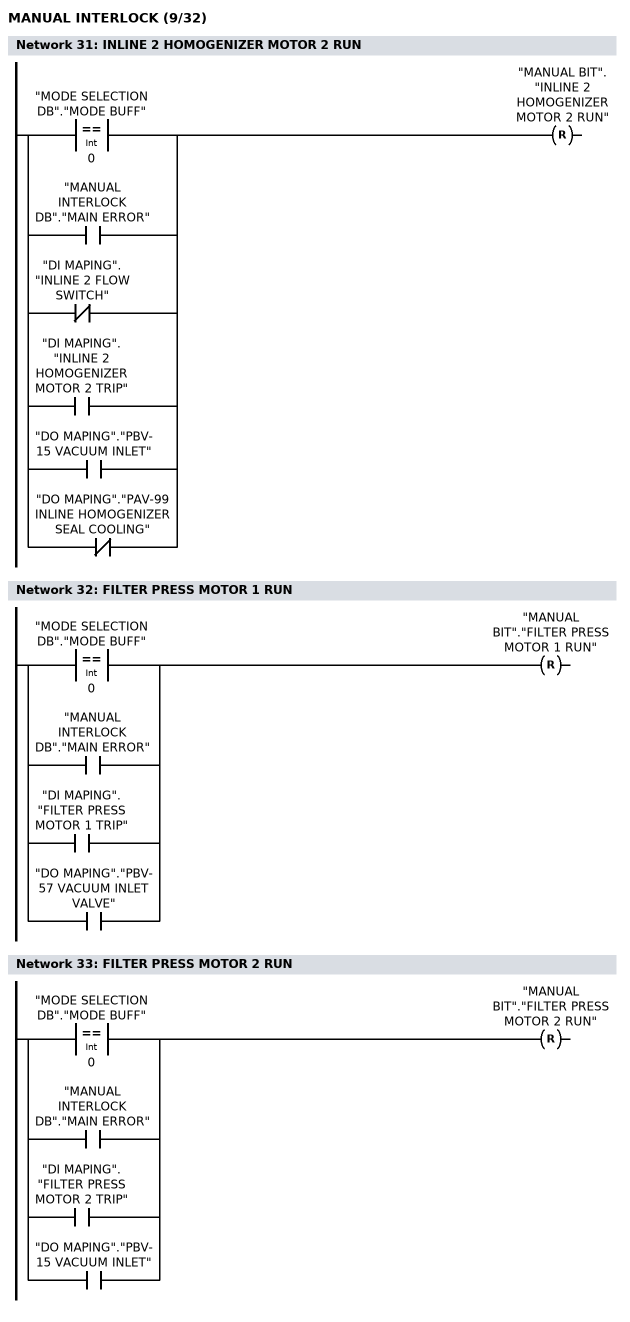
   RUNG wire#powerrail
      { S7_Templates := "SrcType := Int" } EQ_Contact(in1 := "MODE SELECTION DB"."MODE BUFF", in2 := 0)
      wire#w1
      R_Coil( "MANUAL BIT"."INLINE 2 HOMOGENIZER MOTOR 2 RUN" )
   END_RUNG
   RUNG wire#powerrail
      Contact( "MANUAL INTERLOCK DB"."MAIN ERROR" )
   END_RUNG wire#w1
   RUNG wire#powerrail
      I_Contact( "DI MAPING"."INLINE 2 FLOW SWITCH" )
   END_RUNG wire#w1
   RUNG wire#powerrail
      Contact( "DI MAPING"."INLINE 2 HOMOGENIZER MOTOR 2 TRIP" )
   END_RUNG wire#w1
   RUNG wire#powerrail
      Contact( "DO MAPING"."PBV-15 VACUUM INLET" )
   END_RUNG wire#w1
   RUNG wire#powerrail
      I_Contact( "DO MAPING"."PAV-99 INLINE HOMOGENIZER SEAL COOLING" )
   END_RUNG wire#w1
   // the same network as SCL:
   IF ("MODE SELECTION DB"."MODE BUFF" = 0) OR "MANUAL INTERLOCK DB"."MAIN ERROR" OR NOT "DI MAPING"."INLINE 2 FLOW SWITCH" OR "DI MAPING"."INLINE 2 HOMOGENIZER MOTOR 2 TRIP" OR "DO MAPING"."PBV-15 VACUUM INLET" OR NOT "DO MAPING"."PAV-99 INLINE HOMOGENIZER SEAL COOLING" THEN
       "MANUAL BIT"."INLINE 2 HOMOGENIZER MOTOR 2 RUN" := FALSE;
   END_IF;
END_REGION

REGION Network 32: FILTER PRESS MOTOR 1 RUN
   RUNG wire#powerrail
      { S7_Templates := "SrcType := Int" } EQ_Contact(in1 := "MODE SELECTION DB"."MODE BUFF", in2 := 0)
      wire#w1
      R_Coil( "MANUAL BIT"."FILTER PRESS MOTOR 1 RUN" )
   END_RUNG
   RUNG wire#powerrail
      Contact( "MANUAL INTERLOCK DB"."MAIN ERROR" )
   END_RUNG wire#w1
   RUNG wire#powerrail
      Contact( "DI MAPING"."FILTER PRESS MOTOR 1 TRIP" )
   END_RUNG wire#w1
   RUNG wire#powerrail
      Contact( "DO MAPING"."PBV-57 VACUUM INLET VALVE" )
   END_RUNG wire#w1
   // the same network as SCL:
   IF ("MODE SELECTION DB"."MODE BUFF" = 0) OR "MANUAL INTERLOCK DB"."MAIN ERROR" OR "DI MAPING"."FILTER PRESS MOTOR 1 TRIP" OR "DO MAPING"."PBV-57 VACUUM INLET VALVE" THEN
       "MANUAL BIT"."FILTER PRESS MOTOR 1 RUN" := FALSE;
   END_IF;
END_REGION

REGION Network 33: FILTER PRESS MOTOR 2 RUN
   RUNG wire#powerrail
      { S7_Templates := "SrcType := Int" } EQ_Contact(in1 := "MODE SELECTION DB"."MODE BUFF", in2 := 0)
      wire#w1
      R_Coil( "MANUAL BIT"."FILTER PRESS MOTOR 2 RUN" )
   END_RUNG
   RUNG wire#powerrail
      Contact( "MANUAL INTERLOCK DB"."MAIN ERROR" )
   END_RUNG wire#w1
   RUNG wire#powerrail
      Contact( "DI MAPING"."FILTER PRESS MOTOR 2 TRIP" )
   END_RUNG wire#w1
   RUNG wire#powerrail
      Contact( "DO MAPING"."PBV-15 VACUUM INLET" )
   END_RUNG wire#w1
   // the same network as SCL:
   IF ("MODE SELECTION DB"."MODE BUFF" = 0) OR "MANUAL INTERLOCK DB"."MAIN ERROR" OR "DI MAPING"."FILTER PRESS MOTOR 2 TRIP" OR "DO MAPING"."PBV-15 VACUUM INLET" THEN
       "MANUAL BIT"."FILTER PRESS MOTOR 2 RUN" := FALSE;
   END_IF;
END_REGION

REGION Network 34: VACCUM PUMP MOTOR 1 RUN
